       Chars_TO_Strg(Chars := #statDataBuffer.rcv_bddResult,
                     pChars := 2175,
                     Cnt := 8,
                     Strg => #statMonitoring.bddData.dataValue[90]);
       Chars_TO_Strg(Chars := #statDataBuffer.rcv_bddResult,
                     pChars := 2199,
                     Cnt := 8,
                     Strg => #statMonitoring.bddData.dataValue[91]);
       Chars_TO_Strg(Chars := #statDataBuffer.rcv_bddResult,
                     pChars := 2223,
                     Cnt := 8,
                     Strg => #statMonitoring.bddData.dataValue[92]);
       Chars_TO_Strg(Chars := #statDataBuffer.rcv_bddResult,
                     pChars := 2247,
                     Cnt := 8,
                     Strg => #statMonitoring.bddData.dataValue[93]);
       Chars_TO_Strg(Chars := #statDataBuffer.rcv_bddResult,
                     pChars := 2271,
                     Cnt := 8,
                     Strg => #statMonitoring.bddData.dataValue[94]);
       Chars_TO_Strg(Chars := #statDataBuffer.rcv_bddResult,
                     pChars := 2295,
                     Cnt := 8,
                     Strg => #statMonitoring.bddData.dataValue[95]);
       Chars_TO_Strg(Chars := #statDataBuffer.rcv_bddResult,
                     pChars := 2319,
                     Cnt := 8,
                     Strg => #statMonitoring.bddData.dataValue[96]);
       Chars_TO_Strg(Chars := #statDataBuffer.rcv_bddResult,
                     pChars := 2343,
                     Cnt := 8,
                     Strg => #statMonitoring.bddData.dataValue[97]);
       Chars_TO_Strg(Chars := #statDataBuffer.rcv_bddResult,
                     pChars := 2367,
                     Cnt := 8,
                     Strg => #statMonitoring.bddData.dataValue[98]);
       Chars_TO_Strg(Chars := #statDataBuffer.rcv_bddResult,
                     pChars := 2391,
                     Cnt := 8,
                     Strg => #statMonitoring.bddData.dataValue[99]);

       #instTON_bddResult[1](IN := TRUE,
                             PT := T#5000ms);

       IF #instTON_bddResult[1].Q THEN
           #statStep := 430;
       END_IF;
   END_IF;
END_REGION

REGION Network 43: STEP 430 : Bdd count complete
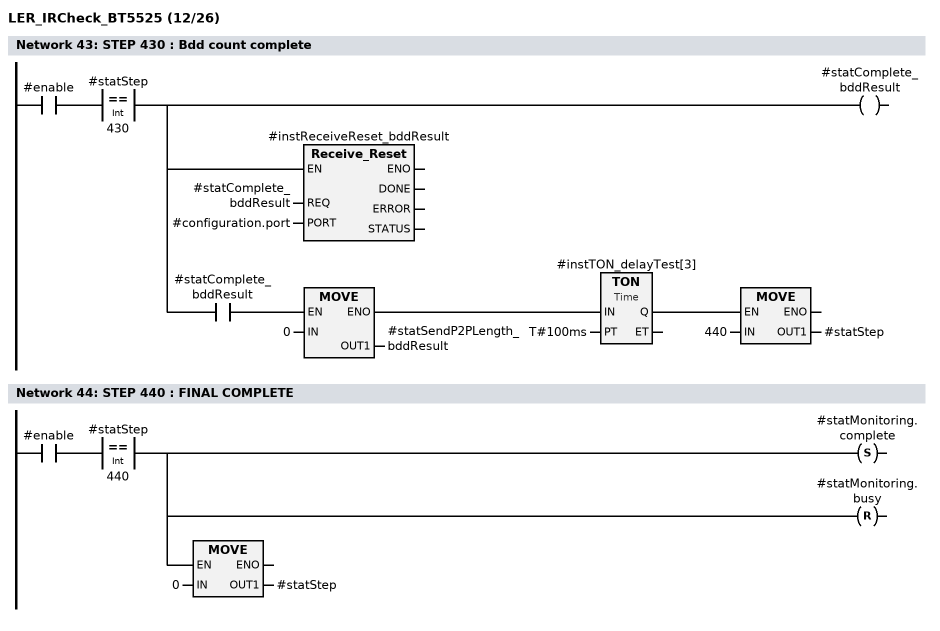
   RUNG wire#powerrail
      Contact( #enable )
      { S7_Templates := "SrcType := Int" } EQ_Contact(in1 := #statStep, in2 := 430)
      wire#w1
      Coil( #statComplete_bddResult )
   END_RUNG
   RUNG wire#w1
      #instReceiveReset_bddResult.Receive_Reset(REQ := #statComplete_bddResult, PORT := #configuration.port, DONE =>, ERROR =>, STATUS =>)
   END_RUNG
   RUNG wire#w1
      Contact( #statComplete_bddResult )
      Move(in := 0, out1 => #statSendP2PLength_bddResult)
      { S7_Templates := "time_type := Time" } #instTON_delayTest[3].TON(pt := T#100ms, et =>)
      Move(in := 440, out1 => #statStep)
   END_RUNG
   // the same network as SCL:
   #statComplete_bddResult := #enable AND (#statStep = 430);
   IF #statComplete_bddResult THEN
       #instReceiveReset_bddResult(REQ := #statComplete_bddResult, PORT := #configuration.port);   // Receive_Reset
   END_IF;
   #_w1 := #statComplete_bddResult AND #statComplete_bddResult;
   IF #_w1 THEN #statSendP2PLength_bddResult := 0; END_IF;
   #instTON_delayTest[3].TON(IN := #_w1, PT := T#100ms);
   IF #instTON_delayTest[3].Q THEN #statStep := 440; END_IF;
END_REGION

REGION Network 44: STEP 440 : FINAL COMPLETE
   RUNG wire#powerrail
      Contact( #enable )
      { S7_Templates := "SrcType := Int" } EQ_Contact(in1 := #statStep, in2 := 440)
      wire#w1
      S_Coil( #statMonitoring.complete )
   END_RUNG
   RUNG wire#w1
      R_Coil( #statMonitoring.busy )
   END_RUNG
   RUNG wire#w1
      Move(in := 0, out1 => #statStep)
   END_RUNG
   // the same network as SCL:
   IF #enable AND (#statStep = 440) THEN
       #statMonitoring.complete := TRUE;
       #statMonitoring.busy := FALSE;
       #statStep := 0;
   END_IF;
END_REGION

REGION Network 45: ========================================== SEQUENCE STEP [PARAMETER]
END_REGION

REGION Network 46: STEP 1000~1030 : VOLTAGE COMMAND
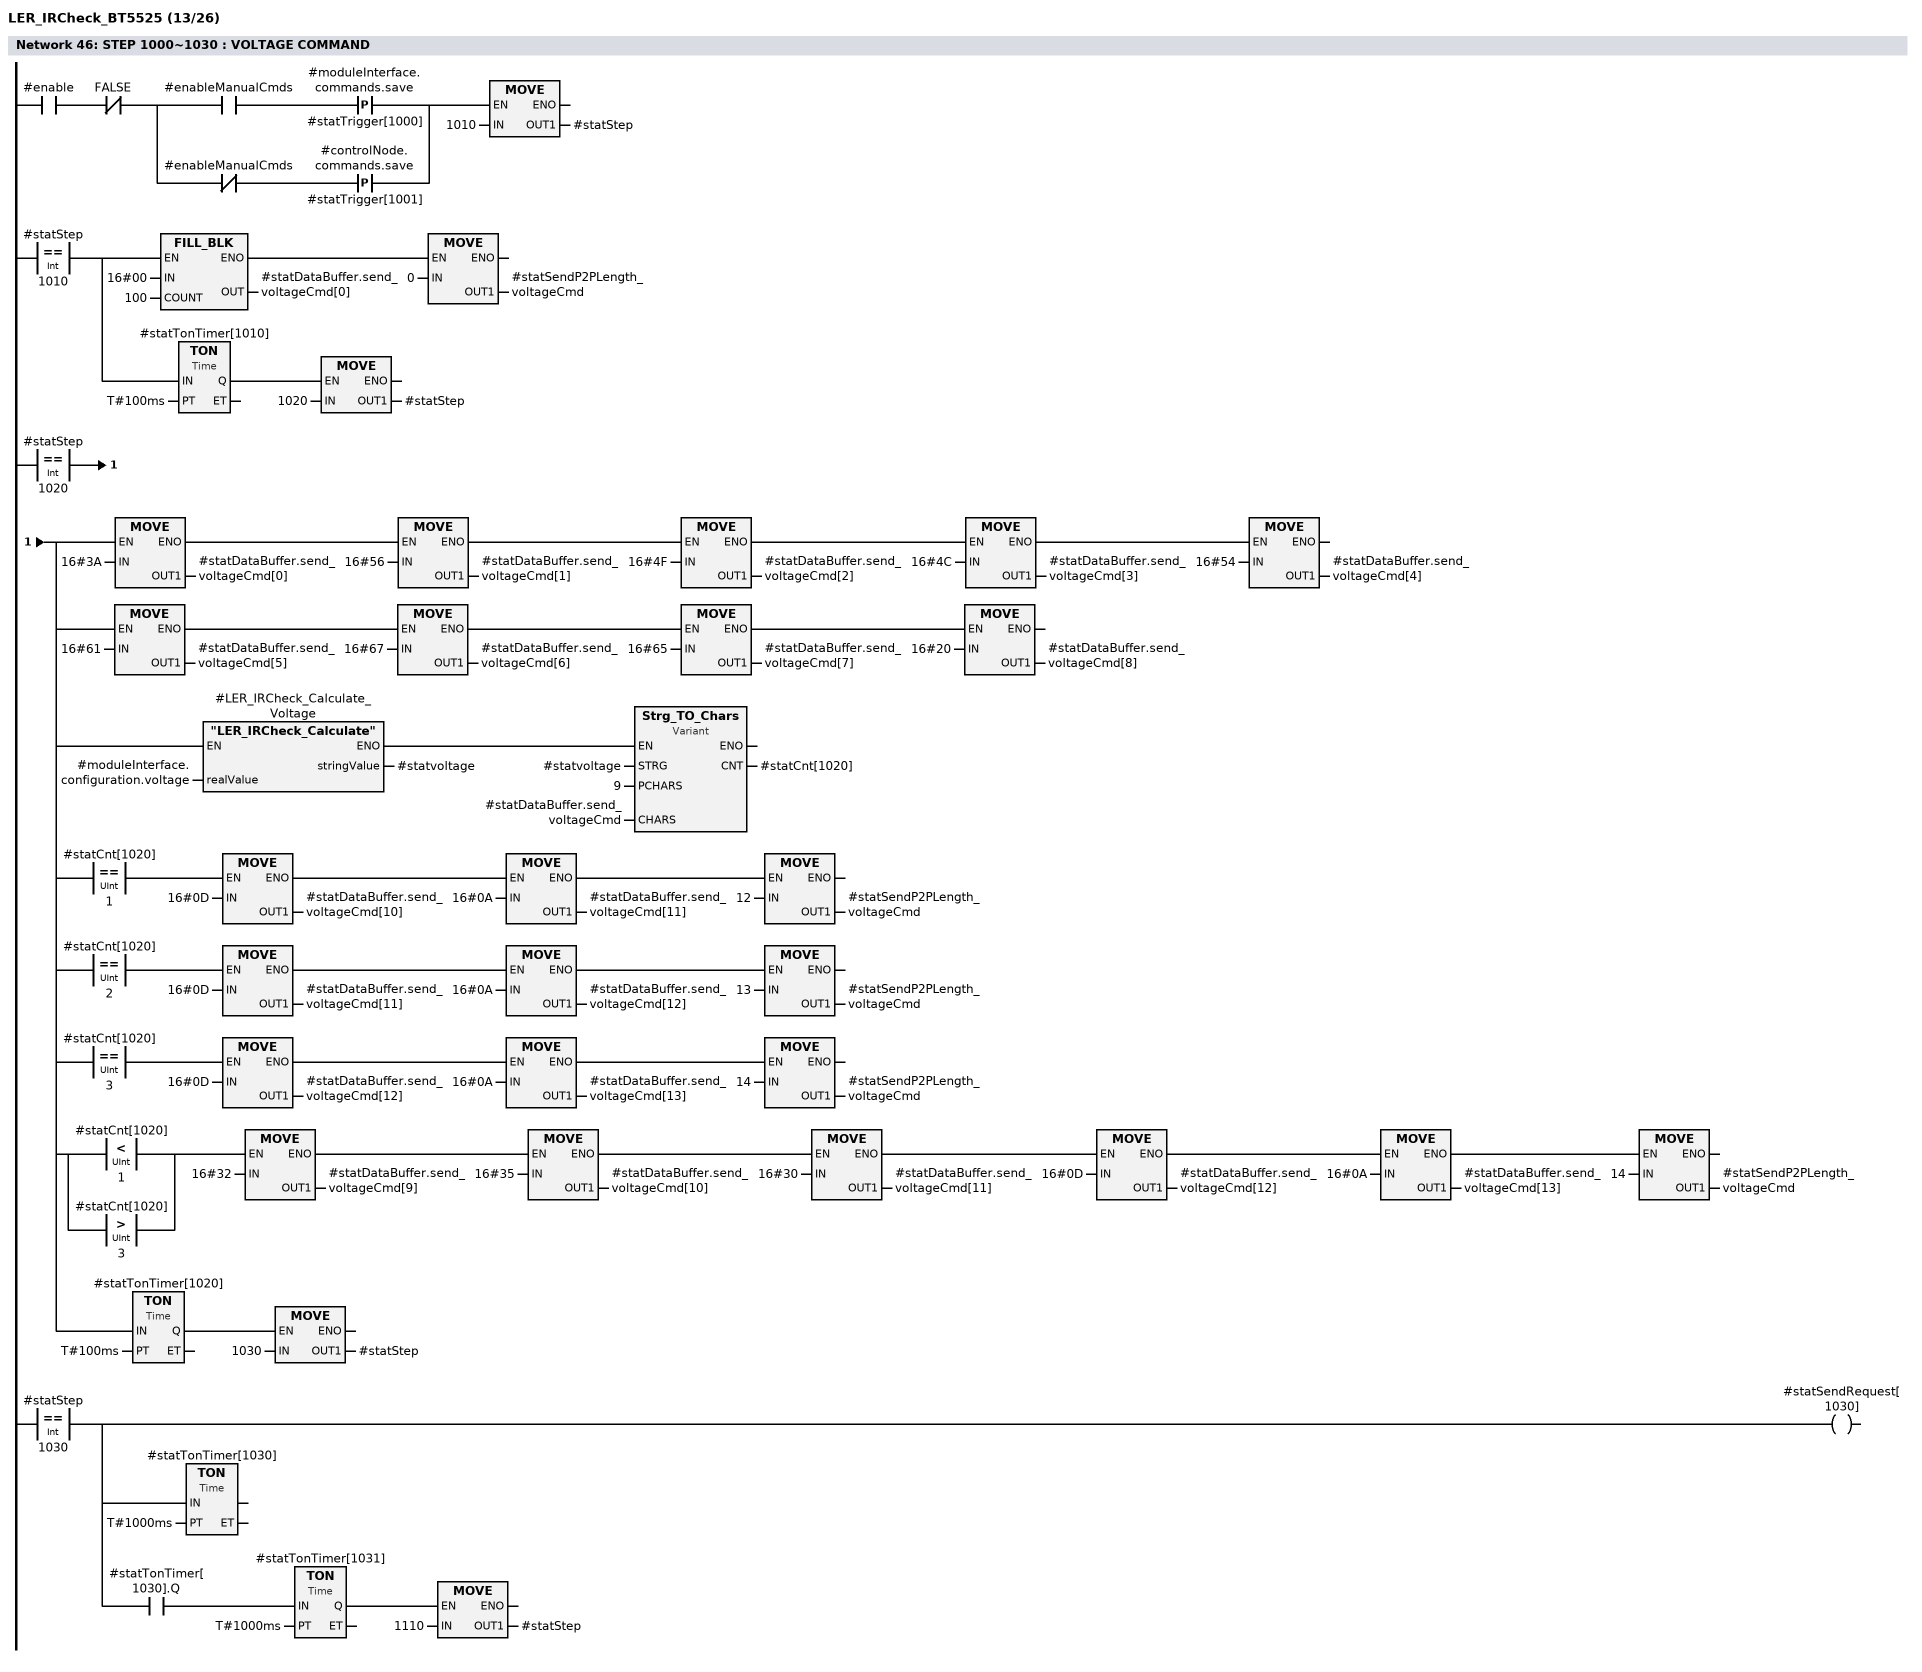
   RUNG wire#powerrail
      Contact( #enable )
      I_Contact( FALSE )
      wire#w1
      Contact( #enableManualCmds )
      P_Contact(operand := #moduleInterface.commands.save, bit := #statTrigger[1000])
      wire#w2
      Move(in := 1010, out1 => #statStep)
   END_RUNG
   RUNG wire#w1
      I_Contact( #enableManualCmds )
      P_Contact(operand := #controlNode.commands.save, bit := #statTrigger[1001])
   END_RUNG wire#w2
   RUNG wire#powerrail
      { S7_Templates := "SrcType := Int" } EQ_Contact(in1 := #statStep, in2 := 1010)
      wire#w3
      FillBlockI(in := 16#00, count := 100, out => #statDataBuffer.send_voltageCmd[0])
      Move(in := 0, out1 => #statSendP2PLength_voltageCmd)
   END_RUNG
   RUNG wire#w3
      { S7_Templates := "time_type := Time" } #statTonTimer[1010].TON(pt := T#100ms, et =>)
      Move(in := 1020, out1 => #statStep)
   END_RUNG
   RUNG wire#powerrail
      { S7_Templates := "SrcType := Int" } EQ_Contact(in1 := #statStep, in2 := 1020)
      wire#w4
      Move(in := 16#3A, out1 => #statDataBuffer.send_voltageCmd[0])
      Move(in := 16#56, out1 => #statDataBuffer.send_voltageCmd[1])
      Move(in := 16#4F, out1 => #statDataBuffer.send_voltageCmd[2])
      Move(in := 16#4C, out1 => #statDataBuffer.send_voltageCmd[3])
      Move(in := 16#54, out1 => #statDataBuffer.send_voltageCmd[4])
   END_RUNG
   RUNG wire#w4
      Move(in := 16#61, out1 => #statDataBuffer.send_voltageCmd[5])
      Move(in := 16#67, out1 => #statDataBuffer.send_voltageCmd[6])
      Move(in := 16#65, out1 => #statDataBuffer.send_voltageCmd[7])
      Move(in := 16#20, out1 => #statDataBuffer.send_voltageCmd[8])
   END_RUNG
   RUNG wire#w4
      #LER_IRCheck_Calculate_Voltage(realValue := #moduleInterface.configuration.voltage, stringValue => #statvoltage)
      { S7_Templates := "[ptr_type := Variant, strg_type := String]" } Strg_TO_Chars(Strg := #statvoltage, pChars := 9, Chars := #statDataBuffer.send_voltageCmd, Cnt => #statCnt[1020])
   END_RUNG
   RUNG wire#w4
      { S7_Templates := "SrcType := UInt" } EQ_Contact(in1 := #statCnt[1020], in2 := 1)
      Move(in := 16#0D, out1 => #statDataBuffer.send_voltageCmd[10])
      Move(in := 16#0A, out1 => #statDataBuffer.send_voltageCmd[11])
      Move(in := 12, out1 => #statSendP2PLength_voltageCmd)
   END_RUNG
   RUNG wire#w4
      { S7_Templates := "SrcType := UInt" } EQ_Contact(in1 := #statCnt[1020], in2 := 2)
      Move(in := 16#0D, out1 => #statDataBuffer.send_voltageCmd[11])
      Move(in := 16#0A, out1 => #statDataBuffer.send_voltageCmd[12])
      Move(in := 13, out1 => #statSendP2PLength_voltageCmd)
   END_RUNG
   RUNG wire#w4
      { S7_Templates := "SrcType := UInt" } EQ_Contact(in1 := #statCnt[1020], in2 := 3)
      Move(in := 16#0D, out1 => #statDataBuffer.send_voltageCmd[12])
      Move(in := 16#0A, out1 => #statDataBuffer.send_voltageCmd[13])
      Move(in := 14, out1 => #statSendP2PLength_voltageCmd)
   END_RUNG
   RUNG wire#w4
      { S7_Templates := "SrcType := UInt" } LT_Contact(in1 := #statCnt[1020], in2 := 1)
      wire#w5
      Move(in := 16#32, out1 => #statDataBuffer.send_voltageCmd[9])
      Move(in := 16#35, out1 => #statDataBuffer.send_voltageCmd[10])
      Move(in := 16#30, out1 => #statDataBuffer.send_voltageCmd[11])
      Move(in := 16#0D, out1 => #statDataBuffer.send_voltageCmd[12])
      Move(in := 16#0A, out1 => #statDataBuffer.send_voltageCmd[13])
      Move(in := 14, out1 => #statSendP2PLength_voltageCmd)
   END_RUNG
   RUNG wire#w4
      { S7_Templates := "SrcType := UInt" } GT_Contact(in1 := #statCnt[1020], in2 := 3)
   END_RUNG wire#w5
   RUNG wire#w4
      { S7_Templates := "time_type := Time" } #statTonTimer[1020].TON(pt := T#100ms, et =>)
      Move(in := 1030, out1 => #statStep)
   END_RUNG
   RUNG wire#powerrail
      { S7_Templates := "SrcType := Int" } EQ_Contact(in1 := #statStep, in2 := 1030)
      wire#w6
      Coil( #statSendRequest[1030] )
   END_RUNG
   RUNG wire#w6
      { S7_Templates := "time_type := Time" } #statTonTimer[1030].TON(pt := T#1000ms, et =>)
   END_RUNG
   RUNG wire#w6
      Contact( #statTonTimer[1030].Q )
      { S7_Templates := "time_type := Time" } #statTonTimer[1031].TON(pt := T#1000ms, et =>)
      Move(in := 1110, out1 => #statStep)
   END_RUNG
   // the same network as SCL:
   #_w1 := #enable AND NOT FALSE AND #enableManualCmds AND #moduleInterface.commands.save AND NOT #statTrigger[1000];   // rising edge of #moduleInterface.commands.save
   #statTrigger[1000] := #moduleInterface.commands.save;
   #_w2 := #enable AND NOT FALSE AND NOT #enableManualCmds AND #controlNode.commands.save AND NOT #statTrigger[1001];   // rising edge of #controlNode.commands.save
   #statTrigger[1001] := #controlNode.commands.save;
   IF #_w1 OR #_w2 THEN #statStep := 1010; END_IF;
   #_w3 := #statStep = 1010;
   IF #_w3 THEN
       FILL_BLK(IN := 16#00, COUNT := 100, OUT => #statDataBuffer.send_voltageCmd[0]);
       #statSendP2PLength_voltageCmd := 0;
   END_IF;
   #statTonTimer[1010].TON(IN := #_w3, PT := T#100ms);
   IF #statTonTimer[1010].Q THEN #statStep := 1020; END_IF;
   #_w4 := #statStep = 1020;
   IF #_w4 THEN
       #statDataBuffer.send_voltageCmd[0] := 16#3A;
       #statDataBuffer.send_voltageCmd[1] := 16#56;
       #statDataBuffer.send_voltageCmd[2] := 16#4F;
       #statDataBuffer.send_voltageCmd[3] := 16#4C;
       #statDataBuffer.send_voltageCmd[4] := 16#54;
       #statDataBuffer.send_voltageCmd[5] := 16#61;
       #statDataBuffer.send_voltageCmd[6] := 16#67;
       #statDataBuffer.send_voltageCmd[7] := 16#65;
       #statDataBuffer.send_voltageCmd[8] := 16#20;
   END_IF;
   #LER_IRCheck_Calculate_Voltage(EN := #_w4,   // "LER_IRCheck_Calculate"
                           realValue := #moduleInterface.configuration.voltage,
                           stringValue => #statvoltage,
                           ENO => #_w5);
   IF #_w5 THEN
       Strg_TO_Chars(Strg := #statvoltage,
                     pChars := 9,
                     Chars := #statDataBuffer.send_voltageCmd,
                     Cnt => #statCnt[1020]);
   END_IF;
   IF #_w4 AND (#statCnt[1020] = 1) THEN
       #statDataBuffer.send_voltageCmd[10] := 16#0D;
       #statDataBuffer.send_voltageCmd[11] := 16#0A;
       #statSendP2PLength_voltageCmd := 12;
   END_IF;
   IF #_w4 AND (#statCnt[1020] = 2) THEN
       #statDataBuffer.send_voltageCmd[11] := 16#0D;
       #statDataBuffer.send_voltageCmd[12] := 16#0A;
       #statSendP2PLength_voltageCmd := 13;
   END_IF;
   IF #_w4 AND (#statCnt[1020] = 3) THEN
       #statDataBuffer.send_voltageCmd[12] := 16#0D;
       #statDataBuffer.send_voltageCmd[13] := 16#0A;
       #statSendP2PLength_voltageCmd := 14;
   END_IF;
   IF #_w4 AND ((#statCnt[1020] < 1) OR (#statCnt[1020] > 3)) THEN
       #statDataBuffer.send_voltageCmd[9] := 16#32;
       #statDataBuffer.send_voltageCmd[10] := 16#35;
       #statDataBuffer.send_voltageCmd[11] := 16#30;
       #statDataBuffer.send_voltageCmd[12] := 16#0D;
       #statDataBuffer.send_voltageCmd[13] := 16#0A;
       #statSendP2PLength_voltageCmd := 14;
   END_IF;
   #statTonTimer[1020].TON(IN := #_w4, PT := T#100ms);
   IF #statTonTimer[1020].Q THEN #statStep := 1030; END_IF;
   #statSendRequest[1030] := #statStep = 1030;
   #statTonTimer[1030].TON(IN := #statStep = 1030, PT := T#1000ms);
   #statTonTimer[1031].TON(IN := (#statStep = 1030) AND #statTonTimer[1030].Q, PT := T#1000ms);
   IF #statTonTimer[1031].Q THEN #statStep := 1110; END_IF;
END_REGION

REGION Network 47: STEP 1110~1140 : VOLTAGE CHECK
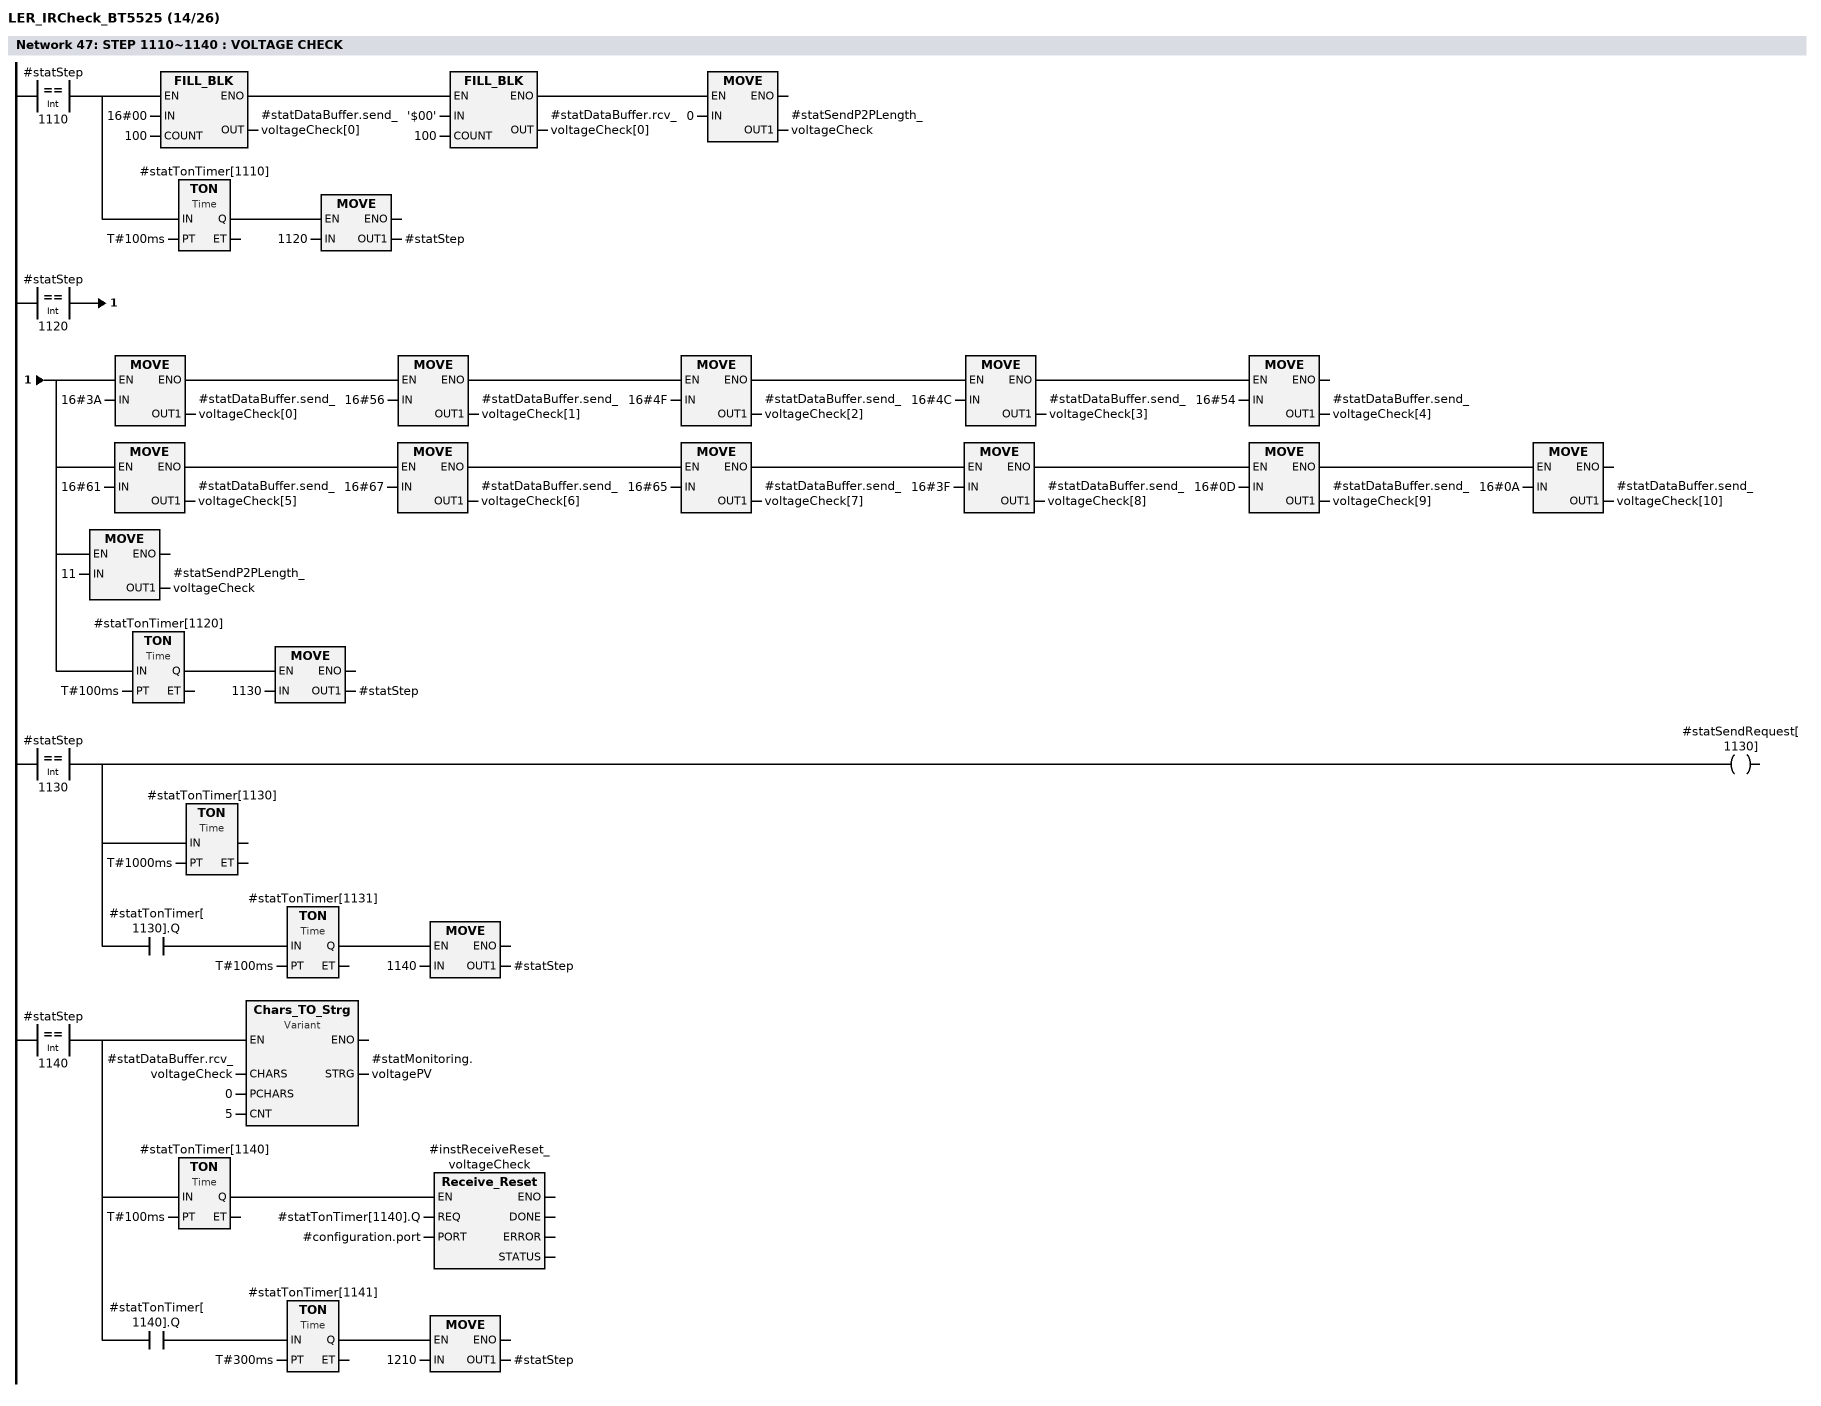
   RUNG wire#powerrail
      { S7_Templates := "SrcType := Int" } EQ_Contact(in1 := #statStep, in2 := 1110)
      wire#w1
      FillBlockI(in := 16#00, count := 100, out => #statDataBuffer.send_voltageCheck[0])
      FillBlockI(in := '$00', count := 100, out => #statDataBuffer.rcv_voltageCheck[0])
      Move(in := 0, out1 => #statSendP2PLength_voltageCheck)
   END_RUNG
   RUNG wire#w1
      { S7_Templates := "time_type := Time" } #statTonTimer[1110].TON(pt := T#100ms, et =>)
      Move(in := 1120, out1 => #statStep)
   END_RUNG
   RUNG wire#powerrail
      { S7_Templates := "SrcType := Int" } EQ_Contact(in1 := #statStep, in2 := 1120)
      wire#w2
      Move(in := 16#3A, out1 => #statDataBuffer.send_voltageCheck[0])
      Move(in := 16#56, out1 => #statDataBuffer.send_voltageCheck[1])
      Move(in := 16#4F, out1 => #statDataBuffer.send_voltageCheck[2])
      Move(in := 16#4C, out1 => #statDataBuffer.send_voltageCheck[3])
      Move(in := 16#54, out1 => #statDataBuffer.send_voltageCheck[4])
   END_RUNG
   RUNG wire#w2
      Move(in := 16#61, out1 => #statDataBuffer.send_voltageCheck[5])
      Move(in := 16#67, out1 => #statDataBuffer.send_voltageCheck[6])
      Move(in := 16#65, out1 => #statDataBuffer.send_voltageCheck[7])
      Move(in := 16#3F, out1 => #statDataBuffer.send_voltageCheck[8])
      Move(in := 16#0D, out1 => #statDataBuffer.send_voltageCheck[9])
      Move(in := 16#0A, out1 => #statDataBuffer.send_voltageCheck[10])
   END_RUNG
   RUNG wire#w2
      Move(in := 11, out1 => #statSendP2PLength_voltageCheck)
   END_RUNG
   RUNG wire#w2
      { S7_Templates := "time_type := Time" } #statTonTimer[1120].TON(pt := T#100ms, et =>)
      Move(in := 1130, out1 => #statStep)
   END_RUNG
   RUNG wire#powerrail
      { S7_Templates := "SrcType := Int" } EQ_Contact(in1 := #statStep, in2 := 1130)
      wire#w3
      Coil( #statSendRequest[1130] )
   END_RUNG
   RUNG wire#w3
      { S7_Templates := "time_type := Time" } #statTonTimer[1130].TON(pt := T#1000ms, et =>)
   END_RUNG
   RUNG wire#w3
      Contact( #statTonTimer[1130].Q )
      { S7_Templates := "time_type := Time" } #statTonTimer[1131].TON(pt := T#100ms, et =>)
      Move(in := 1140, out1 => #statStep)
   END_RUNG
   RUNG wire#powerrail
      { S7_Templates := "SrcType := Int" } EQ_Contact(in1 := #statStep, in2 := 1140)
      wire#w4
      { S7_Templates := "[ptr_type := Variant, str_type := String]" } Chars_TO_Strg(Chars := #statDataBuffer.rcv_voltageCheck, pChars := 0, Cnt := 5, Strg => #statMonitoring.voltagePV)
   END_RUNG
   RUNG wire#w4
      { S7_Templates := "time_type := Time" } #statTonTimer[1140].TON(pt := T#100ms, et =>)
      #instReceiveReset_voltageCheck.Receive_Reset(REQ := #statTonTimer[1140].Q, PORT := #configuration.port, DONE =>, ERROR =>, STATUS =>)
   END_RUNG
   RUNG wire#w4
      Contact( #statTonTimer[1140].Q )
      { S7_Templates := "time_type := Time" } #statTonTimer[1141].TON(pt := T#300ms, et =>)
      Move(in := 1210, out1 => #statStep)
   END_RUNG
   // the same network as SCL:
   #_w1 := #statStep = 1110;
   IF #_w1 THEN
       FILL_BLK(IN := 16#00, COUNT := 100, OUT => #statDataBuffer.send_voltageCheck[0]);
       FILL_BLK(IN := '$00', COUNT := 100, OUT => #statDataBuffer.rcv_voltageCheck[0]);
       #statSendP2PLength_voltageCheck := 0;
   END_IF;
   #statTonTimer[1110].TON(IN := #_w1, PT := T#100ms);
   IF #statTonTimer[1110].Q THEN #statStep := 1120; END_IF;
   #_w2 := #statStep = 1120;
   IF #_w2 THEN
       #statDataBuffer.send_voltageCheck[0] := 16#3A;
       #statDataBuffer.send_voltageCheck[1] := 16#56;
       #statDataBuffer.send_voltageCheck[2] := 16#4F;
       #statDataBuffer.send_voltageCheck[3] := 16#4C;
       #statDataBuffer.send_voltageCheck[4] := 16#54;
       #statDataBuffer.send_voltageCheck[5] := 16#61;
       #statDataBuffer.send_voltageCheck[6] := 16#67;
       #statDataBuffer.send_voltageCheck[7] := 16#65;
       #statDataBuffer.send_voltageCheck[8] := 16#3F;
       #statDataBuffer.send_voltageCheck[9] := 16#0D;
       #statDataBuffer.send_voltageCheck[10] := 16#0A;
       #statSendP2PLength_voltageCheck := 11;
   END_IF;
   #statTonTimer[1120].TON(IN := #_w2, PT := T#100ms);
   IF #statTonTimer[1120].Q THEN #statStep := 1130; END_IF;
   #statSendRequest[1130] := #statStep = 1130;
   #statTonTimer[1130].TON(IN := #statStep = 1130, PT := T#1000ms);
   #statTonTimer[1131].TON(IN := (#statStep = 1130) AND #statTonTimer[1130].Q, PT := T#100ms);
   IF #statTonTimer[1131].Q THEN #statStep := 1140; END_IF;
   #_w3 := #statStep = 1140;
   IF #_w3 THEN
       Chars_TO_Strg(Chars := #statDataBuffer.rcv_voltageCheck,
                     pChars := 0,
                     Cnt := 5,
                     Strg => #statMonitoring.voltagePV);
   END_IF;
   #statTonTimer[1140].TON(IN := #_w3, PT := T#100ms);
   IF #statTonTimer[1140].Q THEN
       #instReceiveReset_voltageCheck(REQ := #statTonTimer[1140].Q, PORT := #configuration.port);   // Receive_Reset
   END_IF;
   #statTonTimer[1141].TON(IN := #_w3 AND #statTonTimer[1140].Q, PT := T#300ms);
   IF #statTonTimer[1141].Q THEN #statStep := 1210; END_IF;
END_REGION

REGION Network 48: STEP 1210~1230 : TIMER COMMAND
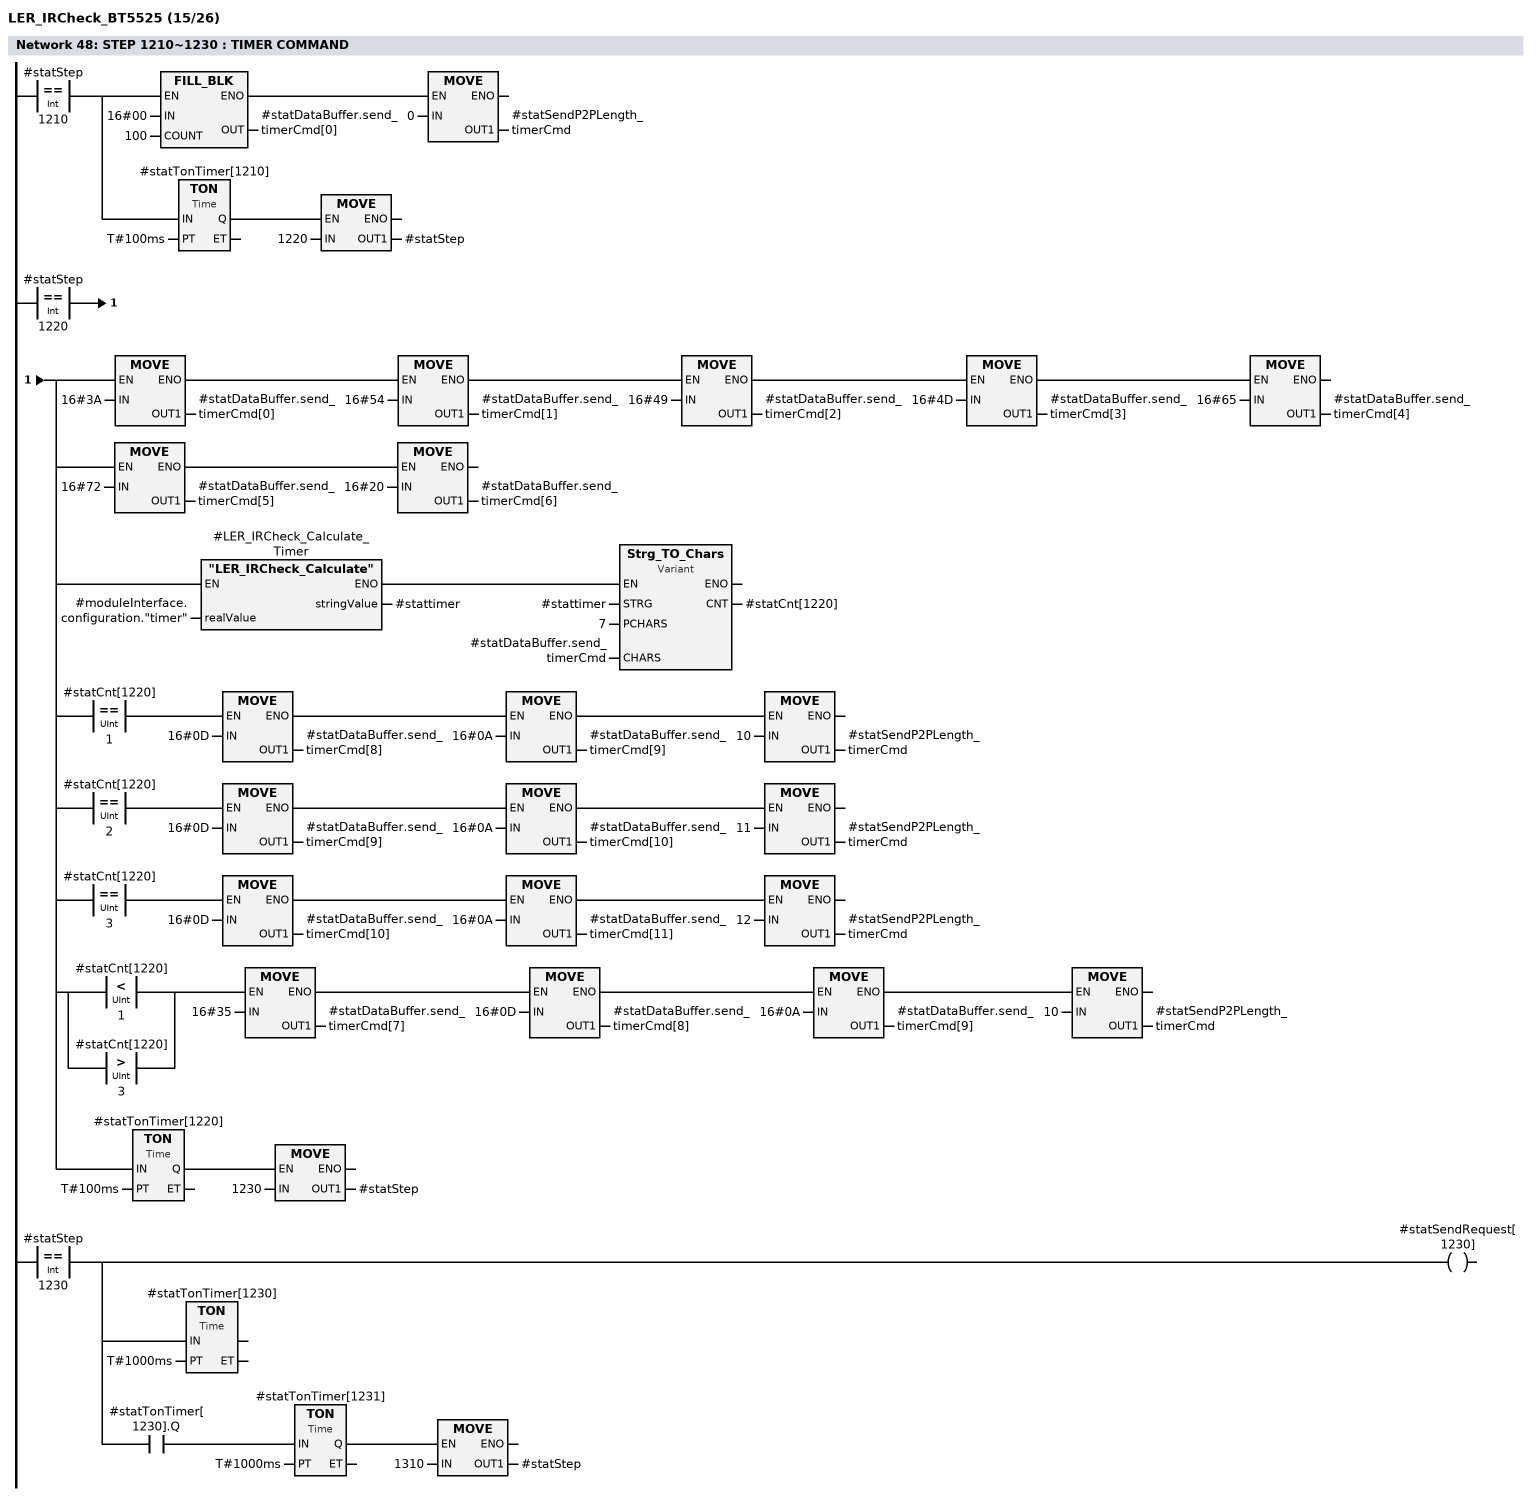
   RUNG wire#powerrail
      { S7_Templates := "SrcType := Int" } EQ_Contact(in1 := #statStep, in2 := 1210)
      wire#w1
      FillBlockI(in := 16#00, count := 100, out => #statDataBuffer.send_timerCmd[0])
      Move(in := 0, out1 => #statSendP2PLength_timerCmd)
   END_RUNG
   RUNG wire#w1
      { S7_Templates := "time_type := Time" } #statTonTimer[1210].TON(pt := T#100ms, et =>)
      Move(in := 1220, out1 => #statStep)
   END_RUNG
   RUNG wire#powerrail
      { S7_Templates := "SrcType := Int" } EQ_Contact(in1 := #statStep, in2 := 1220)
      wire#w2
      Move(in := 16#3A, out1 => #statDataBuffer.send_timerCmd[0])
      Move(in := 16#54, out1 => #statDataBuffer.send_timerCmd[1])
      Move(in := 16#49, out1 => #statDataBuffer.send_timerCmd[2])
      Move(in := 16#4D, out1 => #statDataBuffer.send_timerCmd[3])
      Move(in := 16#65, out1 => #statDataBuffer.send_timerCmd[4])
   END_RUNG
   RUNG wire#w2
      Move(in := 16#72, out1 => #statDataBuffer.send_timerCmd[5])
      Move(in := 16#20, out1 => #statDataBuffer.send_timerCmd[6])
   END_RUNG
   RUNG wire#w2
      #LER_IRCheck_Calculate_Timer(realValue := #moduleInterface.configuration."timer", stringValue => #stattimer)
      { S7_Templates := "[ptr_type := Variant, strg_type := String]" } Strg_TO_Chars(Strg := #stattimer, pChars := 7, Chars := #statDataBuffer.send_timerCmd, Cnt => #statCnt[1220])
   END_RUNG
   RUNG wire#w2
      { S7_Templates := "SrcType := UInt" } EQ_Contact(in1 := #statCnt[1220], in2 := 1)
      Move(in := 16#0D, out1 => #statDataBuffer.send_timerCmd[8])
      Move(in := 16#0A, out1 => #statDataBuffer.send_timerCmd[9])
      Move(in := 10, out1 => #statSendP2PLength_timerCmd)
   END_RUNG
   RUNG wire#w2
      { S7_Templates := "SrcType := UInt" } EQ_Contact(in1 := #statCnt[1220], in2 := 2)
      Move(in := 16#0D, out1 => #statDataBuffer.send_timerCmd[9])
      Move(in := 16#0A, out1 => #statDataBuffer.send_timerCmd[10])
      Move(in := 11, out1 => #statSendP2PLength_timerCmd)
   END_RUNG
   RUNG wire#w2
      { S7_Templates := "SrcType := UInt" } EQ_Contact(in1 := #statCnt[1220], in2 := 3)
      Move(in := 16#0D, out1 => #statDataBuffer.send_timerCmd[10])
      Move(in := 16#0A, out1 => #statDataBuffer.send_timerCmd[11])
      Move(in := 12, out1 => #statSendP2PLength_timerCmd)
   END_RUNG
   RUNG wire#w2
      { S7_Templates := "SrcType := UInt" } LT_Contact(in1 := #statCnt[1220], in2 := 1)
      wire#w3
      Move(in := 16#35, out1 => #statDataBuffer.send_timerCmd[7])
      Move(in := 16#0D, out1 => #statDataBuffer.send_timerCmd[8])
      Move(in := 16#0A, out1 => #statDataBuffer.send_timerCmd[9])
      Move(in := 10, out1 => #statSendP2PLength_timerCmd)
   END_RUNG
   RUNG wire#w2
      { S7_Templates := "SrcType := UInt" } GT_Contact(in1 := #statCnt[1220], in2 := 3)
   END_RUNG wire#w3
   RUNG wire#w2
      { S7_Templates := "time_type := Time" } #statTonTimer[1220].TON(pt := T#100ms, et =>)
      Move(in := 1230, out1 => #statStep)
   END_RUNG
   RUNG wire#powerrail
      { S7_Templates := "SrcType := Int" } EQ_Contact(in1 := #statStep, in2 := 1230)
      wire#w4
      Coil( #statSendRequest[1230] )
   END_RUNG
   RUNG wire#w4
      { S7_Templates := "time_type := Time" } #statTonTimer[1230].TON(pt := T#1000ms, et =>)
   END_RUNG
   RUNG wire#w4
      Contact( #statTonTimer[1230].Q )
      { S7_Templates := "time_type := Time" } #statTonTimer[1231].TON(pt := T#1000ms, et =>)
      Move(in := 1310, out1 => #statStep)
   END_RUNG
   // the same network as SCL:
   #_w1 := #statStep = 1210;
   IF #_w1 THEN
       FILL_BLK(IN := 16#00, COUNT := 100, OUT => #statDataBuffer.send_timerCmd[0]);
       #statSendP2PLength_timerCmd := 0;
   END_IF;
   #statTonTimer[1210].TON(IN := #_w1, PT := T#100ms);
   IF #statTonTimer[1210].Q THEN #statStep := 1220; END_IF;
   #_w2 := #statStep = 1220;
   IF #_w2 THEN
       #statDataBuffer.send_timerCmd[0] := 16#3A;
       #statDataBuffer.send_timerCmd[1] := 16#54;
       #statDataBuffer.send_timerCmd[2] := 16#49;
       #statDataBuffer.send_timerCmd[3] := 16#4D;
       #statDataBuffer.send_timerCmd[4] := 16#65;
       #statDataBuffer.send_timerCmd[5] := 16#72;
       #statDataBuffer.send_timerCmd[6] := 16#20;
   END_IF;
   #LER_IRCheck_Calculate_Timer(EN := #_w2,   // "LER_IRCheck_Calculate"
                           realValue := #moduleInterface.configuration."timer",
                           stringValue => #stattimer,
                           ENO => #_w3);
   IF #_w3 THEN
       Strg_TO_Chars(Strg := #stattimer, pChars := 7, Chars := #statDataBuffer.send_timerCmd, Cnt => #statCnt[1220]);
   END_IF;
   IF #_w2 AND (#statCnt[1220] = 1) THEN
       #statDataBuffer.send_timerCmd[8] := 16#0D;
       #statDataBuffer.send_timerCmd[9] := 16#0A;
       #statSendP2PLength_timerCmd := 10;
   END_IF;
   IF #_w2 AND (#statCnt[1220] = 2) THEN
       #statDataBuffer.send_timerCmd[9] := 16#0D;
       #statDataBuffer.send_timerCmd[10] := 16#0A;
       #statSendP2PLength_timerCmd := 11;
   END_IF;
   IF #_w2 AND (#statCnt[1220] = 3) THEN
       #statDataBuffer.send_timerCmd[10] := 16#0D;
       #statDataBuffer.send_timerCmd[11] := 16#0A;
       #statSendP2PLength_timerCmd := 12;
   END_IF;
   IF #_w2 AND ((#statCnt[1220] < 1) OR (#statCnt[1220] > 3)) THEN
       #statDataBuffer.send_timerCmd[7] := 16#35;
       #statDataBuffer.send_timerCmd[8] := 16#0D;
       #statDataBuffer.send_timerCmd[9] := 16#0A;
       #statSendP2PLength_timerCmd := 10;
   END_IF;
   #statTonTimer[1220].TON(IN := #_w2, PT := T#100ms);
   IF #statTonTimer[1220].Q THEN #statStep := 1230; END_IF;
   #statSendRequest[1230] := #statStep = 1230;
   #statTonTimer[1230].TON(IN := #statStep = 1230, PT := T#1000ms);
   #statTonTimer[1231].TON(IN := (#statStep = 1230) AND #statTonTimer[1230].Q, PT := T#1000ms);
   IF #statTonTimer[1231].Q THEN #statStep := 1310; END_IF;
END_REGION

REGION Network 49: STEP 1310~1340 : TIMER CHECK
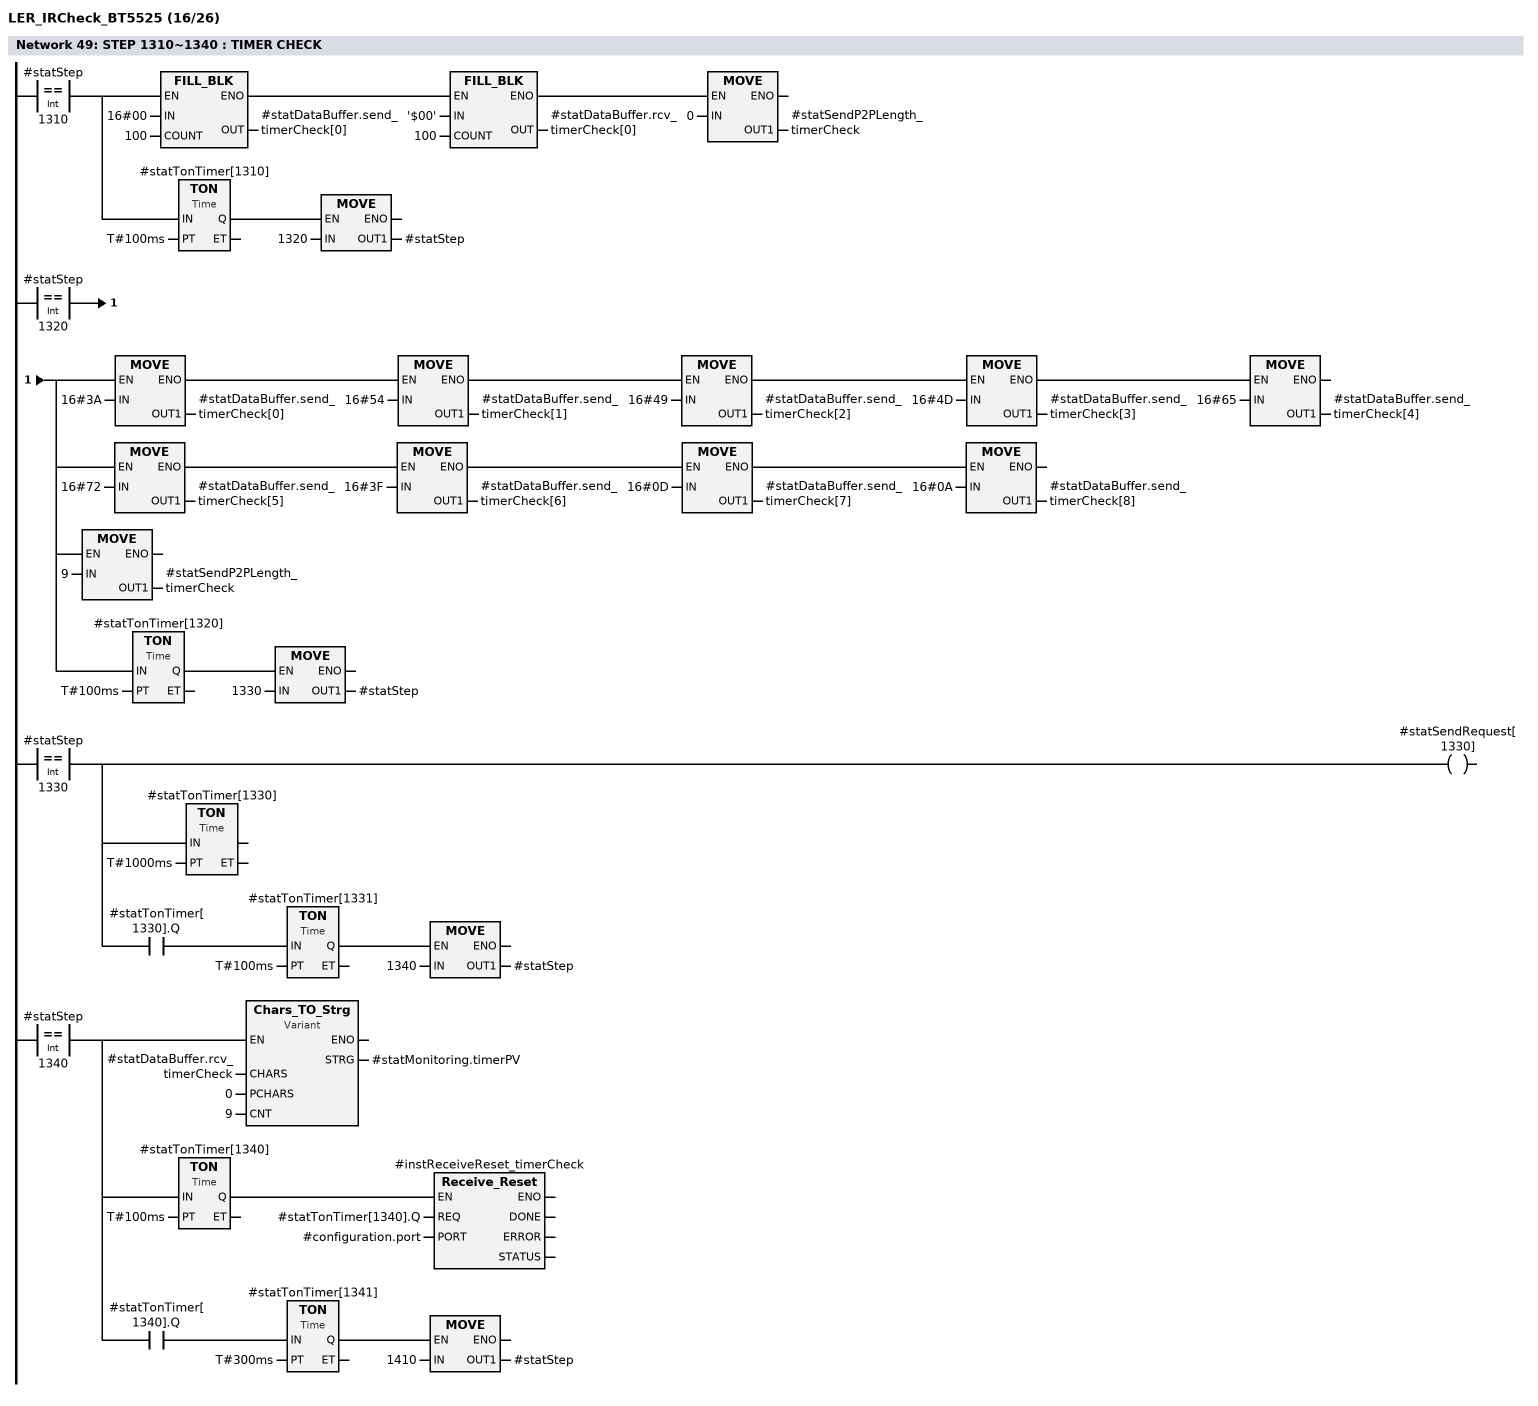
   RUNG wire#powerrail
      { S7_Templates := "SrcType := Int" } EQ_Contact(in1 := #statStep, in2 := 1310)
      wire#w1
      FillBlockI(in := 16#00, count := 100, out => #statDataBuffer.send_timerCheck[0])
      FillBlockI(in := '$00', count := 100, out => #statDataBuffer.rcv_timerCheck[0])
      Move(in := 0, out1 => #statSendP2PLength_timerCheck)
   END_RUNG
   RUNG wire#w1
      { S7_Templates := "time_type := Time" } #statTonTimer[1310].TON(pt := T#100ms, et =>)
      Move(in := 1320, out1 => #statStep)
   END_RUNG
   RUNG wire#powerrail
      { S7_Templates := "SrcType := Int" } EQ_Contact(in1 := #statStep, in2 := 1320)
      wire#w2
      Move(in := 16#3A, out1 => #statDataBuffer.send_timerCheck[0])
      Move(in := 16#54, out1 => #statDataBuffer.send_timerCheck[1])
      Move(in := 16#49, out1 => #statDataBuffer.send_timerCheck[2])
      Move(in := 16#4D, out1 => #statDataBuffer.send_timerCheck[3])
      Move(in := 16#65, out1 => #statDataBuffer.send_timerCheck[4])
   END_RUNG
   RUNG wire#w2
      Move(in := 16#72, out1 => #statDataBuffer.send_timerCheck[5])
      Move(in := 16#3F, out1 => #statDataBuffer.send_timerCheck[6])
      Move(in := 16#0D, out1 => #statDataBuffer.send_timerCheck[7])
      Move(in := 16#0A, out1 => #statDataBuffer.send_timerCheck[8])
   END_RUNG
   RUNG wire#w2
      Move(in := 9, out1 => #statSendP2PLength_timerCheck)
   END_RUNG
   RUNG wire#w2
      { S7_Templates := "time_type := Time" } #statTonTimer[1320].TON(pt := T#100ms, et =>)
      Move(in := 1330, out1 => #statStep)
   END_RUNG
   RUNG wire#powerrail
      { S7_Templates := "SrcType := Int" } EQ_Contact(in1 := #statStep, in2 := 1330)
      wire#w3
      Coil( #statSendRequest[1330] )
   END_RUNG
   RUNG wire#w3
      { S7_Templates := "time_type := Time" } #statTonTimer[1330].TON(pt := T#1000ms, et =>)
   END_RUNG
   RUNG wire#w3
      Contact( #statTonTimer[1330].Q )
      { S7_Templates := "time_type := Time" } #statTonTimer[1331].TON(pt := T#100ms, et =>)
      Move(in := 1340, out1 => #statStep)
   END_RUNG
   RUNG wire#powerrail
      { S7_Templates := "SrcType := Int" } EQ_Contact(in1 := #statStep, in2 := 1340)
      wire#w4
      { S7_Templates := "[ptr_type := Variant, str_type := String]" } Chars_TO_Strg(Chars := #statDataBuffer.rcv_timerCheck, pChars := 0, Cnt := 9, Strg => #statMonitoring.timerPV)
   END_RUNG
   RUNG wire#w4
      { S7_Templates := "time_type := Time" } #statTonTimer[1340].TON(pt := T#100ms, et =>)
      #instReceiveReset_timerCheck.Receive_Reset(REQ := #statTonTimer[1340].Q, PORT := #configuration.port, DONE =>, ERROR =>, STATUS =>)
   END_RUNG
   RUNG wire#w4
      Contact( #statTonTimer[1340].Q )
      { S7_Templates := "time_type := Time" } #statTonTimer[1341].TON(pt := T#300ms, et =>)
      Move(in := 1410, out1 => #statStep)
   END_RUNG
   // the same network as SCL:
   #_w1 := #statStep = 1310;
   IF #_w1 THEN
       FILL_BLK(IN := 16#00, COUNT := 100, OUT => #statDataBuffer.send_timerCheck[0]);
       FILL_BLK(IN := '$00', COUNT := 100, OUT => #statDataBuffer.rcv_timerCheck[0]);
       #statSendP2PLength_timerCheck := 0;
   END_IF;
   #statTonTimer[1310].TON(IN := #_w1, PT := T#100ms);
   IF #statTonTimer[1310].Q THEN #statStep := 1320; END_IF;
   #_w2 := #statStep = 1320;
   IF #_w2 THEN
       #statDataBuffer.send_timerCheck[0] := 16#3A;
       #statDataBuffer.send_timerCheck[1] := 16#54;
       #statDataBuffer.send_timerCheck[2] := 16#49;
       #statDataBuffer.send_timerCheck[3] := 16#4D;
       #statDataBuffer.send_timerCheck[4] := 16#65;
       #statDataBuffer.send_timerCheck[5] := 16#72;
       #statDataBuffer.send_timerCheck[6] := 16#3F;
       #statDataBuffer.send_timerCheck[7] := 16#0D;
       #statDataBuffer.send_timerCheck[8] := 16#0A;
       #statSendP2PLength_timerCheck := 9;
   END_IF;
   #statTonTimer[1320].TON(IN := #_w2, PT := T#100ms);
   IF #statTonTimer[1320].Q THEN #statStep := 1330; END_IF;
   #statSendRequest[1330] := #statStep = 1330;
   #statTonTimer[1330].TON(IN := #statStep = 1330, PT := T#1000ms);
   #statTonTimer[1331].TON(IN := (#statStep = 1330) AND #statTonTimer[1330].Q, PT := T#100ms);
   IF #statTonTimer[1331].Q THEN #statStep := 1340; END_IF;
   #_w3 := #statStep = 1340;
   IF #_w3 THEN
       Chars_TO_Strg(Chars := #statDataBuffer.rcv_timerCheck,
                     pChars := 0,
                     Cnt := 9,
                     Strg => #statMonitoring.timerPV);
   END_IF;
   #statTonTimer[1340].TON(IN := #_w3, PT := T#100ms);
   IF #statTonTimer[1340].Q THEN
       #instReceiveReset_timerCheck(REQ := #statTonTimer[1340].Q, PORT := #configuration.port);   // Receive_Reset
   END_IF;
   #statTonTimer[1341].TON(IN := #_w3 AND #statTonTimer[1340].Q, PT := T#300ms);
   IF #statTonTimer[1341].Q THEN #statStep := 1410; END_IF;
END_REGION

REGION Network 50: STEP 1410~1430 : CONTACT COMMAND
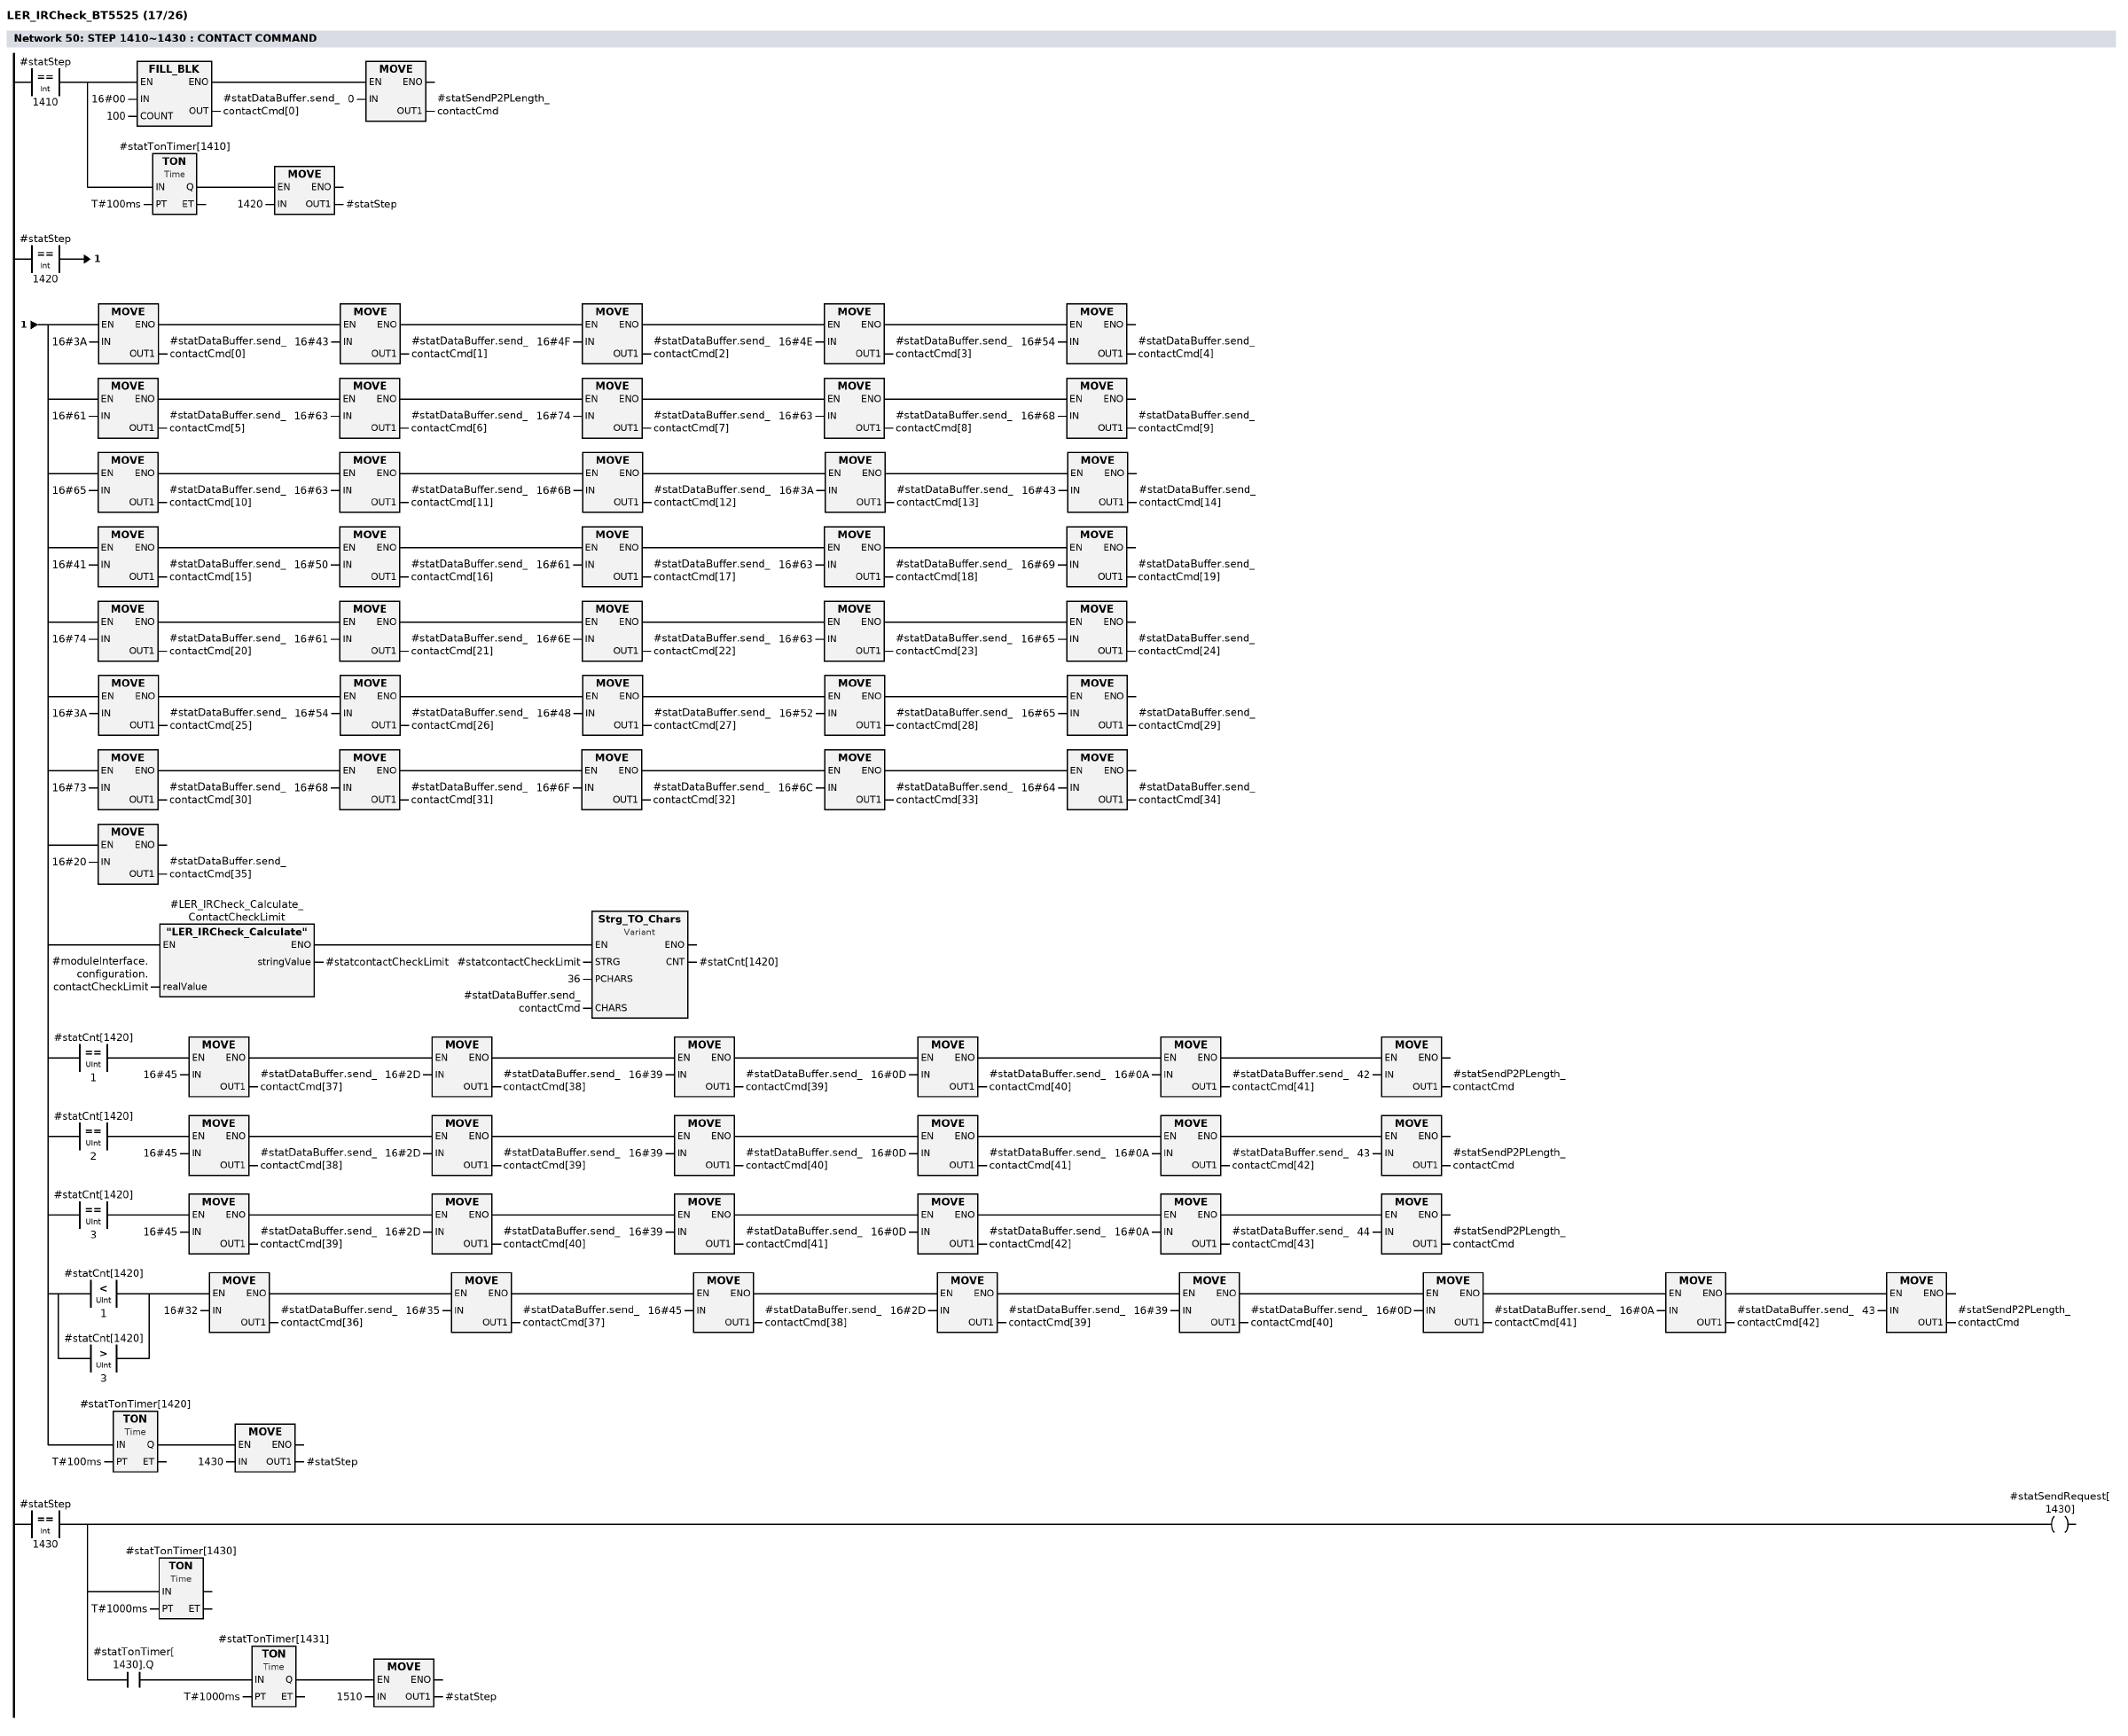
   RUNG wire#powerrail
      { S7_Templates := "SrcType := Int" } EQ_Contact(in1 := #statStep, in2 := 1410)
      wire#w1
      FillBlockI(in := 16#00, count := 100, out => #statDataBuffer.send_contactCmd[0])
      Move(in := 0, out1 => #statSendP2PLength_contactCmd)
   END_RUNG
   RUNG wire#w1
      { S7_Templates := "time_type := Time" } #statTonTimer[1410].TON(pt := T#100ms, et =>)
      Move(in := 1420, out1 => #statStep)
   END_RUNG
   RUNG wire#powerrail
      { S7_Templates := "SrcType := Int" } EQ_Contact(in1 := #statStep, in2 := 1420)
      wire#w2
      Move(in := 16#3A, out1 => #statDataBuffer.send_contactCmd[0])
      Move(in := 16#43, out1 => #statDataBuffer.send_contactCmd[1])
      Move(in := 16#4F, out1 => #statDataBuffer.send_contactCmd[2])
      Move(in := 16#4E, out1 => #statDataBuffer.send_contactCmd[3])
      Move(in := 16#54, out1 => #statDataBuffer.send_contactCmd[4])
   END_RUNG
   RUNG wire#w2
      Move(in := 16#61, out1 => #statDataBuffer.send_contactCmd[5])
      Move(in := 16#63, out1 => #statDataBuffer.send_contactCmd[6])
      Move(in := 16#74, out1 => #statDataBuffer.send_contactCmd[7])
      Move(in := 16#63, out1 => #statDataBuffer.send_contactCmd[8])
      Move(in := 16#68, out1 => #statDataBuffer.send_contactCmd[9])
   END_RUNG
   RUNG wire#w2
      Move(in := 16#65, out1 => #statDataBuffer.send_contactCmd[10])
      Move(in := 16#63, out1 => #statDataBuffer.send_contactCmd[11])
      Move(in := 16#6B, out1 => #statDataBuffer.send_contactCmd[12])
      Move(in := 16#3A, out1 => #statDataBuffer.send_contactCmd[13])
      Move(in := 16#43, out1 => #statDataBuffer.send_contactCmd[14])
   END_RUNG
   RUNG wire#w2
      Move(in := 16#41, out1 => #statDataBuffer.send_contactCmd[15])
      Move(in := 16#50, out1 => #statDataBuffer.send_contactCmd[16])
      Move(in := 16#61, out1 => #statDataBuffer.send_contactCmd[17])
      Move(in := 16#63, out1 => #statDataBuffer.send_contactCmd[18])
      Move(in := 16#69, out1 => #statDataBuffer.send_contactCmd[19])
   END_RUNG
   RUNG wire#w2
      Move(in := 16#74, out1 => #statDataBuffer.send_contactCmd[20])
      Move(in := 16#61, out1 => #statDataBuffer.send_contactCmd[21])
      Move(in := 16#6E, out1 => #statDataBuffer.send_contactCmd[22])
      Move(in := 16#63, out1 => #statDataBuffer.send_contactCmd[23])
      Move(in := 16#65, out1 => #statDataBuffer.send_contactCmd[24])
   END_RUNG
   RUNG wire#w2
      Move(in := 16#3A, out1 => #statDataBuffer.send_contactCmd[25])
      Move(in := 16#54, out1 => #statDataBuffer.send_contactCmd[26])
      Move(in := 16#48, out1 => #statDataBuffer.send_contactCmd[27])
      Move(in := 16#52, out1 => #statDataBuffer.send_contactCmd[28])
      Move(in := 16#65, out1 => #statDataBuffer.send_contactCmd[29])
   END_RUNG
   RUNG wire#w2
      Move(in := 16#73, out1 => #statDataBuffer.send_contactCmd[30])
      Move(in := 16#68, out1 => #statDataBuffer.send_contactCmd[31])
      Move(in := 16#6F, out1 => #statDataBuffer.send_contactCmd[32])
      Move(in := 16#6C, out1 => #statDataBuffer.send_contactCmd[33])
      Move(in := 16#64, out1 => #statDataBuffer.send_contactCmd[34])
   END_RUNG
   RUNG wire#w2
      Move(in := 16#20, out1 => #statDataBuffer.send_contactCmd[35])
   END_RUNG
   RUNG wire#w2
      #LER_IRCheck_Calculate_ContactCheckLimit(realValue := #moduleInterface.configuration.contactCheckLimit, stringValue => #statcontactCheckLimit)
      { S7_Templates := "[ptr_type := Variant, strg_type := String]" } Strg_TO_Chars(Strg := #statcontactCheckLimit, pChars := 36, Chars := #statDataBuffer.send_contactCmd, Cnt => #statCnt[1420])
   END_RUNG
   RUNG wire#w2
      { S7_Templates := "SrcType := UInt" } EQ_Contact(in1 := #statCnt[1420], in2 := 1)
      Move(in := 16#45, out1 => #statDataBuffer.send_contactCmd[37])
      Move(in := 16#2D, out1 => #statDataBuffer.send_contactCmd[38])
      Move(in := 16#39, out1 => #statDataBuffer.send_contactCmd[39])
      Move(in := 16#0D, out1 => #statDataBuffer.send_contactCmd[40])
      Move(in := 16#0A, out1 => #statDataBuffer.send_contactCmd[41])
      Move(in := 42, out1 => #statSendP2PLength_contactCmd)
   END_RUNG
   RUNG wire#w2
      { S7_Templates := "SrcType := UInt" } EQ_Contact(in1 := #statCnt[1420], in2 := 2)
      Move(in := 16#45, out1 => #statDataBuffer.send_contactCmd[38])
      Move(in := 16#2D, out1 => #statDataBuffer.send_contactCmd[39])
      Move(in := 16#39, out1 => #statDataBuffer.send_contactCmd[40])
      Move(in := 16#0D, out1 => #statDataBuffer.send_contactCmd[41])
      Move(in := 16#0A, out1 => #statDataBuffer.send_contactCmd[42])
      Move(in := 43, out1 => #statSendP2PLength_contactCmd)
   END_RUNG
   RUNG wire#w2
      { S7_Templates := "SrcType := UInt" } EQ_Contact(in1 := #statCnt[1420], in2 := 3)
      Move(in := 16#45, out1 => #statDataBuffer.send_contactCmd[39])
      Move(in := 16#2D, out1 => #statDataBuffer.send_contactCmd[40])
      Move(in := 16#39, out1 => #statDataBuffer.send_contactCmd[41])
      Move(in := 16#0D, out1 => #statDataBuffer.send_contactCmd[42])
      Move(in := 16#0A, out1 => #statDataBuffer.send_contactCmd[43])
      Move(in := 44, out1 => #statSendP2PLength_contactCmd)
   END_RUNG
   RUNG wire#w2
      { S7_Templates := "SrcType := UInt" } LT_Contact(in1 := #statCnt[1420], in2 := 1)
      wire#w3
      Move(in := 16#32, out1 => #statDataBuffer.send_contactCmd[36])
      Move(in := 16#35, out1 => #statDataBuffer.send_contactCmd[37])
      Move(in := 16#45, out1 => #statDataBuffer.send_contactCmd[38])
      Move(in := 16#2D, out1 => #statDataBuffer.send_contactCmd[39])
      Move(in := 16#39, out1 => #statDataBuffer.send_contactCmd[40])
      Move(in := 16#0D, out1 => #statDataBuffer.send_contactCmd[41])
      Move(in := 16#0A, out1 => #statDataBuffer.send_contactCmd[42])
      Move(in := 43, out1 => #statSendP2PLength_contactCmd)
   END_RUNG
   RUNG wire#w2
      { S7_Templates := "SrcType := UInt" } GT_Contact(in1 := #statCnt[1420], in2 := 3)
   END_RUNG wire#w3
   RUNG wire#w2
      { S7_Templates := "time_type := Time" } #statTonTimer[1420].TON(pt := T#100ms, et =>)
      Move(in := 1430, out1 => #statStep)
   END_RUNG
   RUNG wire#powerrail
      { S7_Templates := "SrcType := Int" } EQ_Contact(in1 := #statStep, in2 := 1430)
      wire#w4
      Coil( #statSendRequest[1430] )
   END_RUNG
   RUNG wire#w4
      { S7_Templates := "time_type := Time" } #statTonTimer[1430].TON(pt := T#1000ms, et =>)
   END_RUNG
   RUNG wire#w4
      Contact( #statTonTimer[1430].Q )
      { S7_Templates := "time_type := Time" } #statTonTimer[1431].TON(pt := T#1000ms, et =>)
      Move(in := 1510, out1 => #statStep)
   END_RUNG
   // the same network as SCL:
   #_w1 := #statStep = 1410;
   IF #_w1 THEN
       FILL_BLK(IN := 16#00, COUNT := 100, OUT => #statDataBuffer.send_contactCmd[0]);
       #statSendP2PLength_contactCmd := 0;
   END_IF;
   #statTonTimer[1410].TON(IN := #_w1, PT := T#100ms);
   IF #statTonTimer[1410].Q THEN #statStep := 1420; END_IF;
   #_w2 := #statStep = 1420;
   IF #_w2 THEN
       #statDataBuffer.send_contactCmd[0] := 16#3A;
       #statDataBuffer.send_contactCmd[1] := 16#43;
       #statDataBuffer.send_contactCmd[2] := 16#4F;
       #statDataBuffer.send_contactCmd[3] := 16#4E;
       #statDataBuffer.send_contactCmd[4] := 16#54;
       #statDataBuffer.send_contactCmd[5] := 16#61;
       #statDataBuffer.send_contactCmd[6] := 16#63;
       #statDataBuffer.send_contactCmd[7] := 16#74;
       #statDataBuffer.send_contactCmd[8] := 16#63;
       #statDataBuffer.send_contactCmd[9] := 16#68;
       #statDataBuffer.send_contactCmd[10] := 16#65;
       #statDataBuffer.send_contactCmd[11] := 16#63;
       #statDataBuffer.send_contactCmd[12] := 16#6B;
       #statDataBuffer.send_contactCmd[13] := 16#3A;
       #statDataBuffer.send_contactCmd[14] := 16#43;
       #statDataBuffer.send_contactCmd[15] := 16#41;
       #statDataBuffer.send_contactCmd[16] := 16#50;
       #statDataBuffer.send_contactCmd[17] := 16#61;
       #statDataBuffer.send_contactCmd[18] := 16#63;
       #statDataBuffer.send_contactCmd[19] := 16#69;
       #statDataBuffer.send_contactCmd[20] := 16#74;
       #statDataBuffer.send_contactCmd[21] := 16#61;
       #statDataBuffer.send_contactCmd[22] := 16#6E;
       #statDataBuffer.send_contactCmd[23] := 16#63;
       #statDataBuffer.send_contactCmd[24] := 16#65;
       #statDataBuffer.send_contactCmd[25] := 16#3A;
       #statDataBuffer.send_contactCmd[26] := 16#54;
       #statDataBuffer.send_contactCmd[27] := 16#48;
       #statDataBuffer.send_contactCmd[28] := 16#52;
       #statDataBuffer.send_contactCmd[29] := 16#65;
       #statDataBuffer.send_contactCmd[30] := 16#73;
       #statDataBuffer.send_contactCmd[31] := 16#68;
       #statDataBuffer.send_contactCmd[32] := 16#6F;
       #statDataBuffer.send_contactCmd[33] := 16#6C;
       #statDataBuffer.send_contactCmd[34] := 16#64;
       #statDataBuffer.send_contactCmd[35] := 16#20;
   END_IF;
   #LER_IRCheck_Calculate_ContactCheckLimit(EN := #_w2,   // "LER_IRCheck_Calculate"
                           realValue := #moduleInterface.configuration.contactCheckLimit,
                           stringValue => #statcontactCheckLimit,
                           ENO => #_w3);
   IF #_w3 THEN
       Strg_TO_Chars(Strg := #statcontactCheckLimit,
                     pChars := 36,
                     Chars := #statDataBuffer.send_contactCmd,
                     Cnt => #statCnt[1420]);
   END_IF;
   IF #_w2 AND (#statCnt[1420] = 1) THEN
       #statDataBuffer.send_contactCmd[37] := 16#45;
       #statDataBuffer.send_contactCmd[38] := 16#2D;
       #statDataBuffer.send_contactCmd[39] := 16#39;
       #statDataBuffer.send_contactCmd[40] := 16#0D;
       #statDataBuffer.send_contactCmd[41] := 16#0A;
       #statSendP2PLength_contactCmd := 42;
   END_IF;
   IF #_w2 AND (#statCnt[1420] = 2) THEN
       #statDataBuffer.send_contactCmd[38] := 16#45;
       #statDataBuffer.send_contactCmd[39] := 16#2D;
       #statDataBuffer.send_contactCmd[40] := 16#39;
       #statDataBuffer.send_contactCmd[41] := 16#0D;
       #statDataBuffer.send_contactCmd[42] := 16#0A;
       #statSendP2PLength_contactCmd := 43;
   END_IF;
   IF #_w2 AND (#statCnt[1420] = 3) THEN
       #statDataBuffer.send_contactCmd[39] := 16#45;
       #statDataBuffer.send_contactCmd[40] := 16#2D;
       #statDataBuffer.send_contactCmd[41] := 16#39;
       #statDataBuffer.send_contactCmd[42] := 16#0D;
       #statDataBuffer.send_contactCmd[43] := 16#0A;
       #statSendP2PLength_contactCmd := 44;
   END_IF;
   IF #_w2 AND ((#statCnt[1420] < 1) OR (#statCnt[1420] > 3)) THEN
       #statDataBuffer.send_contactCmd[36] := 16#32;
       #statDataBuffer.send_contactCmd[37] := 16#35;
       #statDataBuffer.send_contactCmd[38] := 16#45;
       #statDataBuffer.send_contactCmd[39] := 16#2D;
       #statDataBuffer.send_contactCmd[40] := 16#39;
       #statDataBuffer.send_contactCmd[41] := 16#0D;
       #statDataBuffer.send_contactCmd[42] := 16#0A;
       #statSendP2PLength_contactCmd := 43;
   END_IF;
   #statTonTimer[1420].TON(IN := #_w2, PT := T#100ms);
   IF #statTonTimer[1420].Q THEN #statStep := 1430; END_IF;
   #statSendRequest[1430] := #statStep = 1430;
   #statTonTimer[1430].TON(IN := #statStep = 1430, PT := T#1000ms);
   #statTonTimer[1431].TON(IN := (#statStep = 1430) AND #statTonTimer[1430].Q, PT := T#1000ms);
   IF #statTonTimer[1431].Q THEN #statStep := 1510; END_IF;
END_REGION

REGION Network 51: STEP 1510~1540 : CONTACT CHECK
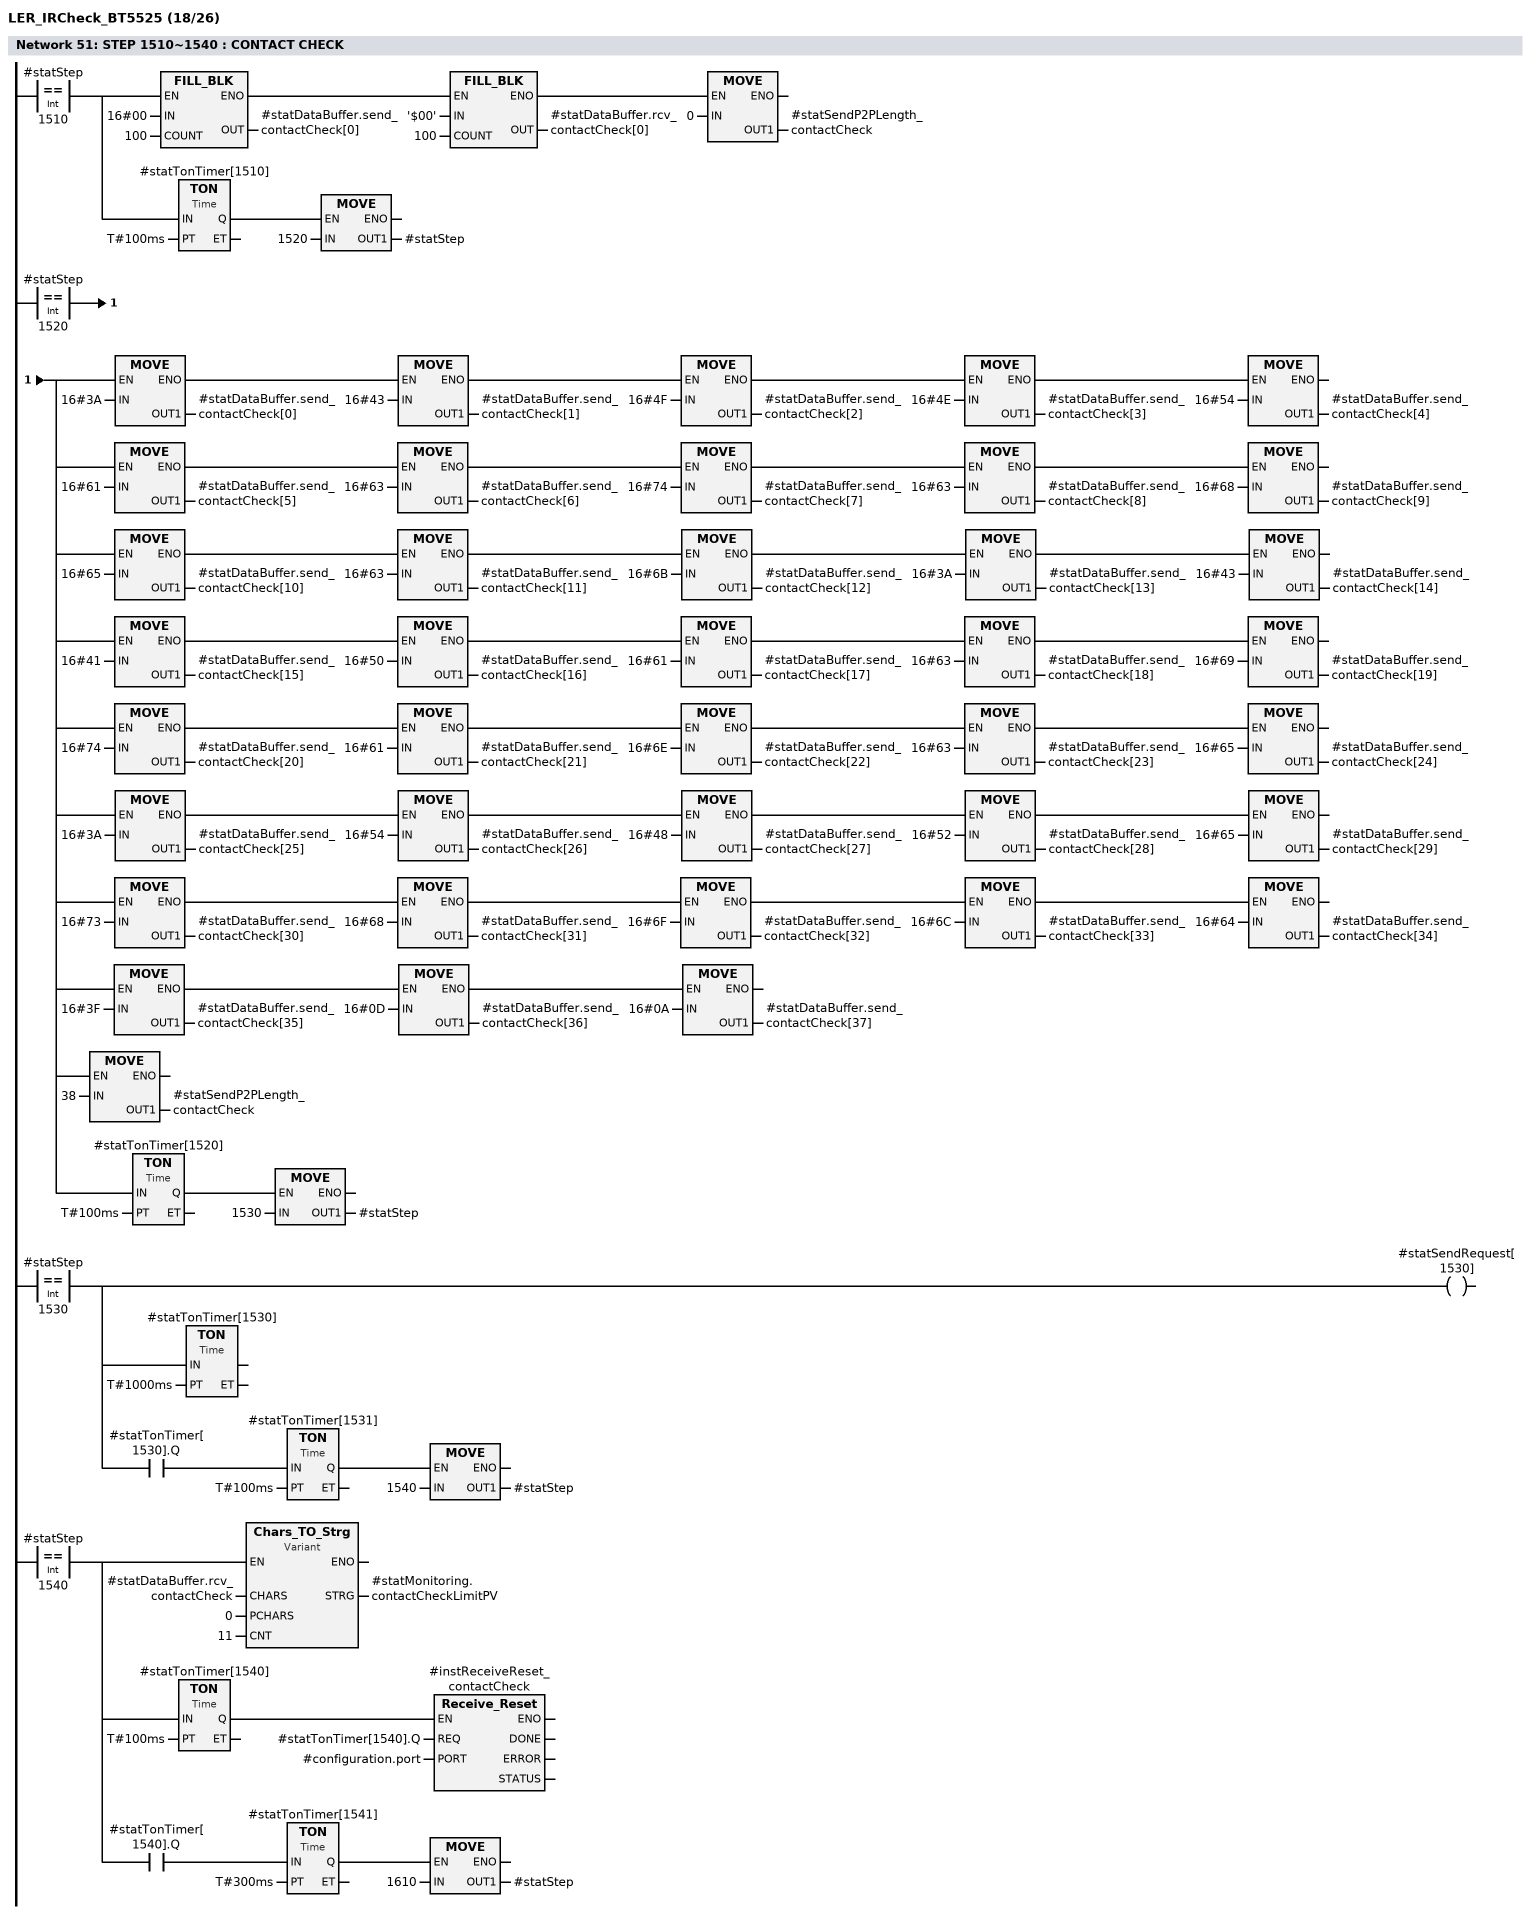
   RUNG wire#powerrail
      { S7_Templates := "SrcType := Int" } EQ_Contact(in1 := #statStep, in2 := 1510)
      wire#w1
      FillBlockI(in := 16#00, count := 100, out => #statDataBuffer.send_contactCheck[0])
      FillBlockI(in := '$00', count := 100, out => #statDataBuffer.rcv_contactCheck[0])
      Move(in := 0, out1 => #statSendP2PLength_contactCheck)
   END_RUNG
   RUNG wire#w1
      { S7_Templates := "time_type := Time" } #statTonTimer[1510].TON(pt := T#100ms, et =>)
      Move(in := 1520, out1 => #statStep)
   END_RUNG
   RUNG wire#powerrail
      { S7_Templates := "SrcType := Int" } EQ_Contact(in1 := #statStep, in2 := 1520)
      wire#w2
      Move(in := 16#3A, out1 => #statDataBuffer.send_contactCheck[0])
      Move(in := 16#43, out1 => #statDataBuffer.send_contactCheck[1])
      Move(in := 16#4F, out1 => #statDataBuffer.send_contactCheck[2])
      Move(in := 16#4E, out1 => #statDataBuffer.send_contactCheck[3])
      Move(in := 16#54, out1 => #statDataBuffer.send_contactCheck[4])
   END_RUNG
   RUNG wire#w2
      Move(in := 16#61, out1 => #statDataBuffer.send_contactCheck[5])
      Move(in := 16#63, out1 => #statDataBuffer.send_contactCheck[6])
      Move(in := 16#74, out1 => #statDataBuffer.send_contactCheck[7])
      Move(in := 16#63, out1 => #statDataBuffer.send_contactCheck[8])
      Move(in := 16#68, out1 => #statDataBuffer.send_contactCheck[9])
   END_RUNG
   RUNG wire#w2
      Move(in := 16#65, out1 => #statDataBuffer.send_contactCheck[10])
      Move(in := 16#63, out1 => #statDataBuffer.send_contactCheck[11])
      Move(in := 16#6B, out1 => #statDataBuffer.send_contactCheck[12])
      Move(in := 16#3A, out1 => #statDataBuffer.send_contactCheck[13])
      Move(in := 16#43, out1 => #statDataBuffer.send_contactCheck[14])
   END_RUNG
   RUNG wire#w2
      Move(in := 16#41, out1 => #statDataBuffer.send_contactCheck[15])
      Move(in := 16#50, out1 => #statDataBuffer.send_contactCheck[16])
      Move(in := 16#61, out1 => #statDataBuffer.send_contactCheck[17])
      Move(in := 16#63, out1 => #statDataBuffer.send_contactCheck[18])
      Move(in := 16#69, out1 => #statDataBuffer.send_contactCheck[19])
   END_RUNG
   RUNG wire#w2
      Move(in := 16#74, out1 => #statDataBuffer.send_contactCheck[20])
      Move(in := 16#61, out1 => #statDataBuffer.send_contactCheck[21])
      Move(in := 16#6E, out1 => #statDataBuffer.send_contactCheck[22])
      Move(in := 16#63, out1 => #statDataBuffer.send_contactCheck[23])
      Move(in := 16#65, out1 => #statDataBuffer.send_contactCheck[24])
   END_RUNG
   RUNG wire#w2
      Move(in := 16#3A, out1 => #statDataBuffer.send_contactCheck[25])
      Move(in := 16#54, out1 => #statDataBuffer.send_contactCheck[26])
      Move(in := 16#48, out1 => #statDataBuffer.send_contactCheck[27])
      Move(in := 16#52, out1 => #statDataBuffer.send_contactCheck[28])
      Move(in := 16#65, out1 => #statDataBuffer.send_contactCheck[29])
   END_RUNG
   RUNG wire#w2
      Move(in := 16#73, out1 => #statDataBuffer.send_contactCheck[30])
      Move(in := 16#68, out1 => #statDataBuffer.send_contactCheck[31])
      Move(in := 16#6F, out1 => #statDataBuffer.send_contactCheck[32])
      Move(in := 16#6C, out1 => #statDataBuffer.send_contactCheck[33])
      Move(in := 16#64, out1 => #statDataBuffer.send_contactCheck[34])
   END_RUNG
   RUNG wire#w2
      Move(in := 16#3F, out1 => #statDataBuffer.send_contactCheck[35])
      Move(in := 16#0D, out1 => #statDataBuffer.send_contactCheck[36])
      Move(in := 16#0A, out1 => #statDataBuffer.send_contactCheck[37])
   END_RUNG
   RUNG wire#w2
      Move(in := 38, out1 => #statSendP2PLength_contactCheck)
   END_RUNG
   RUNG wire#w2
      { S7_Templates := "time_type := Time" } #statTonTimer[1520].TON(pt := T#100ms, et =>)
      Move(in := 1530, out1 => #statStep)
   END_RUNG
   RUNG wire#powerrail
      { S7_Templates := "SrcType := Int" } EQ_Contact(in1 := #statStep, in2 := 1530)
      wire#w3
      Coil( #statSendRequest[1530] )
   END_RUNG
   RUNG wire#w3
      { S7_Templates := "time_type := Time" } #statTonTimer[1530].TON(pt := T#1000ms, et =>)
   END_RUNG
   RUNG wire#w3
      Contact( #statTonTimer[1530].Q )
      { S7_Templates := "time_type := Time" } #statTonTimer[1531].TON(pt := T#100ms, et =>)
      Move(in := 1540, out1 => #statStep)
   END_RUNG
   RUNG wire#powerrail
      { S7_Templates := "SrcType := Int" } EQ_Contact(in1 := #statStep, in2 := 1540)
      wire#w4
      { S7_Templates := "[ptr_type := Variant, str_type := String]" } Chars_TO_Strg(Chars := #statDataBuffer.rcv_contactCheck, pChars := 0, Cnt := 11, Strg => #statMonitoring.contactCheckLimitPV)
   END_RUNG
   RUNG wire#w4
      { S7_Templates := "time_type := Time" } #statTonTimer[1540].TON(pt := T#100ms, et =>)
      #instReceiveReset_contactCheck.Receive_Reset(REQ := #statTonTimer[1540].Q, PORT := #configuration.port, DONE =>, ERROR =>, STATUS =>)
   END_RUNG
   RUNG wire#w4
      Contact( #statTonTimer[1540].Q )
      { S7_Templates := "time_type := Time" } #statTonTimer[1541].TON(pt := T#300ms, et =>)
      Move(in := 1610, out1 => #statStep)
   END_RUNG
   // the same network as SCL:
   #_w1 := #statStep = 1510;
   IF #_w1 THEN
       FILL_BLK(IN := 16#00, COUNT := 100, OUT => #statDataBuffer.send_contactCheck[0]);
       FILL_BLK(IN := '$00', COUNT := 100, OUT => #statDataBuffer.rcv_contactCheck[0]);
       #statSendP2PLength_contactCheck := 0;
   END_IF;
   #statTonTimer[1510].TON(IN := #_w1, PT := T#100ms);
   IF #statTonTimer[1510].Q THEN #statStep := 1520; END_IF;
   #_w2 := #statStep = 1520;
   IF #_w2 THEN
       #statDataBuffer.send_contactCheck[0] := 16#3A;
       #statDataBuffer.send_contactCheck[1] := 16#43;
       #statDataBuffer.send_contactCheck[2] := 16#4F;
       #statDataBuffer.send_contactCheck[3] := 16#4E;
       #statDataBuffer.send_contactCheck[4] := 16#54;
       #statDataBuffer.send_contactCheck[5] := 16#61;
       #statDataBuffer.send_contactCheck[6] := 16#63;
       #statDataBuffer.send_contactCheck[7] := 16#74;
       #statDataBuffer.send_contactCheck[8] := 16#63;
       #statDataBuffer.send_contactCheck[9] := 16#68;
       #statDataBuffer.send_contactCheck[10] := 16#65;
       #statDataBuffer.send_contactCheck[11] := 16#63;
       #statDataBuffer.send_contactCheck[12] := 16#6B;
       #statDataBuffer.send_contactCheck[13] := 16#3A;
       #statDataBuffer.send_contactCheck[14] := 16#43;
       #statDataBuffer.send_contactCheck[15] := 16#41;
       #statDataBuffer.send_contactCheck[16] := 16#50;
       #statDataBuffer.send_contactCheck[17] := 16#61;
       #statDataBuffer.send_contactCheck[18] := 16#63;
       #statDataBuffer.send_contactCheck[19] := 16#69;
       #statDataBuffer.send_contactCheck[20] := 16#74;
       #statDataBuffer.send_contactCheck[21] := 16#61;
       #statDataBuffer.send_contactCheck[22] := 16#6E;
       #statDataBuffer.send_contactCheck[23] := 16#63;
       #statDataBuffer.send_contactCheck[24] := 16#65;
       #statDataBuffer.send_contactCheck[25] := 16#3A;
       #statDataBuffer.send_contactCheck[26] := 16#54;
       #statDataBuffer.send_contactCheck[27] := 16#48;
       #statDataBuffer.send_contactCheck[28] := 16#52;
       #statDataBuffer.send_contactCheck[29] := 16#65;
       #statDataBuffer.send_contactCheck[30] := 16#73;
       #statDataBuffer.send_contactCheck[31] := 16#68;
       #statDataBuffer.send_contactCheck[32] := 16#6F;
       #statDataBuffer.send_contactCheck[33] := 16#6C;
       #statDataBuffer.send_contactCheck[34] := 16#64;
       #statDataBuffer.send_contactCheck[35] := 16#3F;
       #statDataBuffer.send_contactCheck[36] := 16#0D;
       #statDataBuffer.send_contactCheck[37] := 16#0A;
       #statSendP2PLength_contactCheck := 38;
   END_IF;
   #statTonTimer[1520].TON(IN := #_w2, PT := T#100ms);
   IF #statTonTimer[1520].Q THEN #statStep := 1530; END_IF;
   #statSendRequest[1530] := #statStep = 1530;
   #statTonTimer[1530].TON(IN := #statStep = 1530, PT := T#1000ms);
   #statTonTimer[1531].TON(IN := (#statStep = 1530) AND #statTonTimer[1530].Q, PT := T#100ms);
   IF #statTonTimer[1531].Q THEN #statStep := 1540; END_IF;
   #_w3 := #statStep = 1540;
   IF #_w3 THEN
       Chars_TO_Strg(Chars := #statDataBuffer.rcv_contactCheck,
                     pChars := 0,
                     Cnt := 11,
                     Strg => #statMonitoring.contactCheckLimitPV);
   END_IF;
   #statTonTimer[1540].TON(IN := #_w3, PT := T#100ms);
   IF #statTonTimer[1540].Q THEN
       #instReceiveReset_contactCheck(REQ := #statTonTimer[1540].Q, PORT := #configuration.port);   // Receive_Reset
   END_IF;
   #statTonTimer[1541].TON(IN := #_w3 AND #statTonTimer[1540].Q, PT := T#300ms);
   IF #statTonTimer[1541].Q THEN #statStep := 1610; END_IF;
END_REGION

REGION Network 52: STEP 1610~1630 : COMPARATOR COMMAND
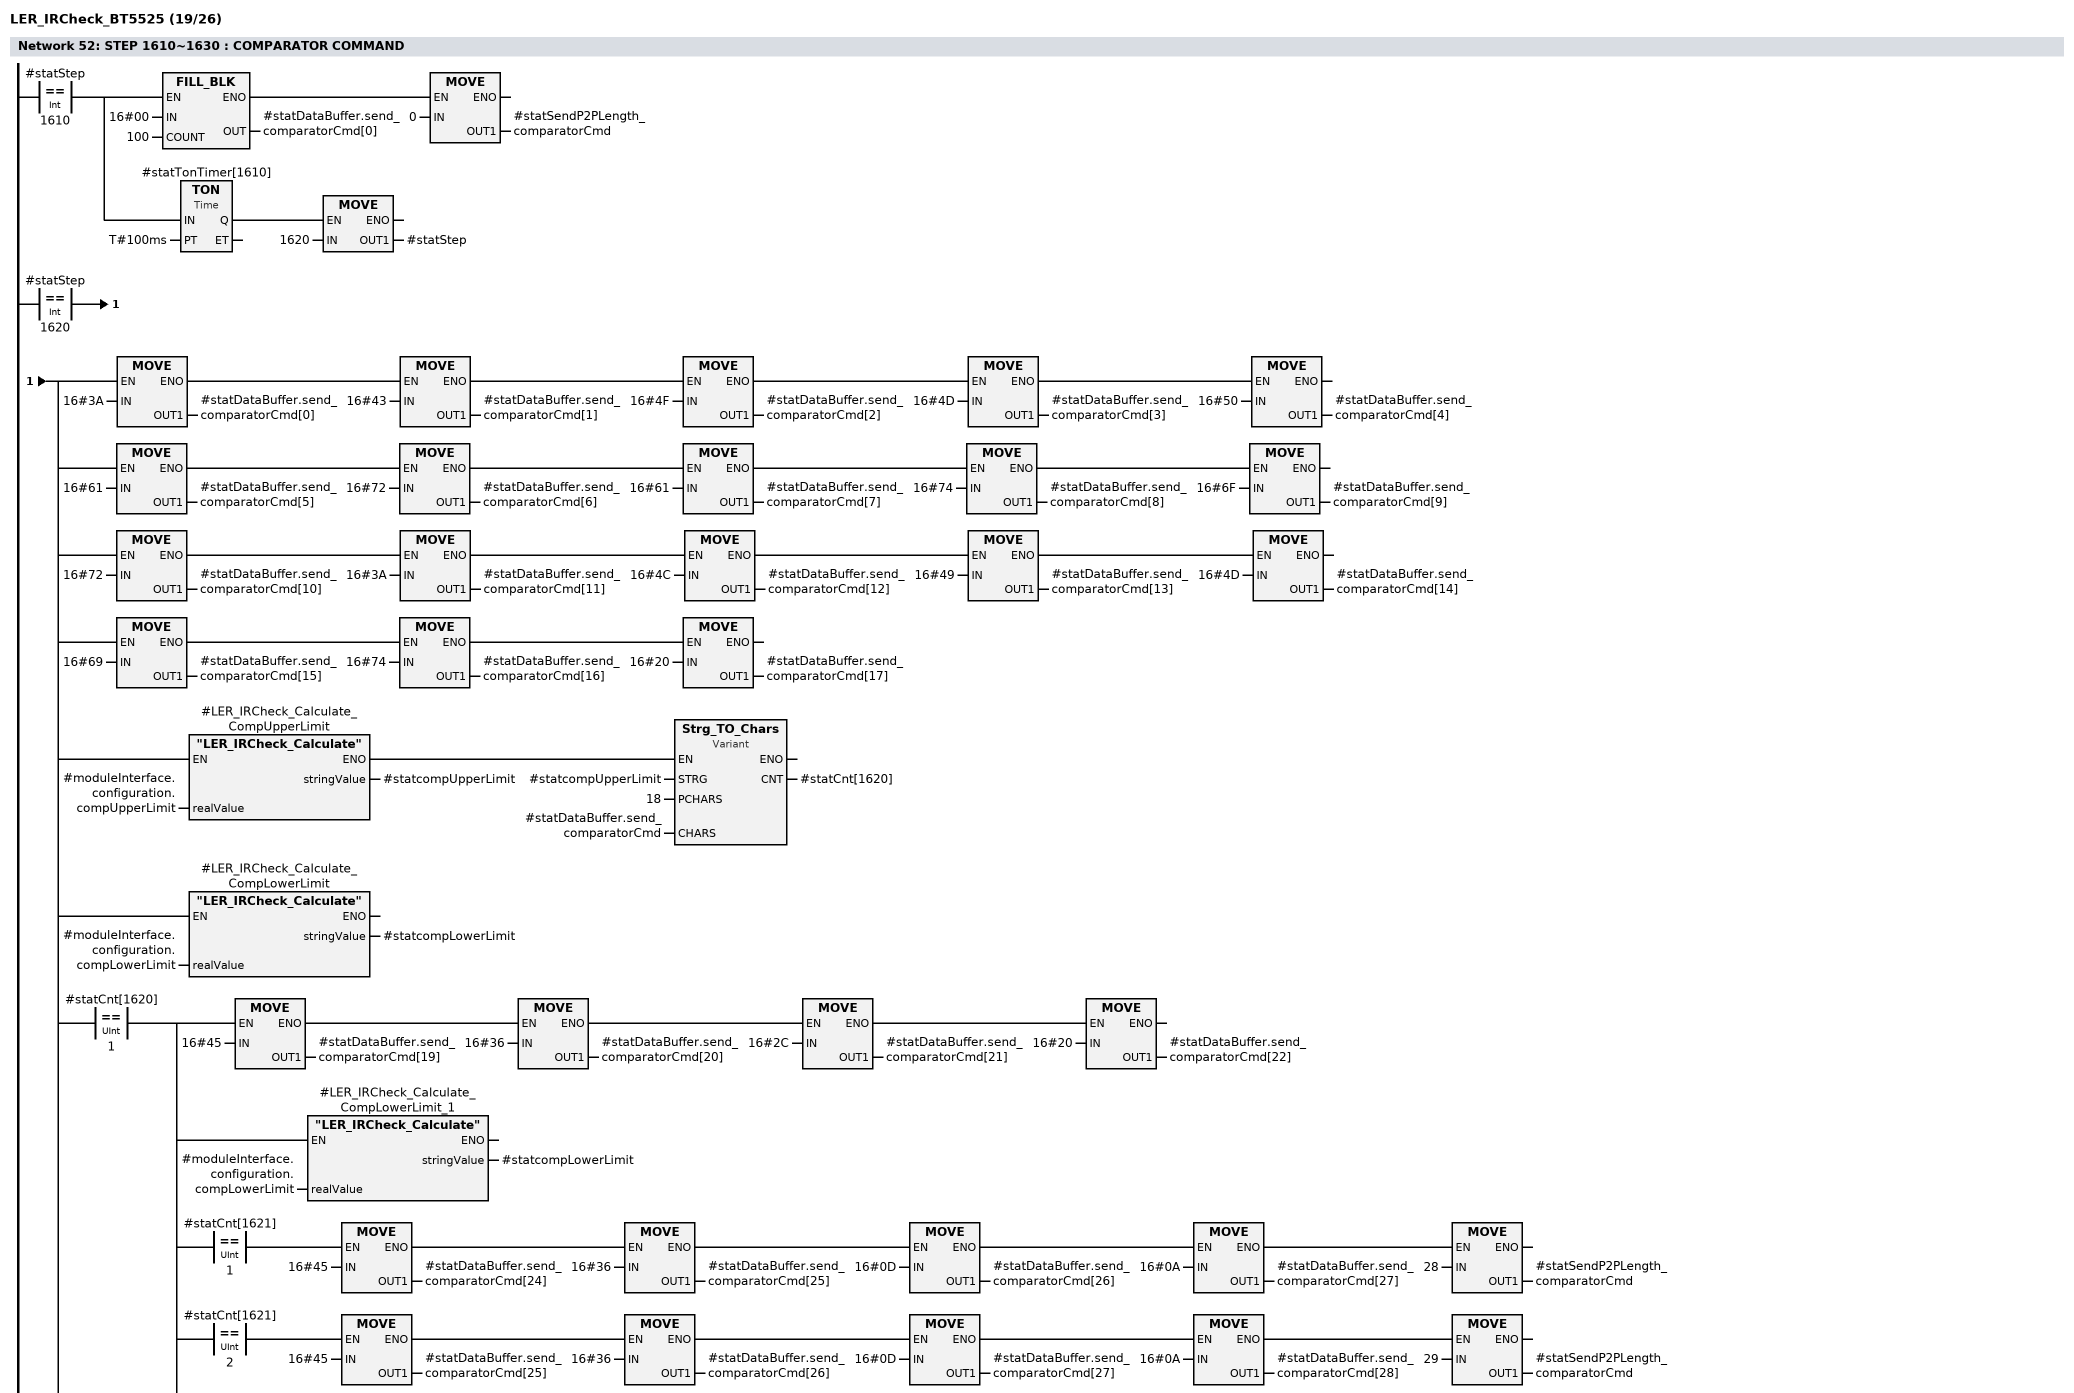
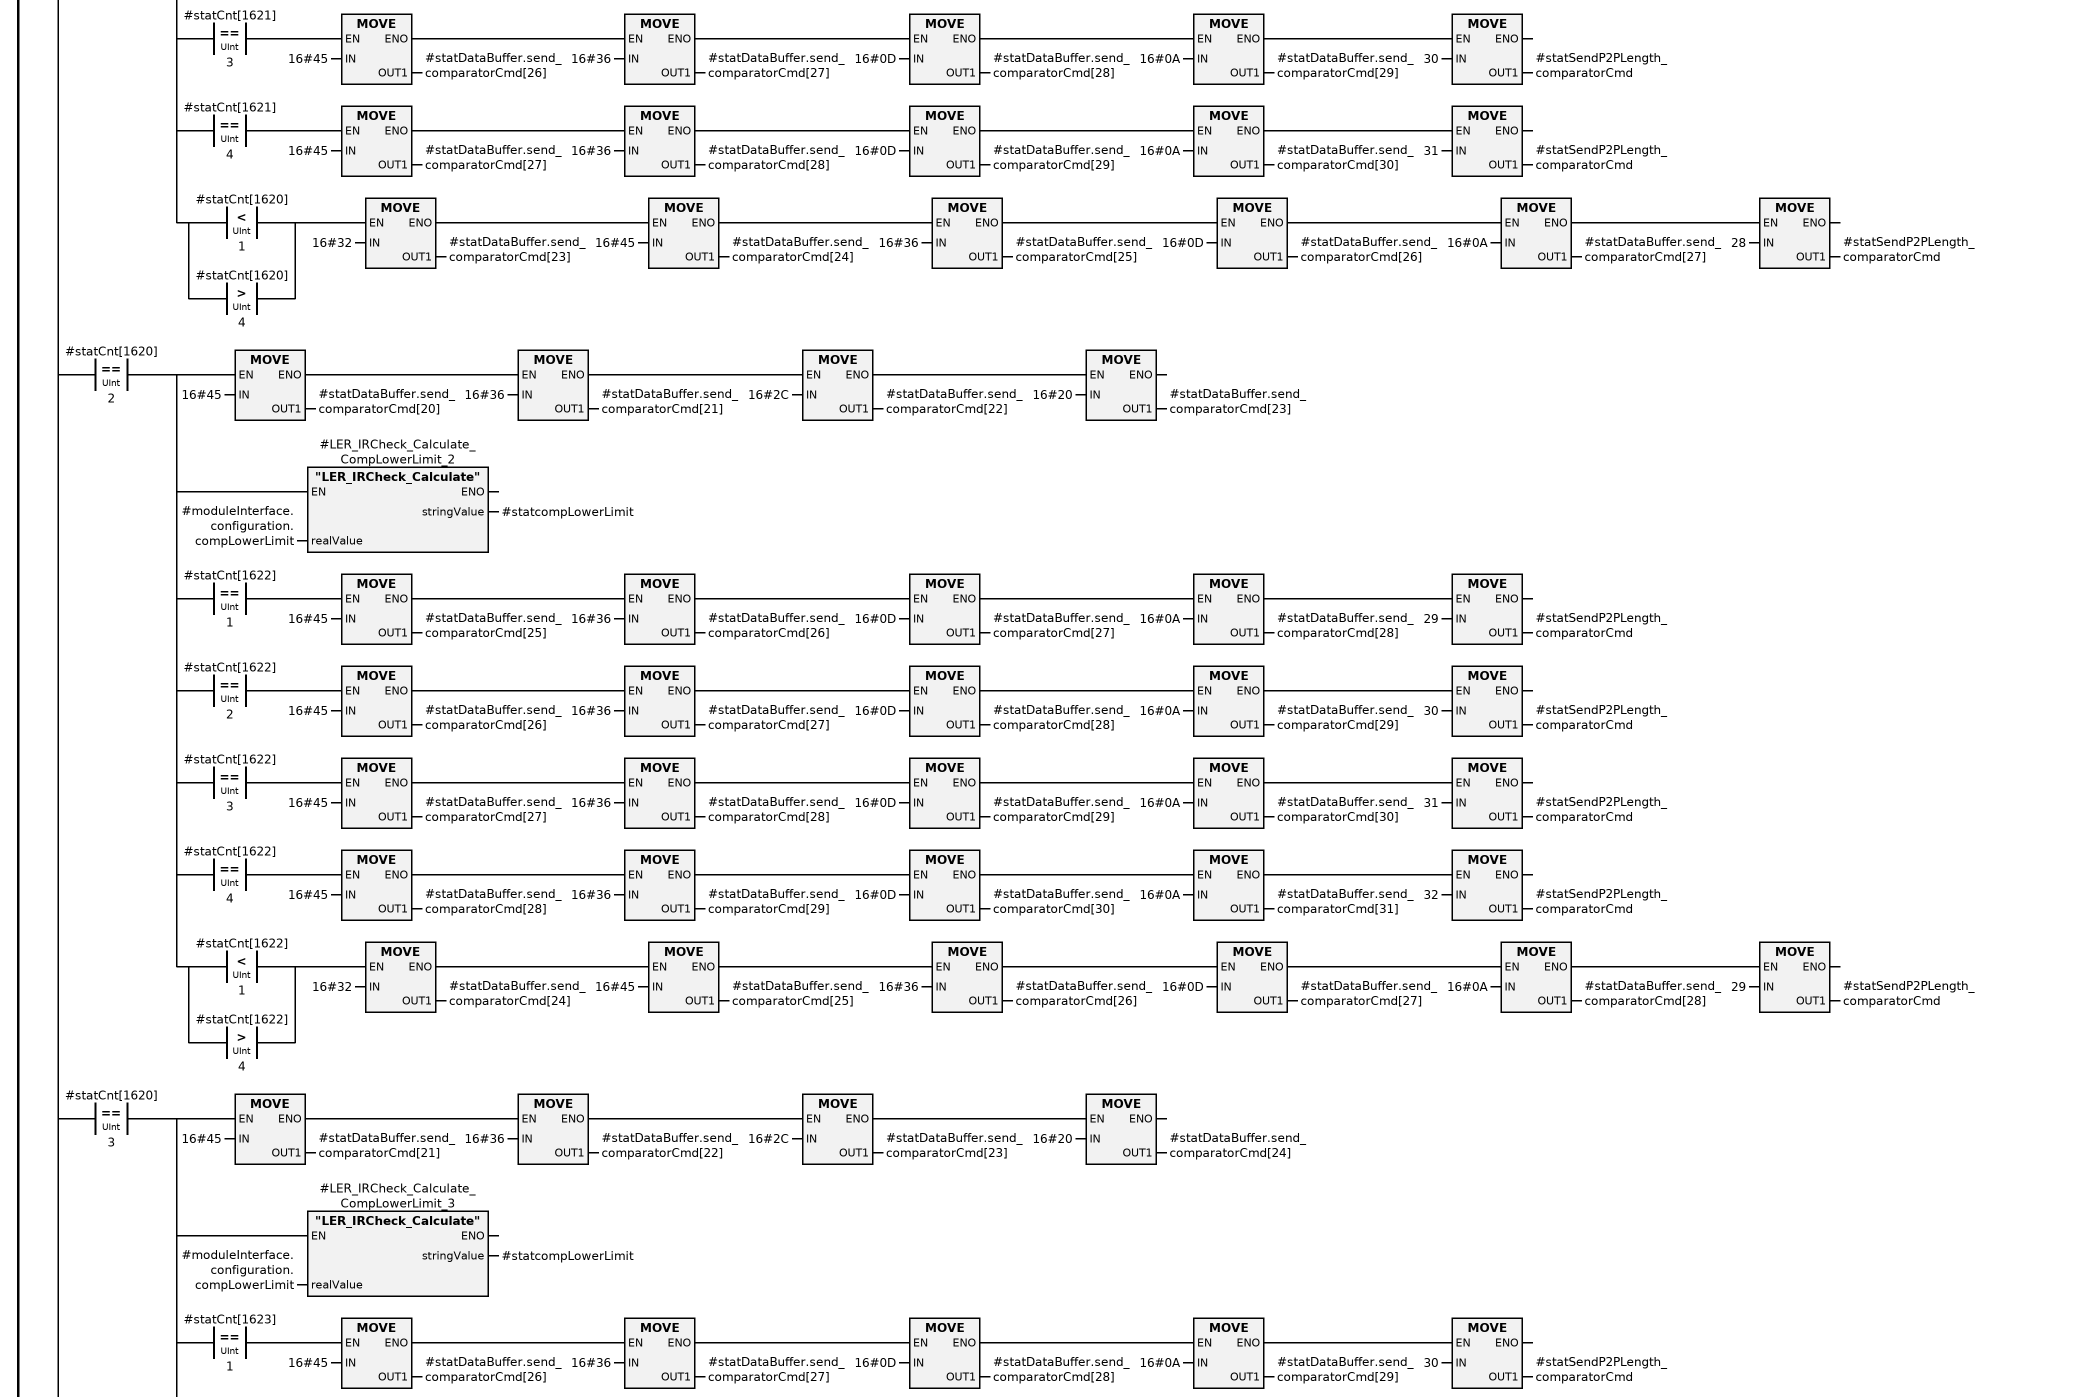
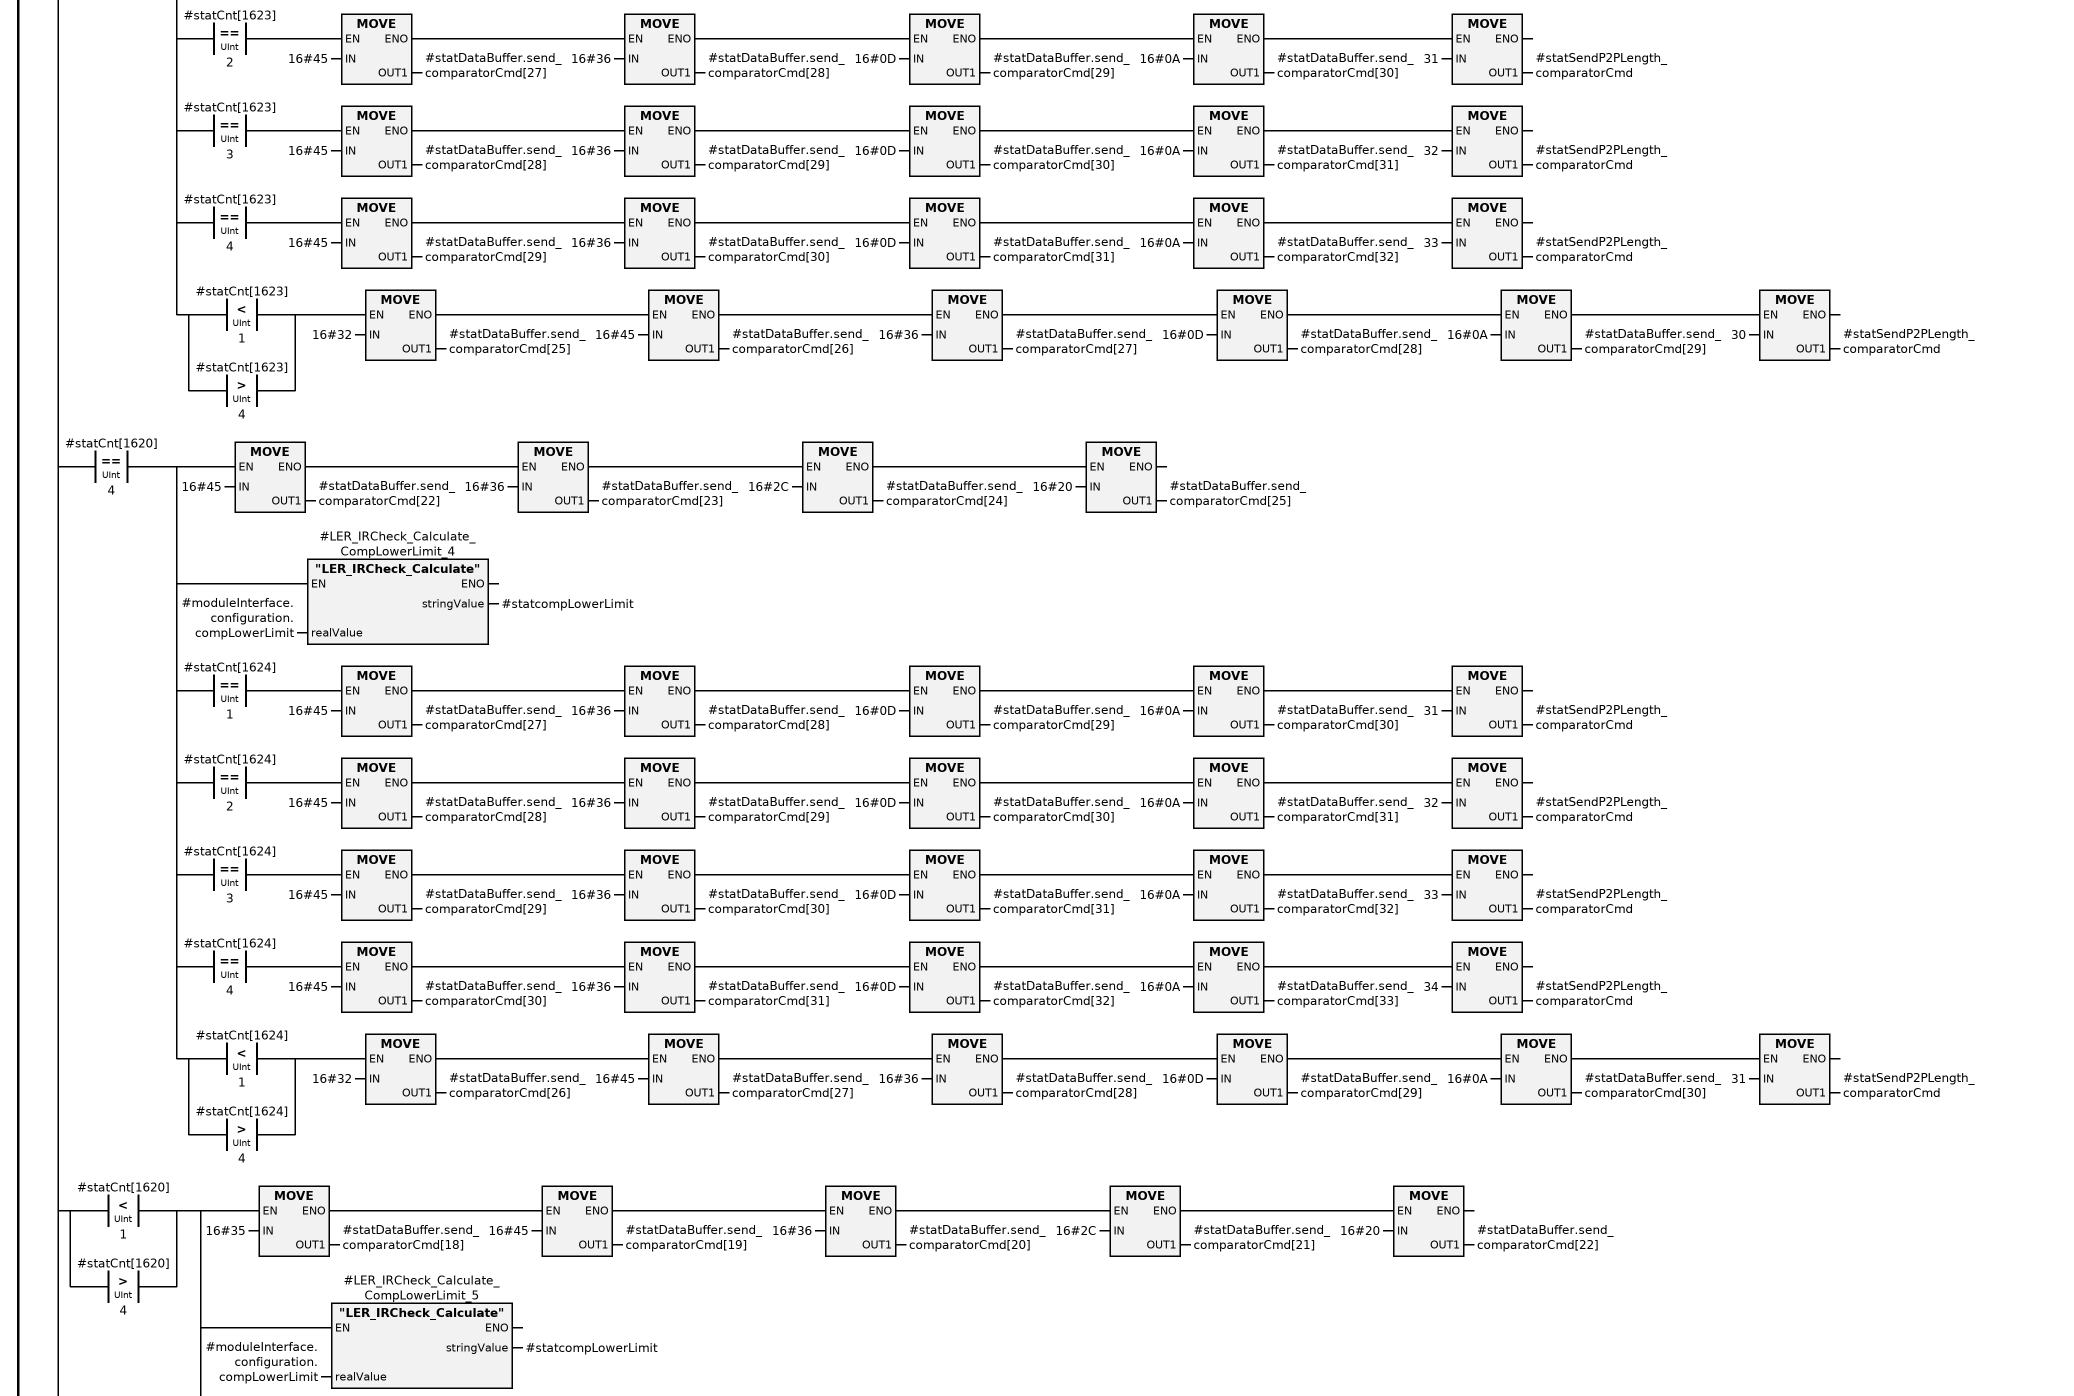
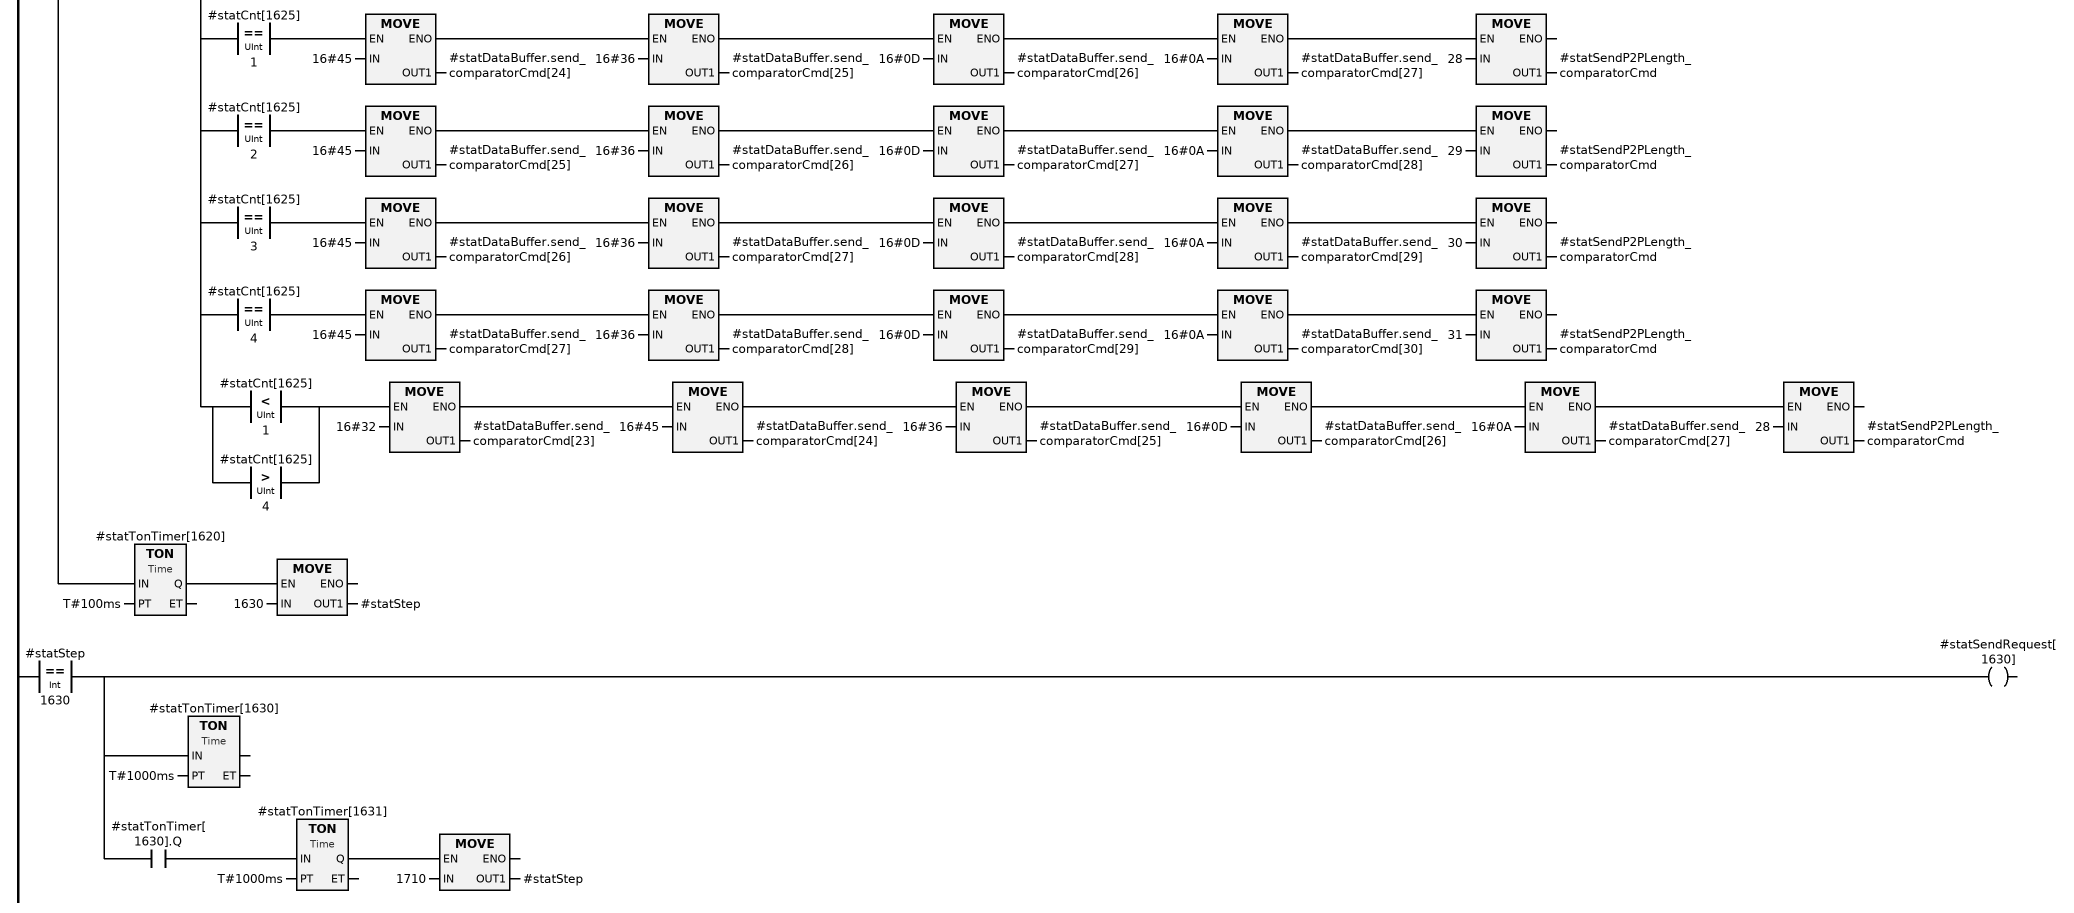
   RUNG wire#powerrail
      { S7_Templates := "SrcType := Int" } EQ_Contact(in1 := #statStep, in2 := 1610)
      wire#w1
      FillBlockI(in := 16#00, count := 100, out => #statDataBuffer.send_comparatorCmd[0])
      Move(in := 0, out1 => #statSendP2PLength_comparatorCmd)
   END_RUNG
   RUNG wire#w1
      { S7_Templates := "time_type := Time" } #statTonTimer[1610].TON(pt := T#100ms, et =>)
      Move(in := 1620, out1 => #statStep)
   END_RUNG
   RUNG wire#powerrail
      { S7_Templates := "SrcType := Int" } EQ_Contact(in1 := #statStep, in2 := 1620)
      wire#w2
      Move(in := 16#3A, out1 => #statDataBuffer.send_comparatorCmd[0])
      Move(in := 16#43, out1 => #statDataBuffer.send_comparatorCmd[1])
      Move(in := 16#4F, out1 => #statDataBuffer.send_comparatorCmd[2])
      Move(in := 16#4D, out1 => #statDataBuffer.send_comparatorCmd[3])
      Move(in := 16#50, out1 => #statDataBuffer.send_comparatorCmd[4])
   END_RUNG
   RUNG wire#w2
      Move(in := 16#61, out1 => #statDataBuffer.send_comparatorCmd[5])
      Move(in := 16#72, out1 => #statDataBuffer.send_comparatorCmd[6])
      Move(in := 16#61, out1 => #statDataBuffer.send_comparatorCmd[7])
      Move(in := 16#74, out1 => #statDataBuffer.send_comparatorCmd[8])
      Move(in := 16#6F, out1 => #statDataBuffer.send_comparatorCmd[9])
   END_RUNG
   RUNG wire#w2
      Move(in := 16#72, out1 => #statDataBuffer.send_comparatorCmd[10])
      Move(in := 16#3A, out1 => #statDataBuffer.send_comparatorCmd[11])
      Move(in := 16#4C, out1 => #statDataBuffer.send_comparatorCmd[12])
      Move(in := 16#49, out1 => #statDataBuffer.send_comparatorCmd[13])
      Move(in := 16#4D, out1 => #statDataBuffer.send_comparatorCmd[14])
   END_RUNG
   RUNG wire#w2
      Move(in := 16#69, out1 => #statDataBuffer.send_comparatorCmd[15])
      Move(in := 16#74, out1 => #statDataBuffer.send_comparatorCmd[16])
      Move(in := 16#20, out1 => #statDataBuffer.send_comparatorCmd[17])
   END_RUNG
   RUNG wire#w2
      #LER_IRCheck_Calculate_CompUpperLimit(realValue := #moduleInterface.configuration.compUpperLimit, stringValue => #statcompUpperLimit)
      { S7_Templates := "[ptr_type := Variant, strg_type := String]" } Strg_TO_Chars(Strg := #statcompUpperLimit, pChars := 18, Chars := #statDataBuffer.send_comparatorCmd, Cnt => #statCnt[1620])
   END_RUNG
   RUNG wire#w2
      #LER_IRCheck_Calculate_CompLowerLimit(realValue := #moduleInterface.configuration.compLowerLimit, stringValue => #statcompLowerLimit)
   END_RUNG
   RUNG wire#w2
      { S7_Templates := "SrcType := UInt" } EQ_Contact(in1 := #statCnt[1620], in2 := 1)
      wire#w3
      Move(in := 16#45, out1 => #statDataBuffer.send_comparatorCmd[19])
      Move(in := 16#36, out1 => #statDataBuffer.send_comparatorCmd[20])
      Move(in := 16#2C, out1 => #statDataBuffer.send_comparatorCmd[21])
      Move(in := 16#20, out1 => #statDataBuffer.send_comparatorCmd[22])
   END_RUNG
   RUNG wire#w3
      #LER_IRCheck_Calculate_CompLowerLimit_1(realValue := #moduleInterface.configuration.compLowerLimit, stringValue => #statcompLowerLimit)
   END_RUNG
   RUNG wire#w3
      { S7_Templates := "SrcType := UInt" } EQ_Contact(in1 := #statCnt[1621], in2 := 1)
      Move(in := 16#45, out1 => #statDataBuffer.send_comparatorCmd[24])
      Move(in := 16#36, out1 => #statDataBuffer.send_comparatorCmd[25])
      Move(in := 16#0D, out1 => #statDataBuffer.send_comparatorCmd[26])
      Move(in := 16#0A, out1 => #statDataBuffer.send_comparatorCmd[27])
      Move(in := 28, out1 => #statSendP2PLength_comparatorCmd)
   END_RUNG
   RUNG wire#w3
      { S7_Templates := "SrcType := UInt" } EQ_Contact(in1 := #statCnt[1621], in2 := 2)
      Move(in := 16#45, out1 => #statDataBuffer.send_comparatorCmd[25])
      Move(in := 16#36, out1 => #statDataBuffer.send_comparatorCmd[26])
      Move(in := 16#0D, out1 => #statDataBuffer.send_comparatorCmd[27])
      Move(in := 16#0A, out1 => #statDataBuffer.send_comparatorCmd[28])
      Move(in := 29, out1 => #statSendP2PLength_comparatorCmd)
   END_RUNG
   RUNG wire#w3
      { S7_Templates := "SrcType := UInt" } EQ_Contact(in1 := #statCnt[1621], in2 := 3)
      Move(in := 16#45, out1 => #statDataBuffer.send_comparatorCmd[26])
      Move(in := 16#36, out1 => #statDataBuffer.send_comparatorCmd[27])
      Move(in := 16#0D, out1 => #statDataBuffer.send_comparatorCmd[28])
      Move(in := 16#0A, out1 => #statDataBuffer.send_comparatorCmd[29])
      Move(in := 30, out1 => #statSendP2PLength_comparatorCmd)
   END_RUNG
   RUNG wire#w3
      { S7_Templates := "SrcType := UInt" } EQ_Contact(in1 := #statCnt[1621], in2 := 4)
      Move(in := 16#45, out1 => #statDataBuffer.send_comparatorCmd[27])
      Move(in := 16#36, out1 => #statDataBuffer.send_comparatorCmd[28])
      Move(in := 16#0D, out1 => #statDataBuffer.send_comparatorCmd[29])
      Move(in := 16#0A, out1 => #statDataBuffer.send_comparatorCmd[30])
      Move(in := 31, out1 => #statSendP2PLength_comparatorCmd)
   END_RUNG
   RUNG wire#w3
      { S7_Templates := "SrcType := UInt" } LT_Contact(in1 := #statCnt[1620], in2 := 1)
      wire#w4
      Move(in := 16#32, out1 => #statDataBuffer.send_comparatorCmd[23])
      Move(in := 16#45, out1 => #statDataBuffer.send_comparatorCmd[24])
      Move(in := 16#36, out1 => #statDataBuffer.send_comparatorCmd[25])
      Move(in := 16#0D, out1 => #statDataBuffer.send_comparatorCmd[26])
      Move(in := 16#0A, out1 => #statDataBuffer.send_comparatorCmd[27])
      Move(in := 28, out1 => #statSendP2PLength_comparatorCmd)
   END_RUNG
   RUNG wire#w3
      { S7_Templates := "SrcType := UInt" } GT_Contact(in1 := #statCnt[1620], in2 := 4)
   END_RUNG wire#w4
   RUNG wire#w2
      { S7_Templates := "SrcType := UInt" } EQ_Contact(in1 := #statCnt[1620], in2 := 2)
      wire#w5
      Move(in := 16#45, out1 => #statDataBuffer.send_comparatorCmd[20])
      Move(in := 16#36, out1 => #statDataBuffer.send_comparatorCmd[21])
      Move(in := 16#2C, out1 => #statDataBuffer.send_comparatorCmd[22])
      Move(in := 16#20, out1 => #statDataBuffer.send_comparatorCmd[23])
   END_RUNG
   RUNG wire#w5
      #LER_IRCheck_Calculate_CompLowerLimit_2(realValue := #moduleInterface.configuration.compLowerLimit, stringValue => #statcompLowerLimit)
   END_RUNG
   RUNG wire#w5
      { S7_Templates := "SrcType := UInt" } EQ_Contact(in1 := #statCnt[1622], in2 := 1)
      Move(in := 16#45, out1 => #statDataBuffer.send_comparatorCmd[25])
      Move(in := 16#36, out1 => #statDataBuffer.send_comparatorCmd[26])
      Move(in := 16#0D, out1 => #statDataBuffer.send_comparatorCmd[27])
      Move(in := 16#0A, out1 => #statDataBuffer.send_comparatorCmd[28])
      Move(in := 29, out1 => #statSendP2PLength_comparatorCmd)
   END_RUNG
   RUNG wire#w5
      { S7_Templates := "SrcType := UInt" } EQ_Contact(in1 := #statCnt[1622], in2 := 2)
      Move(in := 16#45, out1 => #statDataBuffer.send_comparatorCmd[26])
      Move(in := 16#36, out1 => #statDataBuffer.send_comparatorCmd[27])
      Move(in := 16#0D, out1 => #statDataBuffer.send_comparatorCmd[28])
      Move(in := 16#0A, out1 => #statDataBuffer.send_comparatorCmd[29])
      Move(in := 30, out1 => #statSendP2PLength_comparatorCmd)
   END_RUNG
   RUNG wire#w5
      { S7_Templates := "SrcType := UInt" } EQ_Contact(in1 := #statCnt[1622], in2 := 3)
      Move(in := 16#45, out1 => #statDataBuffer.send_comparatorCmd[27])
      Move(in := 16#36, out1 => #statDataBuffer.send_comparatorCmd[28])
      Move(in := 16#0D, out1 => #statDataBuffer.send_comparatorCmd[29])
      Move(in := 16#0A, out1 => #statDataBuffer.send_comparatorCmd[30])
      Move(in := 31, out1 => #statSendP2PLength_comparatorCmd)
   END_RUNG
   RUNG wire#w5
      { S7_Templates := "SrcType := UInt" } EQ_Contact(in1 := #statCnt[1622], in2 := 4)
      Move(in := 16#45, out1 => #statDataBuffer.send_comparatorCmd[28])
      Move(in := 16#36, out1 => #statDataBuffer.send_comparatorCmd[29])
      Move(in := 16#0D, out1 => #statDataBuffer.send_comparatorCmd[30])
      Move(in := 16#0A, out1 => #statDataBuffer.send_comparatorCmd[31])
      Move(in := 32, out1 => #statSendP2PLength_comparatorCmd)
   END_RUNG
   RUNG wire#w5
      { S7_Templates := "SrcType := UInt" } LT_Contact(in1 := #statCnt[1622], in2 := 1)
      wire#w6
      Move(in := 16#32, out1 => #statDataBuffer.send_comparatorCmd[24])
      Move(in := 16#45, out1 => #statDataBuffer.send_comparatorCmd[25])
      Move(in := 16#36, out1 => #statDataBuffer.send_comparatorCmd[26])
      Move(in := 16#0D, out1 => #statDataBuffer.send_comparatorCmd[27])
      Move(in := 16#0A, out1 => #statDataBuffer.send_comparatorCmd[28])
      Move(in := 29, out1 => #statSendP2PLength_comparatorCmd)
   END_RUNG
   RUNG wire#w5
      { S7_Templates := "SrcType := UInt" } GT_Contact(in1 := #statCnt[1622], in2 := 4)
   END_RUNG wire#w6
   RUNG wire#w2
      { S7_Templates := "SrcType := UInt" } EQ_Contact(in1 := #statCnt[1620], in2 := 3)
      wire#w7
      Move(in := 16#45, out1 => #statDataBuffer.send_comparatorCmd[21])
      Move(in := 16#36, out1 => #statDataBuffer.send_comparatorCmd[22])
      Move(in := 16#2C, out1 => #statDataBuffer.send_comparatorCmd[23])
      Move(in := 16#20, out1 => #statDataBuffer.send_comparatorCmd[24])
   END_RUNG
   RUNG wire#w7
      #LER_IRCheck_Calculate_CompLowerLimit_3(realValue := #moduleInterface.configuration.compLowerLimit, stringValue => #statcompLowerLimit)
   END_RUNG
   RUNG wire#w7
      { S7_Templates := "SrcType := UInt" } EQ_Contact(in1 := #statCnt[1623], in2 := 1)
      Move(in := 16#45, out1 => #statDataBuffer.send_comparatorCmd[26])
      Move(in := 16#36, out1 => #statDataBuffer.send_comparatorCmd[27])
      Move(in := 16#0D, out1 => #statDataBuffer.send_comparatorCmd[28])
      Move(in := 16#0A, out1 => #statDataBuffer.send_comparatorCmd[29])
      Move(in := 30, out1 => #statSendP2PLength_comparatorCmd)
   END_RUNG
   RUNG wire#w7
      { S7_Templates := "SrcType := UInt" } EQ_Contact(in1 := #statCnt[1623], in2 := 2)
      Move(in := 16#45, out1 => #statDataBuffer.send_comparatorCmd[27])
      Move(in := 16#36, out1 => #statDataBuffer.send_comparatorCmd[28])
      Move(in := 16#0D, out1 => #statDataBuffer.send_comparatorCmd[29])
      Move(in := 16#0A, out1 => #statDataBuffer.send_comparatorCmd[30])
      Move(in := 31, out1 => #statSendP2PLength_comparatorCmd)
   END_RUNG
   RUNG wire#w7
      { S7_Templates := "SrcType := UInt" } EQ_Contact(in1 := #statCnt[1623], in2 := 3)
      Move(in := 16#45, out1 => #statDataBuffer.send_comparatorCmd[28])
      Move(in := 16#36, out1 => #statDataBuffer.send_comparatorCmd[29])
      Move(in := 16#0D, out1 => #statDataBuffer.send_comparatorCmd[30])
      Move(in := 16#0A, out1 => #statDataBuffer.send_comparatorCmd[31])
      Move(in := 32, out1 => #statSendP2PLength_comparatorCmd)
   END_RUNG
   RUNG wire#w7
      { S7_Templates := "SrcType := UInt" } EQ_Contact(in1 := #statCnt[1623], in2 := 4)
      Move(in := 16#45, out1 => #statDataBuffer.send_comparatorCmd[29])
      Move(in := 16#36, out1 => #statDataBuffer.send_comparatorCmd[30])
      Move(in := 16#0D, out1 => #statDataBuffer.send_comparatorCmd[31])
      Move(in := 16#0A, out1 => #statDataBuffer.send_comparatorCmd[32])
      Move(in := 33, out1 => #statSendP2PLength_comparatorCmd)
   END_RUNG
   RUNG wire#w7
      { S7_Templates := "SrcType := UInt" } LT_Contact(in1 := #statCnt[1623], in2 := 1)
      wire#w8
      Move(in := 16#32, out1 => #statDataBuffer.send_comparatorCmd[25])
      Move(in := 16#45, out1 => #statDataBuffer.send_comparatorCmd[26])
      Move(in := 16#36, out1 => #statDataBuffer.send_comparatorCmd[27])
      Move(in := 16#0D, out1 => #statDataBuffer.send_comparatorCmd[28])
      Move(in := 16#0A, out1 => #statDataBuffer.send_comparatorCmd[29])
      Move(in := 30, out1 => #statSendP2PLength_comparatorCmd)
   END_RUNG
   RUNG wire#w7
      { S7_Templates := "SrcType := UInt" } GT_Contact(in1 := #statCnt[1623], in2 := 4)
   END_RUNG wire#w8
   RUNG wire#w2
      { S7_Templates := "SrcType := UInt" } EQ_Contact(in1 := #statCnt[1620], in2 := 4)
      wire#w9
      Move(in := 16#45, out1 => #statDataBuffer.send_comparatorCmd[22])
      Move(in := 16#36, out1 => #statDataBuffer.send_comparatorCmd[23])
      Move(in := 16#2C, out1 => #statDataBuffer.send_comparatorCmd[24])
      Move(in := 16#20, out1 => #statDataBuffer.send_comparatorCmd[25])
   END_RUNG
   RUNG wire#w9
      #LER_IRCheck_Calculate_CompLowerLimit_4(realValue := #moduleInterface.configuration.compLowerLimit, stringValue => #statcompLowerLimit)
   END_RUNG
   RUNG wire#w9
      { S7_Templates := "SrcType := UInt" } EQ_Contact(in1 := #statCnt[1624], in2 := 1)
      Move(in := 16#45, out1 => #statDataBuffer.send_comparatorCmd[27])
      Move(in := 16#36, out1 => #statDataBuffer.send_comparatorCmd[28])
      Move(in := 16#0D, out1 => #statDataBuffer.send_comparatorCmd[29])
      Move(in := 16#0A, out1 => #statDataBuffer.send_comparatorCmd[30])
      Move(in := 31, out1 => #statSendP2PLength_comparatorCmd)
   END_RUNG
   RUNG wire#w9
      { S7_Templates := "SrcType := UInt" } EQ_Contact(in1 := #statCnt[1624], in2 := 2)
      Move(in := 16#45, out1 => #statDataBuffer.send_comparatorCmd[28])
      Move(in := 16#36, out1 => #statDataBuffer.send_comparatorCmd[29])
      Move(in := 16#0D, out1 => #statDataBuffer.send_comparatorCmd[30])
      Move(in := 16#0A, out1 => #statDataBuffer.send_comparatorCmd[31])
      Move(in := 32, out1 => #statSendP2PLength_comparatorCmd)
   END_RUNG
   RUNG wire#w9
      { S7_Templates := "SrcType := UInt" } EQ_Contact(in1 := #statCnt[1624], in2 := 3)
      Move(in := 16#45, out1 => #statDataBuffer.send_comparatorCmd[29])
      Move(in := 16#36, out1 => #statDataBuffer.send_comparatorCmd[30])
      Move(in := 16#0D, out1 => #statDataBuffer.send_comparatorCmd[31])
      Move(in := 16#0A, out1 => #statDataBuffer.send_comparatorCmd[32])
      Move(in := 33, out1 => #statSendP2PLength_comparatorCmd)
   END_RUNG
   RUNG wire#w9
      { S7_Templates := "SrcType := UInt" } EQ_Contact(in1 := #statCnt[1624], in2 := 4)
      Move(in := 16#45, out1 => #statDataBuffer.send_comparatorCmd[30])
      Move(in := 16#36, out1 => #statDataBuffer.send_comparatorCmd[31])
      Move(in := 16#0D, out1 => #statDataBuffer.send_comparatorCmd[32])
      Move(in := 16#0A, out1 => #statDataBuffer.send_comparatorCmd[33])
      Move(in := 34, out1 => #statSendP2PLength_comparatorCmd)
   END_RUNG
   RUNG wire#w9
      { S7_Templates := "SrcType := UInt" } LT_Contact(in1 := #statCnt[1624], in2 := 1)
      wire#w10
      Move(in := 16#32, out1 => #statDataBuffer.send_comparatorCmd[26])
      Move(in := 16#45, out1 => #statDataBuffer.send_comparatorCmd[27])
      Move(in := 16#36, out1 => #statDataBuffer.send_comparatorCmd[28])
      Move(in := 16#0D, out1 => #statDataBuffer.send_comparatorCmd[29])
      Move(in := 16#0A, out1 => #statDataBuffer.send_comparatorCmd[30])
      Move(in := 31, out1 => #statSendP2PLength_comparatorCmd)
   END_RUNG
   RUNG wire#w9
      { S7_Templates := "SrcType := UInt" } GT_Contact(in1 := #statCnt[1624], in2 := 4)
   END_RUNG wire#w10
   RUNG wire#w2
      { S7_Templates := "SrcType := UInt" } LT_Contact(in1 := #statCnt[1620], in2 := 1)
      wire#w11
      Move(in := 16#35, out1 => #statDataBuffer.send_comparatorCmd[18])
      Move(in := 16#45, out1 => #statDataBuffer.send_comparatorCmd[19])
      Move(in := 16#36, out1 => #statDataBuffer.send_comparatorCmd[20])
      Move(in := 16#2C, out1 => #statDataBuffer.send_comparatorCmd[21])
      Move(in := 16#20, out1 => #statDataBuffer.send_comparatorCmd[22])
   END_RUNG
   RUNG wire#w2
      { S7_Templates := "SrcType := UInt" } GT_Contact(in1 := #statCnt[1620], in2 := 4)
   END_RUNG wire#w11
   RUNG wire#w11
      #LER_IRCheck_Calculate_CompLowerLimit_5(realValue := #moduleInterface.configuration.compLowerLimit, stringValue => #statcompLowerLimit)
   END_RUNG
   RUNG wire#w11
      { S7_Templates := "SrcType := UInt" } EQ_Contact(in1 := #statCnt[1625], in2 := 1)
      Move(in := 16#45, out1 => #statDataBuffer.send_comparatorCmd[24])
      Move(in := 16#36, out1 => #statDataBuffer.send_comparatorCmd[25])
      Move(in := 16#0D, out1 => #statDataBuffer.send_comparatorCmd[26])
      Move(in := 16#0A, out1 => #statDataBuffer.send_comparatorCmd[27])
      Move(in := 28, out1 => #statSendP2PLength_comparatorCmd)
   END_RUNG
   RUNG wire#w11
      { S7_Templates := "SrcType := UInt" } EQ_Contact(in1 := #statCnt[1625], in2 := 2)
      Move(in := 16#45, out1 => #statDataBuffer.send_comparatorCmd[25])
      Move(in := 16#36, out1 => #statDataBuffer.send_comparatorCmd[26])
      Move(in := 16#0D, out1 => #statDataBuffer.send_comparatorCmd[27])
      Move(in := 16#0A, out1 => #statDataBuffer.send_comparatorCmd[28])
      Move(in := 29, out1 => #statSendP2PLength_comparatorCmd)
   END_RUNG
   RUNG wire#w11
      { S7_Templates := "SrcType := UInt" } EQ_Contact(in1 := #statCnt[1625], in2 := 3)
      Move(in := 16#45, out1 => #statDataBuffer.send_comparatorCmd[26])
      Move(in := 16#36, out1 => #statDataBuffer.send_comparatorCmd[27])
      Move(in := 16#0D, out1 => #statDataBuffer.send_comparatorCmd[28])
      Move(in := 16#0A, out1 => #statDataBuffer.send_comparatorCmd[29])
      Move(in := 30, out1 => #statSendP2PLength_comparatorCmd)
   END_RUNG
   RUNG wire#w11
      { S7_Templates := "SrcType := UInt" } EQ_Contact(in1 := #statCnt[1625], in2 := 4)
      Move(in := 16#45, out1 => #statDataBuffer.send_comparatorCmd[27])
      Move(in := 16#36, out1 => #statDataBuffer.send_comparatorCmd[28])
      Move(in := 16#0D, out1 => #statDataBuffer.send_comparatorCmd[29])
      Move(in := 16#0A, out1 => #statDataBuffer.send_comparatorCmd[30])
      Move(in := 31, out1 => #statSendP2PLength_comparatorCmd)
   END_RUNG
   RUNG wire#w11
      { S7_Templates := "SrcType := UInt" } LT_Contact(in1 := #statCnt[1625], in2 := 1)
      wire#w12
      Move(in := 16#32, out1 => #statDataBuffer.send_comparatorCmd[23])
      Move(in := 16#45, out1 => #statDataBuffer.send_comparatorCmd[24])
      Move(in := 16#36, out1 => #statDataBuffer.send_comparatorCmd[25])
      Move(in := 16#0D, out1 => #statDataBuffer.send_comparatorCmd[26])
      Move(in := 16#0A, out1 => #statDataBuffer.send_comparatorCmd[27])
      Move(in := 28, out1 => #statSendP2PLength_comparatorCmd)
   END_RUNG
   RUNG wire#w11
      { S7_Templates := "SrcType := UInt" } GT_Contact(in1 := #statCnt[1625], in2 := 4)
   END_RUNG wire#w12
   RUNG wire#w2
      { S7_Templates := "time_type := Time" } #statTonTimer[1620].TON(pt := T#100ms, et =>)
      Move(in := 1630, out1 => #statStep)
   END_RUNG
   RUNG wire#powerrail
      { S7_Templates := "SrcType := Int" } EQ_Contact(in1 := #statStep, in2 := 1630)
      wire#w13
      Coil( #statSendRequest[1630] )
   END_RUNG
   RUNG wire#w13
      { S7_Templates := "time_type := Time" } #statTonTimer[1630].TON(pt := T#1000ms, et =>)
   END_RUNG
   RUNG wire#w13
      Contact( #statTonTimer[1630].Q )
      { S7_Templates := "time_type := Time" } #statTonTimer[1631].TON(pt := T#1000ms, et =>)
      Move(in := 1710, out1 => #statStep)
   END_RUNG
   // the same network as SCL:
   #_w1 := #statStep = 1610;
   IF #_w1 THEN
       FILL_BLK(IN := 16#00, COUNT := 100, OUT => #statDataBuffer.send_comparatorCmd[0]);
       #statSendP2PLength_comparatorCmd := 0;
   END_IF;
   #statTonTimer[1610].TON(IN := #_w1, PT := T#100ms);
   IF #statTonTimer[1610].Q THEN #statStep := 1620; END_IF;
   #_w2 := #statStep = 1620;
   IF #_w2 THEN
       #statDataBuffer.send_comparatorCmd[0] := 16#3A;
       #statDataBuffer.send_comparatorCmd[1] := 16#43;
       #statDataBuffer.send_comparatorCmd[2] := 16#4F;
       #statDataBuffer.send_comparatorCmd[3] := 16#4D;
       #statDataBuffer.send_comparatorCmd[4] := 16#50;
       #statDataBuffer.send_comparatorCmd[5] := 16#61;
       #statDataBuffer.send_comparatorCmd[6] := 16#72;
       #statDataBuffer.send_comparatorCmd[7] := 16#61;
       #statDataBuffer.send_comparatorCmd[8] := 16#74;
       #statDataBuffer.send_comparatorCmd[9] := 16#6F;
       #statDataBuffer.send_comparatorCmd[10] := 16#72;
       #statDataBuffer.send_comparatorCmd[11] := 16#3A;
       #statDataBuffer.send_comparatorCmd[12] := 16#4C;
       #statDataBuffer.send_comparatorCmd[13] := 16#49;
       #statDataBuffer.send_comparatorCmd[14] := 16#4D;
       #statDataBuffer.send_comparatorCmd[15] := 16#69;
       #statDataBuffer.send_comparatorCmd[16] := 16#74;
       #statDataBuffer.send_comparatorCmd[17] := 16#20;
   END_IF;
   #LER_IRCheck_Calculate_CompUpperLimit(EN := #_w2,   // "LER_IRCheck_Calculate"
                           realValue := #moduleInterface.configuration.compUpperLimit,
                           stringValue => #statcompUpperLimit,
                           ENO => #_w3);
   IF #_w3 THEN
       Strg_TO_Chars(Strg := #statcompUpperLimit,
                     pChars := 18,
                     Chars := #statDataBuffer.send_comparatorCmd,
                     Cnt => #statCnt[1620]);
   END_IF;
   IF #_w2 THEN
       #LER_IRCheck_Calculate_CompLowerLimit(realValue := #moduleInterface.configuration.compLowerLimit,   // "LER_IRCheck_Calculate"
                               stringValue => #statcompLowerLimit);
   END_IF;
   #_w4 := #_w2 AND (#statCnt[1620] = 1);
   IF #_w4 THEN
       #statDataBuffer.send_comparatorCmd[19] := 16#45;
       #statDataBuffer.send_comparatorCmd[20] := 16#36;
       #statDataBuffer.send_comparatorCmd[21] := 16#2C;
       #statDataBuffer.send_comparatorCmd[22] := 16#20;
       #LER_IRCheck_Calculate_CompLowerLimit_1(realValue := #moduleInterface.configuration.compLowerLimit,   // "LER_IRCheck_Calculate"
                               stringValue => #statcompLowerLimit);
   END_IF;
   IF #_w4 AND (#statCnt[1621] = 1) THEN
       #statDataBuffer.send_comparatorCmd[24] := 16#45;
       #statDataBuffer.send_comparatorCmd[25] := 16#36;
       #statDataBuffer.send_comparatorCmd[26] := 16#0D;
       #statDataBuffer.send_comparatorCmd[27] := 16#0A;
       #statSendP2PLength_comparatorCmd := 28;
   END_IF;
   IF #_w4 AND (#statCnt[1621] = 2) THEN
       #statDataBuffer.send_comparatorCmd[25] := 16#45;
       #statDataBuffer.send_comparatorCmd[26] := 16#36;
       #statDataBuffer.send_comparatorCmd[27] := 16#0D;
       #statDataBuffer.send_comparatorCmd[28] := 16#0A;
       #statSendP2PLength_comparatorCmd := 29;
   END_IF;
   IF #_w4 AND (#statCnt[1621] = 3) THEN
       #statDataBuffer.send_comparatorCmd[26] := 16#45;
       #statDataBuffer.send_comparatorCmd[27] := 16#36;
       #statDataBuffer.send_comparatorCmd[28] := 16#0D;
       #statDataBuffer.send_comparatorCmd[29] := 16#0A;
       #statSendP2PLength_comparatorCmd := 30;
   END_IF;
   IF #_w4 AND (#statCnt[1621] = 4) THEN
       #statDataBuffer.send_comparatorCmd[27] := 16#45;
       #statDataBuffer.send_comparatorCmd[28] := 16#36;
       #statDataBuffer.send_comparatorCmd[29] := 16#0D;
       #statDataBuffer.send_comparatorCmd[30] := 16#0A;
       #statSendP2PLength_comparatorCmd := 31;
   END_IF;
   IF #_w4 AND ((#statCnt[1620] < 1) OR (#statCnt[1620] > 4)) THEN
       #statDataBuffer.send_comparatorCmd[23] := 16#32;
       #statDataBuffer.send_comparatorCmd[24] := 16#45;
       #statDataBuffer.send_comparatorCmd[25] := 16#36;
       #statDataBuffer.send_comparatorCmd[26] := 16#0D;
       #statDataBuffer.send_comparatorCmd[27] := 16#0A;
       #statSendP2PLength_comparatorCmd := 28;
   END_IF;
   #_w5 := #_w2 AND (#statCnt[1620] = 2);
   IF #_w5 THEN
       #statDataBuffer.send_comparatorCmd[20] := 16#45;
       #statDataBuffer.send_comparatorCmd[21] := 16#36;
       #statDataBuffer.send_comparatorCmd[22] := 16#2C;
       #statDataBuffer.send_comparatorCmd[23] := 16#20;
       #LER_IRCheck_Calculate_CompLowerLimit_2(realValue := #moduleInterface.configuration.compLowerLimit,   // "LER_IRCheck_Calculate"
                               stringValue => #statcompLowerLimit);
   END_IF;
   IF #_w5 AND (#statCnt[1622] = 1) THEN
       #statDataBuffer.send_comparatorCmd[25] := 16#45;
       #statDataBuffer.send_comparatorCmd[26] := 16#36;
       #statDataBuffer.send_comparatorCmd[27] := 16#0D;
       #statDataBuffer.send_comparatorCmd[28] := 16#0A;
       #statSendP2PLength_comparatorCmd := 29;
   END_IF;
   IF #_w5 AND (#statCnt[1622] = 2) THEN
       #statDataBuffer.send_comparatorCmd[26] := 16#45;
       #statDataBuffer.send_comparatorCmd[27] := 16#36;
       #statDataBuffer.send_comparatorCmd[28] := 16#0D;
       #statDataBuffer.send_comparatorCmd[29] := 16#0A;
       #statSendP2PLength_comparatorCmd := 30;
   END_IF;
   IF #_w5 AND (#statCnt[1622] = 3) THEN
       #statDataBuffer.send_comparatorCmd[27] := 16#45;
       #statDataBuffer.send_comparatorCmd[28] := 16#36;
       #statDataBuffer.send_comparatorCmd[29] := 16#0D;
       #statDataBuffer.send_comparatorCmd[30] := 16#0A;
       #statSendP2PLength_comparatorCmd := 31;
   END_IF;
   IF #_w5 AND (#statCnt[1622] = 4) THEN
       #statDataBuffer.send_comparatorCmd[28] := 16#45;
       #statDataBuffer.send_comparatorCmd[29] := 16#36;
       #statDataBuffer.send_comparatorCmd[30] := 16#0D;
       #statDataBuffer.send_comparatorCmd[31] := 16#0A;
       #statSendP2PLength_comparatorCmd := 32;
   END_IF;
   IF #_w5 AND ((#statCnt[1622] < 1) OR (#statCnt[1622] > 4)) THEN
       #statDataBuffer.send_comparatorCmd[24] := 16#32;
       #statDataBuffer.send_comparatorCmd[25] := 16#45;
       #statDataBuffer.send_comparatorCmd[26] := 16#36;
       #statDataBuffer.send_comparatorCmd[27] := 16#0D;
       #statDataBuffer.send_comparatorCmd[28] := 16#0A;
       #statSendP2PLength_comparatorCmd := 29;
   END_IF;
   #_w6 := #_w2 AND (#statCnt[1620] = 3);
   IF #_w6 THEN
       #statDataBuffer.send_comparatorCmd[21] := 16#45;
       #statDataBuffer.send_comparatorCmd[22] := 16#36;
       #statDataBuffer.send_comparatorCmd[23] := 16#2C;
       #statDataBuffer.send_comparatorCmd[24] := 16#20;
       #LER_IRCheck_Calculate_CompLowerLimit_3(realValue := #moduleInterface.configuration.compLowerLimit,   // "LER_IRCheck_Calculate"
                               stringValue => #statcompLowerLimit);
   END_IF;
   IF #_w6 AND (#statCnt[1623] = 1) THEN
       #statDataBuffer.send_comparatorCmd[26] := 16#45;
       #statDataBuffer.send_comparatorCmd[27] := 16#36;
       #statDataBuffer.send_comparatorCmd[28] := 16#0D;
       #statDataBuffer.send_comparatorCmd[29] := 16#0A;
       #statSendP2PLength_comparatorCmd := 30;
   END_IF;
   IF #_w6 AND (#statCnt[1623] = 2) THEN
       #statDataBuffer.send_comparatorCmd[27] := 16#45;
       #statDataBuffer.send_comparatorCmd[28] := 16#36;
       #statDataBuffer.send_comparatorCmd[29] := 16#0D;
       #statDataBuffer.send_comparatorCmd[30] := 16#0A;
       #statSendP2PLength_comparatorCmd := 31;
   END_IF;
   IF #_w6 AND (#statCnt[1623] = 3) THEN
       #statDataBuffer.send_comparatorCmd[28] := 16#45;
       #statDataBuffer.send_comparatorCmd[29] := 16#36;
       #statDataBuffer.send_comparatorCmd[30] := 16#0D;
       #statDataBuffer.send_comparatorCmd[31] := 16#0A;
       #statSendP2PLength_comparatorCmd := 32;
   END_IF;
   IF #_w6 AND (#statCnt[1623] = 4) THEN
       #statDataBuffer.send_comparatorCmd[29] := 16#45;
       #statDataBuffer.send_comparatorCmd[30] := 16#36;
       #statDataBuffer.send_comparatorCmd[31] := 16#0D;
       #statDataBuffer.send_comparatorCmd[32] := 16#0A;
       #statSendP2PLength_comparatorCmd := 33;
   END_IF;
   IF #_w6 AND ((#statCnt[1623] < 1) OR (#statCnt[1623] > 4)) THEN
       #statDataBuffer.send_comparatorCmd[25] := 16#32;
       #statDataBuffer.send_comparatorCmd[26] := 16#45;
       #statDataBuffer.send_comparatorCmd[27] := 16#36;
       #statDataBuffer.send_comparatorCmd[28] := 16#0D;
       #statDataBuffer.send_comparatorCmd[29] := 16#0A;
       #statSendP2PLength_comparatorCmd := 30;
   END_IF;
   #_w7 := #_w2 AND (#statCnt[1620] = 4);
   IF #_w7 THEN
       #statDataBuffer.send_comparatorCmd[22] := 16#45;
       #statDataBuffer.send_comparatorCmd[23] := 16#36;
       #statDataBuffer.send_comparatorCmd[24] := 16#2C;
       #statDataBuffer.send_comparatorCmd[25] := 16#20;
       #LER_IRCheck_Calculate_CompLowerLimit_4(realValue := #moduleInterface.configuration.compLowerLimit,   // "LER_IRCheck_Calculate"
                               stringValue => #statcompLowerLimit);
   END_IF;
   IF #_w7 AND (#statCnt[1624] = 1) THEN
       #statDataBuffer.send_comparatorCmd[27] := 16#45;
       #statDataBuffer.send_comparatorCmd[28] := 16#36;
       #statDataBuffer.send_comparatorCmd[29] := 16#0D;
       #statDataBuffer.send_comparatorCmd[30] := 16#0A;
       #statSendP2PLength_comparatorCmd := 31;
   END_IF;
   IF #_w7 AND (#statCnt[1624] = 2) THEN
       #statDataBuffer.send_comparatorCmd[28] := 16#45;
       #statDataBuffer.send_comparatorCmd[29] := 16#36;
       #statDataBuffer.send_comparatorCmd[30] := 16#0D;
       #statDataBuffer.send_comparatorCmd[31] := 16#0A;
       #statSendP2PLength_comparatorCmd := 32;
   END_IF;
   IF #_w7 AND (#statCnt[1624] = 3) THEN
       #statDataBuffer.send_comparatorCmd[29] := 16#45;
       #statDataBuffer.send_comparatorCmd[30] := 16#36;
       #statDataBuffer.send_comparatorCmd[31] := 16#0D;
       #statDataBuffer.send_comparatorCmd[32] := 16#0A;
       #statSendP2PLength_comparatorCmd := 33;
   END_IF;
   IF #_w7 AND (#statCnt[1624] = 4) THEN
       #statDataBuffer.send_comparatorCmd[30] := 16#45;
       #statDataBuffer.send_comparatorCmd[31] := 16#36;
       #statDataBuffer.send_comparatorCmd[32] := 16#0D;
       #statDataBuffer.send_comparatorCmd[33] := 16#0A;
       #statSendP2PLength_comparatorCmd := 34;
   END_IF;
   IF #_w7 AND ((#statCnt[1624] < 1) OR (#statCnt[1624] > 4)) THEN
       #statDataBuffer.send_comparatorCmd[26] := 16#32;
       #statDataBuffer.send_comparatorCmd[27] := 16#45;
       #statDataBuffer.send_comparatorCmd[28] := 16#36;
       #statDataBuffer.send_comparatorCmd[29] := 16#0D;
       #statDataBuffer.send_comparatorCmd[30] := 16#0A;
       #statSendP2PLength_comparatorCmd := 31;
   END_IF;
   #_w8 := #_w2 AND ((#statCnt[1620] < 1) OR (#statCnt[1620] > 4));
   IF #_w8 THEN
       #statDataBuffer.send_comparatorCmd[18] := 16#35;
       #statDataBuffer.send_comparatorCmd[19] := 16#45;
       #statDataBuffer.send_comparatorCmd[20] := 16#36;
       #statDataBuffer.send_comparatorCmd[21] := 16#2C;
       #statDataBuffer.send_comparatorCmd[22] := 16#20;
       #LER_IRCheck_Calculate_CompLowerLimit_5(realValue := #moduleInterface.configuration.compLowerLimit,   // "LER_IRCheck_Calculate"
                               stringValue => #statcompLowerLimit);
   END_IF;
   IF #_w8 AND (#statCnt[1625] = 1) THEN
       #statDataBuffer.send_comparatorCmd[24] := 16#45;
       #statDataBuffer.send_comparatorCmd[25] := 16#36;
       #statDataBuffer.send_comparatorCmd[26] := 16#0D;
       #statDataBuffer.send_comparatorCmd[27] := 16#0A;
       #statSendP2PLength_comparatorCmd := 28;
   END_IF;
   IF #_w8 AND (#statCnt[1625] = 2) THEN
       #statDataBuffer.send_comparatorCmd[25] := 16#45;
       #statDataBuffer.send_comparatorCmd[26] := 16#36;
       #statDataBuffer.send_comparatorCmd[27] := 16#0D;
       #statDataBuffer.send_comparatorCmd[28] := 16#0A;
       #statSendP2PLength_comparatorCmd := 29;
   END_IF;
   IF #_w8 AND (#statCnt[1625] = 3) THEN
       #statDataBuffer.send_comparatorCmd[26] := 16#45;
       #statDataBuffer.send_comparatorCmd[27] := 16#36;
       #statDataBuffer.send_comparatorCmd[28] := 16#0D;
       #statDataBuffer.send_comparatorCmd[29] := 16#0A;
       #statSendP2PLength_comparatorCmd := 30;
   END_IF;
   IF #_w8 AND (#statCnt[1625] = 4) THEN
       #statDataBuffer.send_comparatorCmd[27] := 16#45;
       #statDataBuffer.send_comparatorCmd[28] := 16#36;
       #statDataBuffer.send_comparatorCmd[29] := 16#0D;
       #statDataBuffer.send_comparatorCmd[30] := 16#0A;
       #statSendP2PLength_comparatorCmd := 31;
   END_IF;
   IF #_w8 AND ((#statCnt[1625] < 1) OR (#statCnt[1625] > 4)) THEN
       #statDataBuffer.send_comparatorCmd[23] := 16#32;
       #statDataBuffer.send_comparatorCmd[24] := 16#45;
       #statDataBuffer.send_comparatorCmd[25] := 16#36;
       #statDataBuffer.send_comparatorCmd[26] := 16#0D;
       #statDataBuffer.send_comparatorCmd[27] := 16#0A;
       #statSendP2PLength_comparatorCmd := 28;
   END_IF;
   #statTonTimer[1620].TON(IN := #_w2, PT := T#100ms);
   IF #statTonTimer[1620].Q THEN #statStep := 1630; END_IF;
   #statSendRequest[1630] := #statStep = 1630;
   #statTonTimer[1630].TON(IN := #statStep = 1630, PT := T#1000ms);
   #statTonTimer[1631].TON(IN := (#statStep = 1630) AND #statTonTimer[1630].Q, PT := T#1000ms);
   IF #statTonTimer[1631].Q THEN #statStep := 1710; END_IF;
END_REGION

REGION Network 53: STEP 1710~1740 : COMPARATOR CHECK
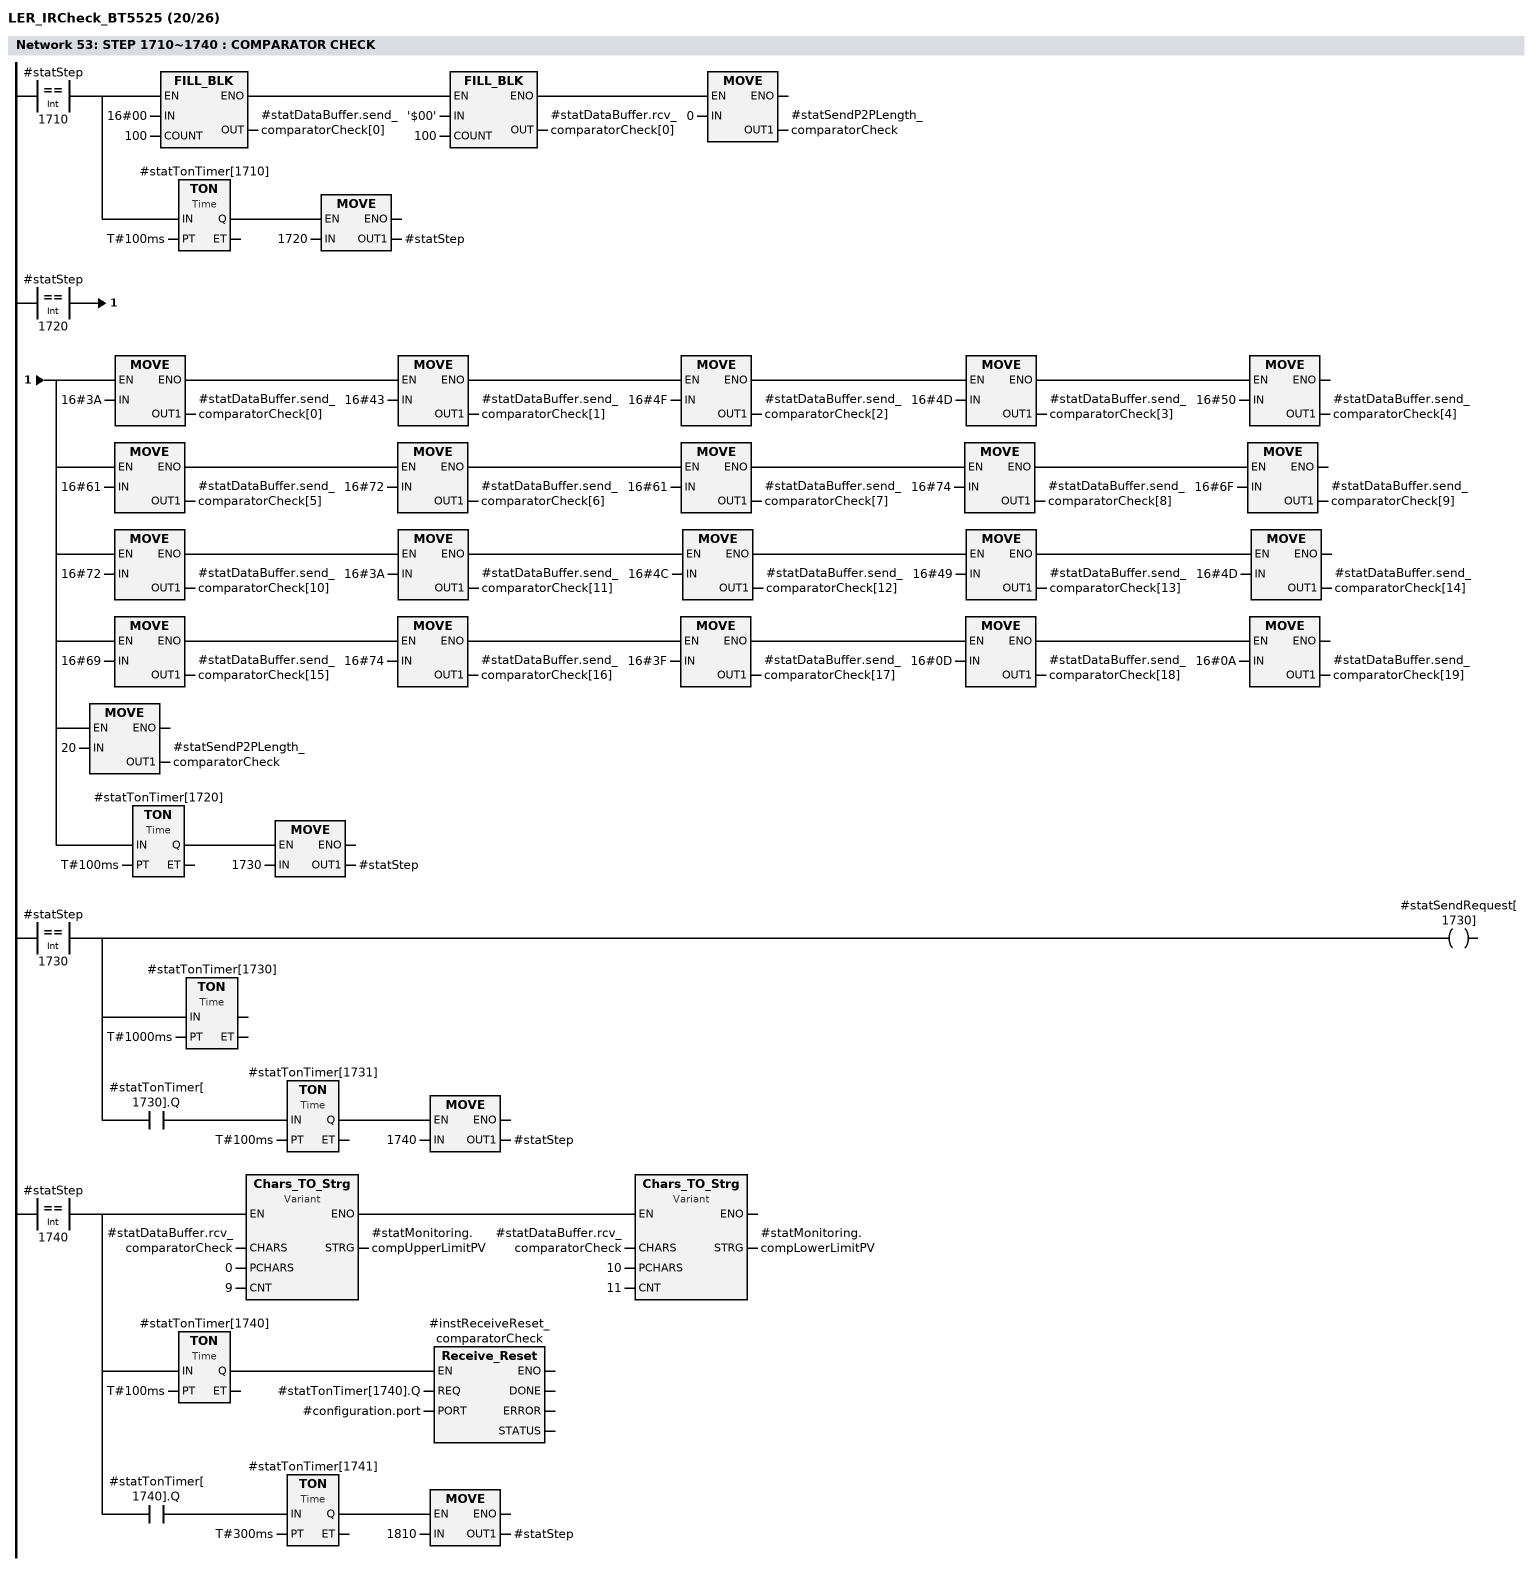
   RUNG wire#powerrail
      { S7_Templates := "SrcType := Int" } EQ_Contact(in1 := #statStep, in2 := 1710)
      wire#w1
      FillBlockI(in := 16#00, count := 100, out => #statDataBuffer.send_comparatorCheck[0])
      FillBlockI(in := '$00', count := 100, out => #statDataBuffer.rcv_comparatorCheck[0])
      Move(in := 0, out1 => #statSendP2PLength_comparatorCheck)
   END_RUNG
   RUNG wire#w1
      { S7_Templates := "time_type := Time" } #statTonTimer[1710].TON(pt := T#100ms, et =>)
      Move(in := 1720, out1 => #statStep)
   END_RUNG
   RUNG wire#powerrail
      { S7_Templates := "SrcType := Int" } EQ_Contact(in1 := #statStep, in2 := 1720)
      wire#w2
      Move(in := 16#3A, out1 => #statDataBuffer.send_comparatorCheck[0])
      Move(in := 16#43, out1 => #statDataBuffer.send_comparatorCheck[1])
      Move(in := 16#4F, out1 => #statDataBuffer.send_comparatorCheck[2])
      Move(in := 16#4D, out1 => #statDataBuffer.send_comparatorCheck[3])
      Move(in := 16#50, out1 => #statDataBuffer.send_comparatorCheck[4])
   END_RUNG
   RUNG wire#w2
      Move(in := 16#61, out1 => #statDataBuffer.send_comparatorCheck[5])
      Move(in := 16#72, out1 => #statDataBuffer.send_comparatorCheck[6])
      Move(in := 16#61, out1 => #statDataBuffer.send_comparatorCheck[7])
      Move(in := 16#74, out1 => #statDataBuffer.send_comparatorCheck[8])
      Move(in := 16#6F, out1 => #statDataBuffer.send_comparatorCheck[9])
   END_RUNG
   RUNG wire#w2
      Move(in := 16#72, out1 => #statDataBuffer.send_comparatorCheck[10])
      Move(in := 16#3A, out1 => #statDataBuffer.send_comparatorCheck[11])
      Move(in := 16#4C, out1 => #statDataBuffer.send_comparatorCheck[12])
      Move(in := 16#49, out1 => #statDataBuffer.send_comparatorCheck[13])
      Move(in := 16#4D, out1 => #statDataBuffer.send_comparatorCheck[14])
   END_RUNG
   RUNG wire#w2
      Move(in := 16#69, out1 => #statDataBuffer.send_comparatorCheck[15])
      Move(in := 16#74, out1 => #statDataBuffer.send_comparatorCheck[16])
      Move(in := 16#3F, out1 => #statDataBuffer.send_comparatorCheck[17])
      Move(in := 16#0D, out1 => #statDataBuffer.send_comparatorCheck[18])
      Move(in := 16#0A, out1 => #statDataBuffer.send_comparatorCheck[19])
   END_RUNG
   RUNG wire#w2
      Move(in := 20, out1 => #statSendP2PLength_comparatorCheck)
   END_RUNG
   RUNG wire#w2
      { S7_Templates := "time_type := Time" } #statTonTimer[1720].TON(pt := T#100ms, et =>)
      Move(in := 1730, out1 => #statStep)
   END_RUNG
   RUNG wire#powerrail
      { S7_Templates := "SrcType := Int" } EQ_Contact(in1 := #statStep, in2 := 1730)
      wire#w3
      Coil( #statSendRequest[1730] )
   END_RUNG
   RUNG wire#w3
      { S7_Templates := "time_type := Time" } #statTonTimer[1730].TON(pt := T#1000ms, et =>)
   END_RUNG
   RUNG wire#w3
      Contact( #statTonTimer[1730].Q )
      { S7_Templates := "time_type := Time" } #statTonTimer[1731].TON(pt := T#100ms, et =>)
      Move(in := 1740, out1 => #statStep)
   END_RUNG
   RUNG wire#powerrail
      { S7_Templates := "SrcType := Int" } EQ_Contact(in1 := #statStep, in2 := 1740)
      wire#w4
      { S7_Templates := "[ptr_type := Variant, str_type := String]" } Chars_TO_Strg(Chars := #statDataBuffer.rcv_comparatorCheck, pChars := 0, Cnt := 9, Strg => #statMonitoring.compUpperLimitPV)
      { S7_Templates := "[ptr_type := Variant, str_type := String]" } Chars_TO_Strg(Chars := #statDataBuffer.rcv_comparatorCheck, pChars := 10, Cnt := 11, Strg => #statMonitoring.compLowerLimitPV)
   END_RUNG
   RUNG wire#w4
      { S7_Templates := "time_type := Time" } #statTonTimer[1740].TON(pt := T#100ms, et =>)
      #instReceiveReset_comparatorCheck.Receive_Reset(REQ := #statTonTimer[1740].Q, PORT := #configuration.port, DONE =>, ERROR =>, STATUS =>)
   END_RUNG
   RUNG wire#w4
      Contact( #statTonTimer[1740].Q )
      { S7_Templates := "time_type := Time" } #statTonTimer[1741].TON(pt := T#300ms, et =>)
      Move(in := 1810, out1 => #statStep)
   END_RUNG
   // the same network as SCL:
   #_w1 := #statStep = 1710;
   IF #_w1 THEN
       FILL_BLK(IN := 16#00, COUNT := 100, OUT => #statDataBuffer.send_comparatorCheck[0]);
       FILL_BLK(IN := '$00', COUNT := 100, OUT => #statDataBuffer.rcv_comparatorCheck[0]);
       #statSendP2PLength_comparatorCheck := 0;
   END_IF;
   #statTonTimer[1710].TON(IN := #_w1, PT := T#100ms);
   IF #statTonTimer[1710].Q THEN #statStep := 1720; END_IF;
   #_w2 := #statStep = 1720;
   IF #_w2 THEN
       #statDataBuffer.send_comparatorCheck[0] := 16#3A;
       #statDataBuffer.send_comparatorCheck[1] := 16#43;
       #statDataBuffer.send_comparatorCheck[2] := 16#4F;
       #statDataBuffer.send_comparatorCheck[3] := 16#4D;
       #statDataBuffer.send_comparatorCheck[4] := 16#50;
       #statDataBuffer.send_comparatorCheck[5] := 16#61;
       #statDataBuffer.send_comparatorCheck[6] := 16#72;
       #statDataBuffer.send_comparatorCheck[7] := 16#61;
       #statDataBuffer.send_comparatorCheck[8] := 16#74;
       #statDataBuffer.send_comparatorCheck[9] := 16#6F;
       #statDataBuffer.send_comparatorCheck[10] := 16#72;
       #statDataBuffer.send_comparatorCheck[11] := 16#3A;
       #statDataBuffer.send_comparatorCheck[12] := 16#4C;
       #statDataBuffer.send_comparatorCheck[13] := 16#49;
       #statDataBuffer.send_comparatorCheck[14] := 16#4D;
       #statDataBuffer.send_comparatorCheck[15] := 16#69;
       #statDataBuffer.send_comparatorCheck[16] := 16#74;
       #statDataBuffer.send_comparatorCheck[17] := 16#3F;
       #statDataBuffer.send_comparatorCheck[18] := 16#0D;
       #statDataBuffer.send_comparatorCheck[19] := 16#0A;
       #statSendP2PLength_comparatorCheck := 20;
   END_IF;
   #statTonTimer[1720].TON(IN := #_w2, PT := T#100ms);
   IF #statTonTimer[1720].Q THEN #statStep := 1730; END_IF;
   #statSendRequest[1730] := #statStep = 1730;
   #statTonTimer[1730].TON(IN := #statStep = 1730, PT := T#1000ms);
   #statTonTimer[1731].TON(IN := (#statStep = 1730) AND #statTonTimer[1730].Q, PT := T#100ms);
   IF #statTonTimer[1731].Q THEN #statStep := 1740; END_IF;
   #_w3 := #statStep = 1740;
   Chars_TO_Strg(EN := #_w3,
                 Chars := #statDataBuffer.rcv_comparatorCheck,
                 pChars := 0,
                 Cnt := 9,
                 Strg => #statMonitoring.compUpperLimitPV,
                 ENO => #_w4);
   IF #_w4 THEN
       Chars_TO_Strg(Chars := #statDataBuffer.rcv_comparatorCheck,
                     pChars := 10,
                     Cnt := 11,
                     Strg => #statMonitoring.compLowerLimitPV);
   END_IF;
   #statTonTimer[1740].TON(IN := #_w3, PT := T#100ms);
   IF #statTonTimer[1740].Q THEN
       #instReceiveReset_comparatorCheck(REQ := #statTonTimer[1740].Q, PORT := #configuration.port);   // Receive_Reset
   END_IF;
   #statTonTimer[1741].TON(IN := #_w3 AND #statTonTimer[1740].Q, PT := T#300ms);
   IF #statTonTimer[1741].Q THEN #statStep := 1810; END_IF;
END_REGION

REGION Network 54: STEP 1810~1830 : BDD CCV COMMAND
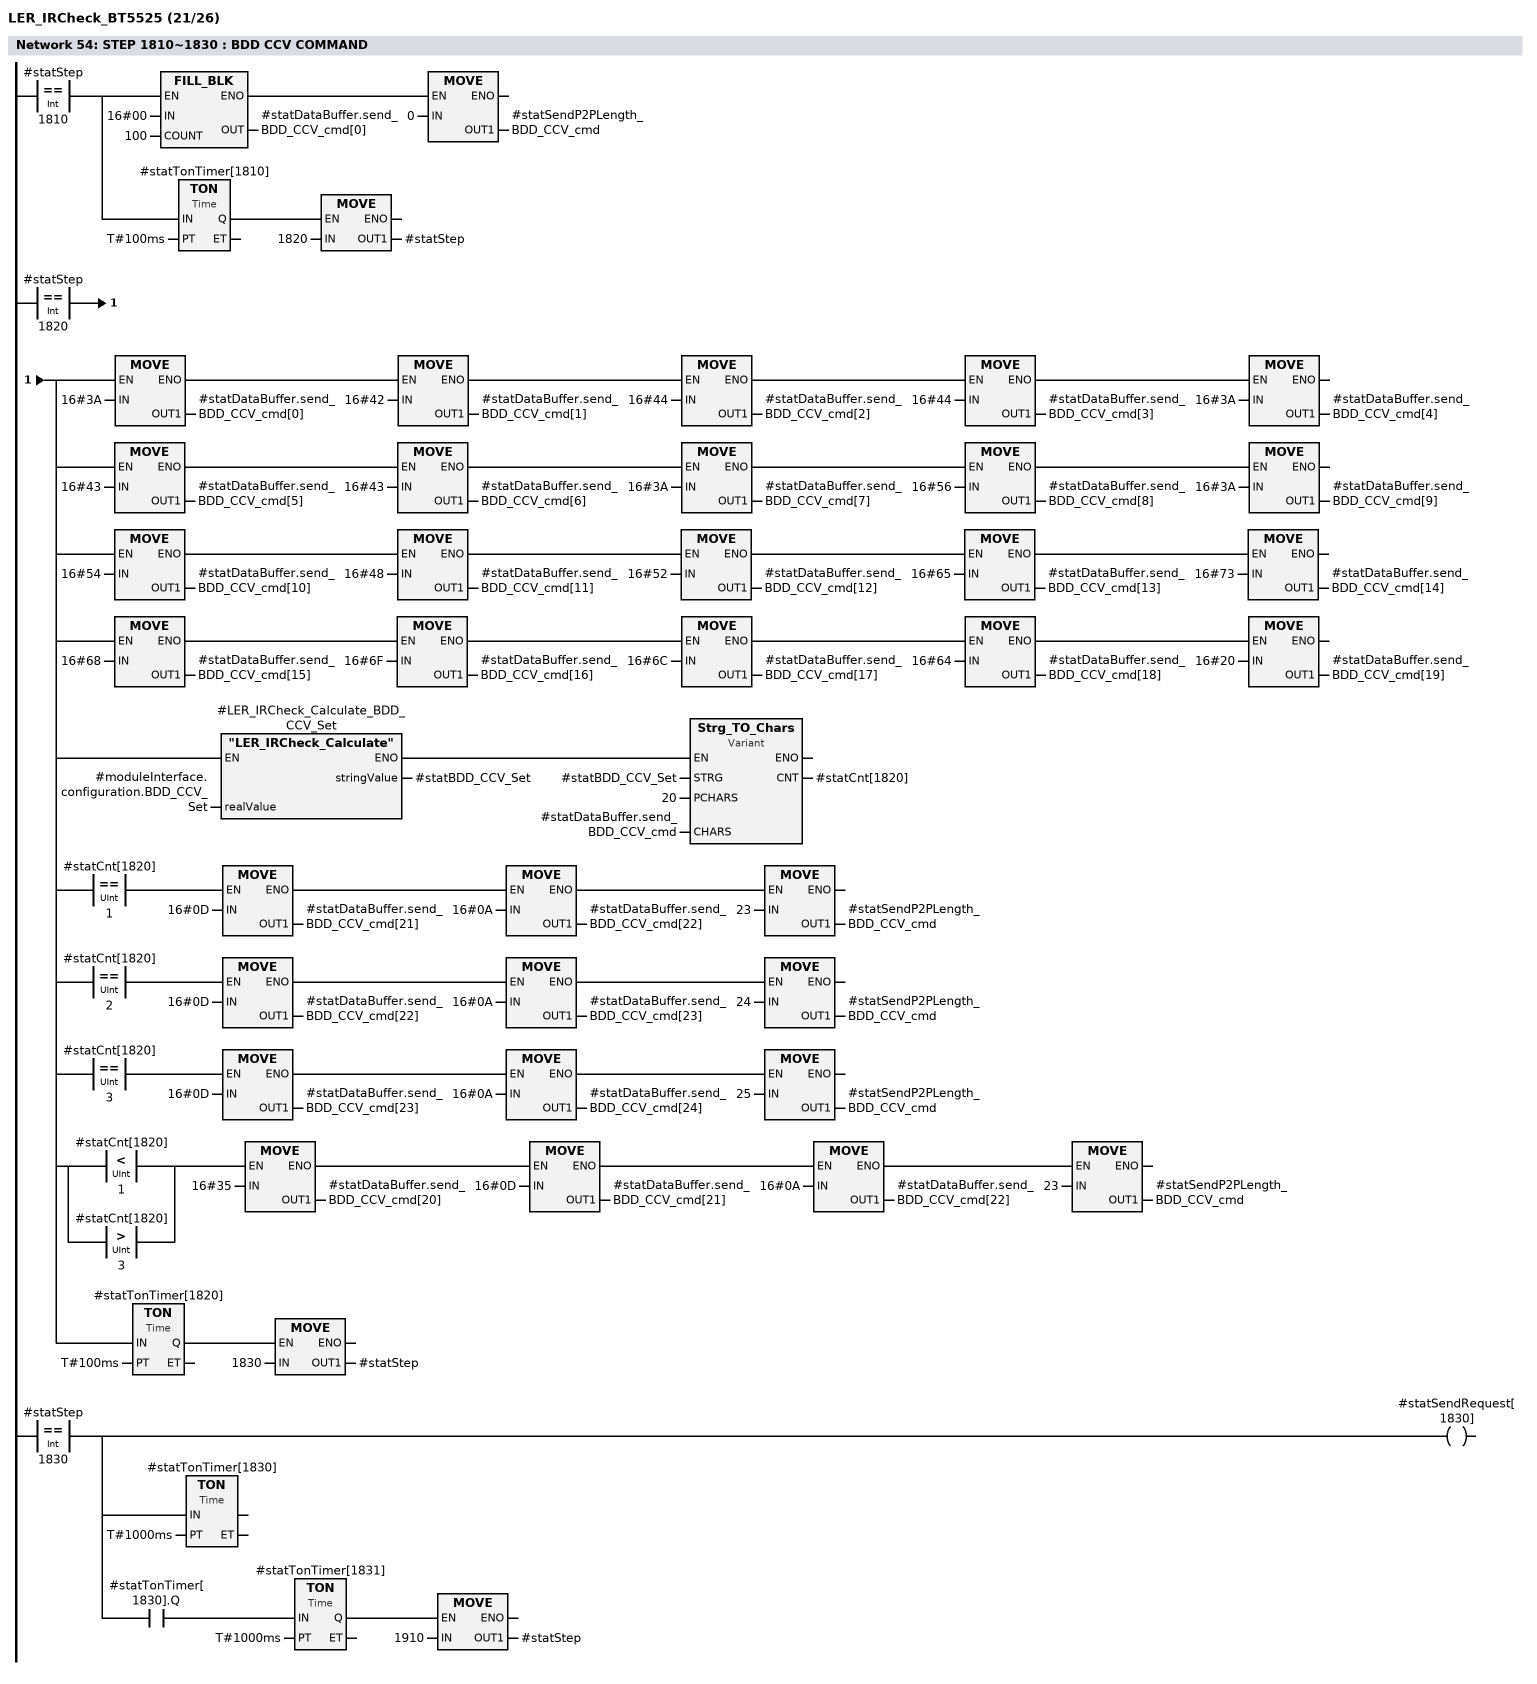
   RUNG wire#powerrail
      { S7_Templates := "SrcType := Int" } EQ_Contact(in1 := #statStep, in2 := 1810)
      wire#w1
      FillBlockI(in := 16#00, count := 100, out => #statDataBuffer.send_BDD_CCV_cmd[0])
      Move(in := 0, out1 => #statSendP2PLength_BDD_CCV_cmd)
   END_RUNG
   RUNG wire#w1
      { S7_Templates := "time_type := Time" } #statTonTimer[1810].TON(pt := T#100ms, et =>)
      Move(in := 1820, out1 => #statStep)
   END_RUNG
   RUNG wire#powerrail
      { S7_Templates := "SrcType := Int" } EQ_Contact(in1 := #statStep, in2 := 1820)
      wire#w2
      Move(in := 16#3A, out1 => #statDataBuffer.send_BDD_CCV_cmd[0])
      Move(in := 16#42, out1 => #statDataBuffer.send_BDD_CCV_cmd[1])
      Move(in := 16#44, out1 => #statDataBuffer.send_BDD_CCV_cmd[2])
      Move(in := 16#44, out1 => #statDataBuffer.send_BDD_CCV_cmd[3])
      Move(in := 16#3A, out1 => #statDataBuffer.send_BDD_CCV_cmd[4])
   END_RUNG
   RUNG wire#w2
      Move(in := 16#43, out1 => #statDataBuffer.send_BDD_CCV_cmd[5])
      Move(in := 16#43, out1 => #statDataBuffer.send_BDD_CCV_cmd[6])
      Move(in := 16#3A, out1 => #statDataBuffer.send_BDD_CCV_cmd[7])
      Move(in := 16#56, out1 => #statDataBuffer.send_BDD_CCV_cmd[8])
      Move(in := 16#3A, out1 => #statDataBuffer.send_BDD_CCV_cmd[9])
   END_RUNG
   RUNG wire#w2
      Move(in := 16#54, out1 => #statDataBuffer.send_BDD_CCV_cmd[10])
      Move(in := 16#48, out1 => #statDataBuffer.send_BDD_CCV_cmd[11])
      Move(in := 16#52, out1 => #statDataBuffer.send_BDD_CCV_cmd[12])
      Move(in := 16#65, out1 => #statDataBuffer.send_BDD_CCV_cmd[13])
      Move(in := 16#73, out1 => #statDataBuffer.send_BDD_CCV_cmd[14])
   END_RUNG
   RUNG wire#w2
      Move(in := 16#68, out1 => #statDataBuffer.send_BDD_CCV_cmd[15])
      Move(in := 16#6F, out1 => #statDataBuffer.send_BDD_CCV_cmd[16])
      Move(in := 16#6C, out1 => #statDataBuffer.send_BDD_CCV_cmd[17])
      Move(in := 16#64, out1 => #statDataBuffer.send_BDD_CCV_cmd[18])
      Move(in := 16#20, out1 => #statDataBuffer.send_BDD_CCV_cmd[19])
   END_RUNG
   RUNG wire#w2
      #LER_IRCheck_Calculate_BDD_CCV_Set(realValue := #moduleInterface.configuration.BDD_CCV_Set, stringValue => #statBDD_CCV_Set)
      { S7_Templates := "[ptr_type := Variant, strg_type := String]" } Strg_TO_Chars(Strg := #statBDD_CCV_Set, pChars := 20, Chars := #statDataBuffer.send_BDD_CCV_cmd, Cnt => #statCnt[1820])
   END_RUNG
   RUNG wire#w2
      { S7_Templates := "SrcType := UInt" } EQ_Contact(in1 := #statCnt[1820], in2 := 1)
      Move(in := 16#0D, out1 => #statDataBuffer.send_BDD_CCV_cmd[21])
      Move(in := 16#0A, out1 => #statDataBuffer.send_BDD_CCV_cmd[22])
      Move(in := 23, out1 => #statSendP2PLength_BDD_CCV_cmd)
   END_RUNG
   RUNG wire#w2
      { S7_Templates := "SrcType := UInt" } EQ_Contact(in1 := #statCnt[1820], in2 := 2)
      Move(in := 16#0D, out1 => #statDataBuffer.send_BDD_CCV_cmd[22])
      Move(in := 16#0A, out1 => #statDataBuffer.send_BDD_CCV_cmd[23])
      Move(in := 24, out1 => #statSendP2PLength_BDD_CCV_cmd)
   END_RUNG
   RUNG wire#w2
      { S7_Templates := "SrcType := UInt" } EQ_Contact(in1 := #statCnt[1820], in2 := 3)
      Move(in := 16#0D, out1 => #statDataBuffer.send_BDD_CCV_cmd[23])
      Move(in := 16#0A, out1 => #statDataBuffer.send_BDD_CCV_cmd[24])
      Move(in := 25, out1 => #statSendP2PLength_BDD_CCV_cmd)
   END_RUNG
   RUNG wire#w2
      { S7_Templates := "SrcType := UInt" } LT_Contact(in1 := #statCnt[1820], in2 := 1)
      wire#w3
      Move(in := 16#35, out1 => #statDataBuffer.send_BDD_CCV_cmd[20])
      Move(in := 16#0D, out1 => #statDataBuffer.send_BDD_CCV_cmd[21])
      Move(in := 16#0A, out1 => #statDataBuffer.send_BDD_CCV_cmd[22])
      Move(in := 23, out1 => #statSendP2PLength_BDD_CCV_cmd)
   END_RUNG
   RUNG wire#w2
      { S7_Templates := "SrcType := UInt" } GT_Contact(in1 := #statCnt[1820], in2 := 3)
   END_RUNG wire#w3
   RUNG wire#w2
      { S7_Templates := "time_type := Time" } #statTonTimer[1820].TON(pt := T#100ms, et =>)
      Move(in := 1830, out1 => #statStep)
   END_RUNG
   RUNG wire#powerrail
      { S7_Templates := "SrcType := Int" } EQ_Contact(in1 := #statStep, in2 := 1830)
      wire#w4
      Coil( #statSendRequest[1830] )
   END_RUNG
   RUNG wire#w4
      { S7_Templates := "time_type := Time" } #statTonTimer[1830].TON(pt := T#1000ms, et =>)
   END_RUNG
   RUNG wire#w4
      Contact( #statTonTimer[1830].Q )
      { S7_Templates := "time_type := Time" } #statTonTimer[1831].TON(pt := T#1000ms, et =>)
      Move(in := 1910, out1 => #statStep)
   END_RUNG
   // the same network as SCL:
   #_w1 := #statStep = 1810;
   IF #_w1 THEN
       FILL_BLK(IN := 16#00, COUNT := 100, OUT => #statDataBuffer.send_BDD_CCV_cmd[0]);
       #statSendP2PLength_BDD_CCV_cmd := 0;
   END_IF;
   #statTonTimer[1810].TON(IN := #_w1, PT := T#100ms);
   IF #statTonTimer[1810].Q THEN #statStep := 1820; END_IF;
   #_w2 := #statStep = 1820;
   IF #_w2 THEN
       #statDataBuffer.send_BDD_CCV_cmd[0] := 16#3A;
       #statDataBuffer.send_BDD_CCV_cmd[1] := 16#42;
       #statDataBuffer.send_BDD_CCV_cmd[2] := 16#44;
       #statDataBuffer.send_BDD_CCV_cmd[3] := 16#44;
       #statDataBuffer.send_BDD_CCV_cmd[4] := 16#3A;
       #statDataBuffer.send_BDD_CCV_cmd[5] := 16#43;
       #statDataBuffer.send_BDD_CCV_cmd[6] := 16#43;
       #statDataBuffer.send_BDD_CCV_cmd[7] := 16#3A;
       #statDataBuffer.send_BDD_CCV_cmd[8] := 16#56;
       #statDataBuffer.send_BDD_CCV_cmd[9] := 16#3A;
       #statDataBuffer.send_BDD_CCV_cmd[10] := 16#54;
       #statDataBuffer.send_BDD_CCV_cmd[11] := 16#48;
       #statDataBuffer.send_BDD_CCV_cmd[12] := 16#52;
       #statDataBuffer.send_BDD_CCV_cmd[13] := 16#65;
       #statDataBuffer.send_BDD_CCV_cmd[14] := 16#73;
       #statDataBuffer.send_BDD_CCV_cmd[15] := 16#68;
       #statDataBuffer.send_BDD_CCV_cmd[16] := 16#6F;
       #statDataBuffer.send_BDD_CCV_cmd[17] := 16#6C;
       #statDataBuffer.send_BDD_CCV_cmd[18] := 16#64;
       #statDataBuffer.send_BDD_CCV_cmd[19] := 16#20;
   END_IF;
   #LER_IRCheck_Calculate_BDD_CCV_Set(EN := #_w2,   // "LER_IRCheck_Calculate"
                           realValue := #moduleInterface.configuration.BDD_CCV_Set,
                           stringValue => #statBDD_CCV_Set,
                           ENO => #_w3);
   IF #_w3 THEN
       Strg_TO_Chars(Strg := #statBDD_CCV_Set,
                     pChars := 20,
                     Chars := #statDataBuffer.send_BDD_CCV_cmd,
                     Cnt => #statCnt[1820]);
   END_IF;
   IF #_w2 AND (#statCnt[1820] = 1) THEN
       #statDataBuffer.send_BDD_CCV_cmd[21] := 16#0D;
       #statDataBuffer.send_BDD_CCV_cmd[22] := 16#0A;
       #statSendP2PLength_BDD_CCV_cmd := 23;
   END_IF;
   IF #_w2 AND (#statCnt[1820] = 2) THEN
       #statDataBuffer.send_BDD_CCV_cmd[22] := 16#0D;
       #statDataBuffer.send_BDD_CCV_cmd[23] := 16#0A;
       #statSendP2PLength_BDD_CCV_cmd := 24;
   END_IF;
   IF #_w2 AND (#statCnt[1820] = 3) THEN
       #statDataBuffer.send_BDD_CCV_cmd[23] := 16#0D;
       #statDataBuffer.send_BDD_CCV_cmd[24] := 16#0A;
       #statSendP2PLength_BDD_CCV_cmd := 25;
   END_IF;
   IF #_w2 AND ((#statCnt[1820] < 1) OR (#statCnt[1820] > 3)) THEN
       #statDataBuffer.send_BDD_CCV_cmd[20] := 16#35;
       #statDataBuffer.send_BDD_CCV_cmd[21] := 16#0D;
       #statDataBuffer.send_BDD_CCV_cmd[22] := 16#0A;
       #statSendP2PLength_BDD_CCV_cmd := 23;
   END_IF;
   #statTonTimer[1820].TON(IN := #_w2, PT := T#100ms);
   IF #statTonTimer[1820].Q THEN #statStep := 1830; END_IF;
   #statSendRequest[1830] := #statStep = 1830;
   #statTonTimer[1830].TON(IN := #statStep = 1830, PT := T#1000ms);
   #statTonTimer[1831].TON(IN := (#statStep = 1830) AND #statTonTimer[1830].Q, PT := T#1000ms);
   IF #statTonTimer[1831].Q THEN #statStep := 1910; END_IF;
END_REGION

